REGION Network 34: TMP - ERROR - Protrusión
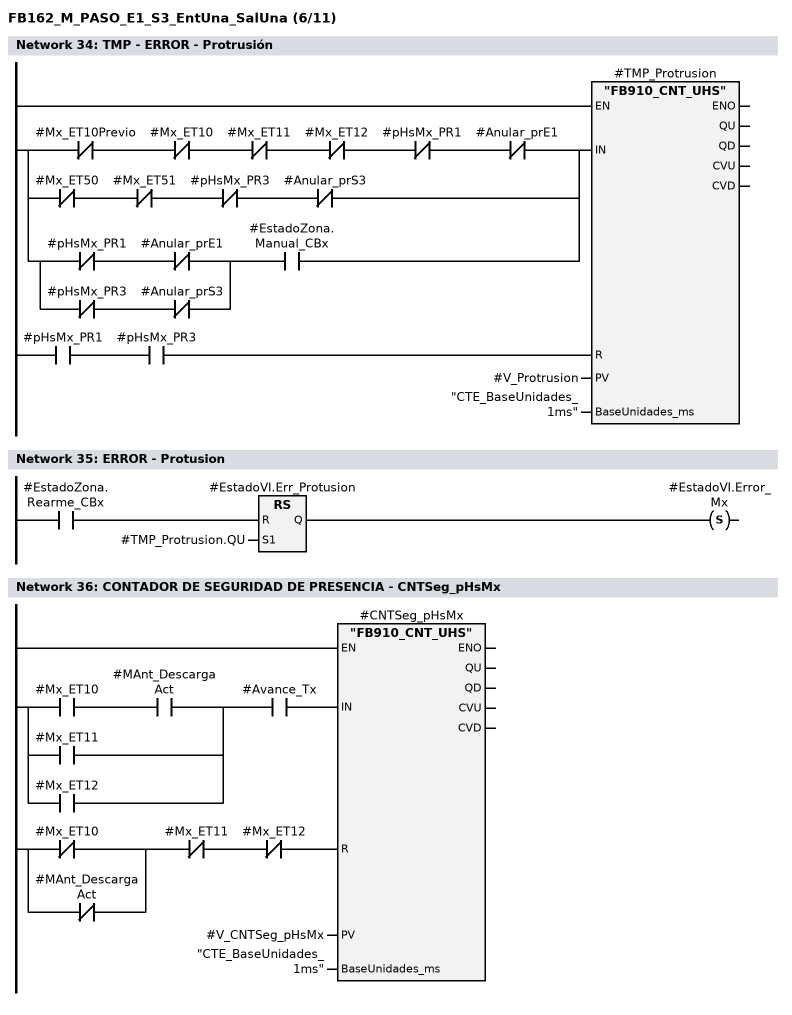
   RUNG wire#powerrail
      #TMP_Protrusion(IN := wire#w2, R := wire#w3, PV := #V_Protrusion, BaseUnidades_ms := "CTE_BaseUnidades_1ms", QU =>, QD =>, CVU =>, CVD =>)
   END_RUNG
   RUNG wire#powerrail
      I_Contact( #Mx_ET10Previo )
      I_Contact( #Mx_ET10 )
      I_Contact( #Mx_ET11 )
      I_Contact( #Mx_ET12 )
      I_Contact( #pHsMx_PR1 )
      I_Contact( #Anular_prE1 )
   END_RUNG wire#w2
   RUNG wire#powerrail
      I_Contact( #Mx_ET50 )
      I_Contact( #Mx_ET51 )
      I_Contact( #pHsMx_PR3 )
      I_Contact( #Anular_prS3 )
   END_RUNG wire#w2
   RUNG wire#powerrail
      I_Contact( #pHsMx_PR1 )
      I_Contact( #Anular_prE1 )
      wire#w1
      Contact( #EstadoZona.Manual_CBx )
   END_RUNG wire#w2
   RUNG wire#powerrail
      I_Contact( #pHsMx_PR3 )
      I_Contact( #Anular_prS3 )
   END_RUNG wire#w1
   RUNG wire#powerrail
      Contact( #pHsMx_PR1 )
      Contact( #pHsMx_PR3 )
   END_RUNG wire#w3
   // the same network as SCL:
   #TMP_Protrusion(IN := (NOT #Mx_ET10Previo AND NOT #Mx_ET10 AND NOT #Mx_ET11 AND NOT #Mx_ET12 AND NOT #pHsMx_PR1 AND NOT #Anular_prE1) OR (NOT #Mx_ET50 AND NOT #Mx_ET51 AND NOT #pHsMx_PR3 AND NOT #Anular_prS3) OR (((NOT #pHsMx_PR1 AND NOT #Anular_prE1) OR (NOT #pHsMx_PR3 AND NOT #Anular_prS3)) AND #EstadoZona.Manual_CBx),   // "FB910_CNT_UHS"
                   R := #pHsMx_PR1 AND #pHsMx_PR3,
                   PV := #V_Protrusion,
                   BaseUnidades_ms := "CTE_BaseUnidades_1ms");
END_REGION

REGION Network 35: ERROR - Protusion
   RUNG wire#powerrail
      Contact( #EstadoZona.Rearme_CBx )
      S_RS(operand := #EstadoVI.Err_Protusion, s1 := #TMP_Protrusion.QU)
      S_Coil( #EstadoVI.Error_Mx )
   END_RUNG
   // the same network as SCL:
   IF #EstadoZona.Rearme_CBx THEN
       #EstadoVI.Err_Protusion := FALSE;   // RS flip-flop
   END_IF;
   IF #TMP_Protrusion.QU THEN #EstadoVI.Err_Protusion := TRUE; END_IF;
   IF #EstadoVI.Err_Protusion THEN #EstadoVI.Error_Mx := TRUE; END_IF;
END_REGION

REGION Network 36: CONTADOR DE SEGURIDAD DE PRESENCIA - CNTSeg_pHsMx
   RUNG wire#powerrail
      #CNTSeg_pHsMx(IN := wire#w2, R := wire#w4, PV := #V_CNTSeg_pHsMx, BaseUnidades_ms := "CTE_BaseUnidades_1ms", QU =>, QD =>, CVU =>, CVD =>)
   END_RUNG
   RUNG wire#powerrail
      Contact( #Mx_ET10 )
      Contact( #MAnt_DescargaAct )
      wire#w1
      Contact( #Avance_Tx )
   END_RUNG wire#w2
   RUNG wire#powerrail
      Contact( #Mx_ET11 )
   END_RUNG wire#w1
   RUNG wire#powerrail
      Contact( #Mx_ET12 )
   END_RUNG wire#w1
   RUNG wire#powerrail
      I_Contact( #Mx_ET10 )
      wire#w3
      I_Contact( #Mx_ET11 )
      I_Contact( #Mx_ET12 )
   END_RUNG wire#w4
   RUNG wire#powerrail
      I_Contact( #MAnt_DescargaAct )
   END_RUNG wire#w3
   // the same network as SCL:
   #CNTSeg_pHsMx(IN := ((#Mx_ET10 AND #MAnt_DescargaAct) OR #Mx_ET11 OR #Mx_ET12) AND #Avance_Tx,   // "FB910_CNT_UHS"
                 R := (NOT #Mx_ET10 OR NOT #MAnt_DescargaAct) AND NOT #Mx_ET11 AND NOT #Mx_ET12,
                 PV := #V_CNTSeg_pHsMx,
                 BaseUnidades_ms := "CTE_BaseUnidades_1ms");
END_REGION

REGION Network 37: CONTADOR DE PRESENCIA - CNT_pHsMx
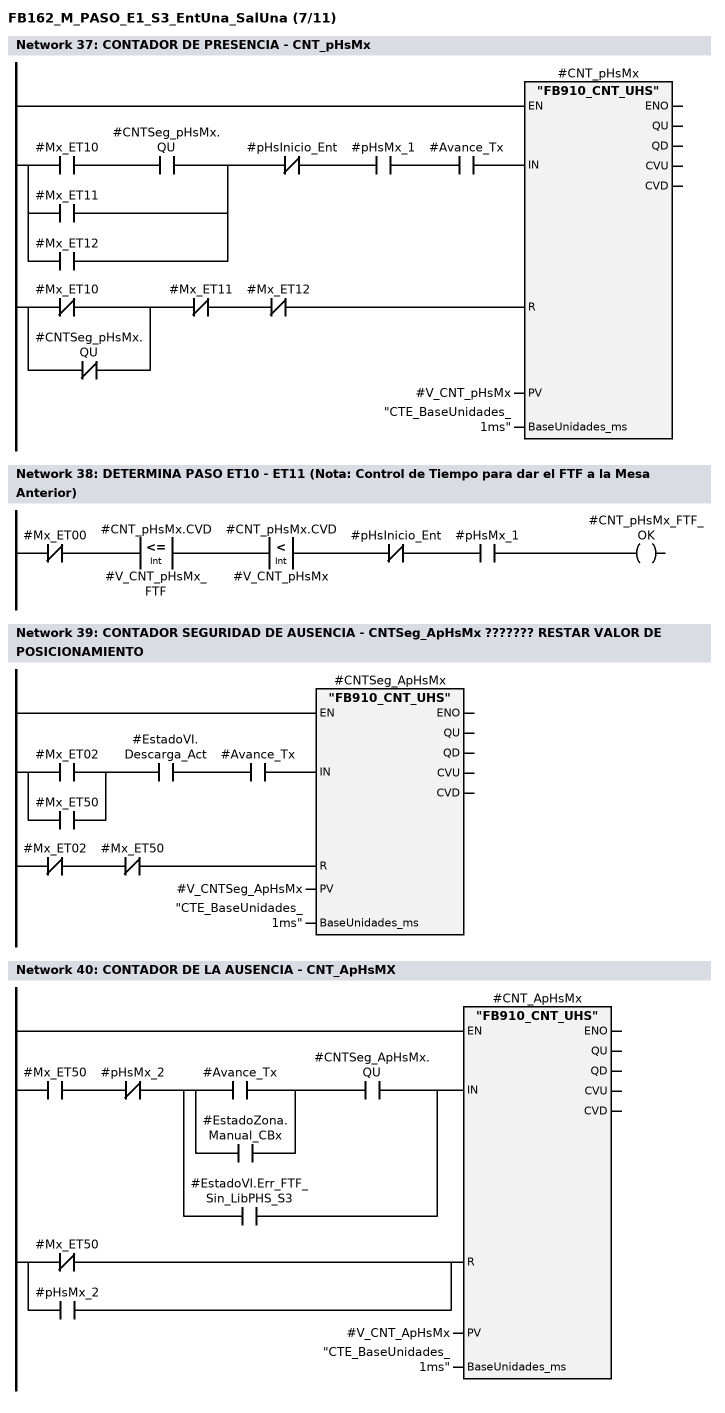
   RUNG wire#powerrail
      #CNT_pHsMx(IN := wire#w2, R := wire#w4, PV := #V_CNT_pHsMx, BaseUnidades_ms := "CTE_BaseUnidades_1ms", QU =>, QD =>, CVU =>, CVD =>)
   END_RUNG
   RUNG wire#powerrail
      Contact( #Mx_ET10 )
      Contact( #CNTSeg_pHsMx.QU )
      wire#w1
      I_Contact( #pHsInicio_Ent )
      Contact( #pHsMx_1 )
      Contact( #Avance_Tx )
   END_RUNG wire#w2
   RUNG wire#powerrail
      Contact( #Mx_ET11 )
   END_RUNG wire#w1
   RUNG wire#powerrail
      Contact( #Mx_ET12 )
   END_RUNG wire#w1
   RUNG wire#powerrail
      I_Contact( #Mx_ET10 )
      wire#w3
      I_Contact( #Mx_ET11 )
      I_Contact( #Mx_ET12 )
   END_RUNG wire#w4
   RUNG wire#powerrail
      I_Contact( #CNTSeg_pHsMx.QU )
   END_RUNG wire#w3
   // the same network as SCL:
   #CNT_pHsMx(IN := ((#Mx_ET10 AND #CNTSeg_pHsMx.QU) OR #Mx_ET11 OR #Mx_ET12) AND NOT #pHsInicio_Ent AND #pHsMx_1 AND #Avance_Tx,   // "FB910_CNT_UHS"
              R := (NOT #Mx_ET10 OR NOT #CNTSeg_pHsMx.QU) AND NOT #Mx_ET11 AND NOT #Mx_ET12,
              PV := #V_CNT_pHsMx,
              BaseUnidades_ms := "CTE_BaseUnidades_1ms");
END_REGION

REGION Network 38: DETERMINA PASO ET10 - ET11 (Nota: Control de Tiempo para dar el FTF a la Mesa Anterior)
   RUNG wire#powerrail
      I_Contact( #Mx_ET00 )
      { S7_Templates := "SrcType := Int" } LE_Contact(in1 := #CNT_pHsMx.CVD, in2 := #V_CNT_pHsMx_FTF)
      { S7_Templates := "SrcType := Int" } LT_Contact(in1 := #CNT_pHsMx.CVD, in2 := #V_CNT_pHsMx)
      I_Contact( #pHsInicio_Ent )
      Contact( #pHsMx_1 )
      Coil( #CNT_pHsMx_FTF_OK )
   END_RUNG
   // the same network as SCL:
   #CNT_pHsMx_FTF_OK := NOT #Mx_ET00 AND (#CNT_pHsMx.CVD <= #V_CNT_pHsMx_FTF) AND (#CNT_pHsMx.CVD < #V_CNT_pHsMx) AND NOT #pHsInicio_Ent AND #pHsMx_1;
END_REGION

REGION Network 39: CONTADOR SEGURIDAD DE AUSENCIA - CNTSeg_ApHsMx ??????? RESTAR VALOR DE POSICIONAMIENTO
   RUNG wire#powerrail
      #CNTSeg_ApHsMx(IN := wire#w2, R := wire#w3, PV := #V_CNTSeg_ApHsMx, BaseUnidades_ms := "CTE_BaseUnidades_1ms", QU =>, QD =>, CVU =>, CVD =>)
   END_RUNG
   RUNG wire#powerrail
      Contact( #Mx_ET02 )
      wire#w1
      Contact( #EstadoVI.Descarga_Act )
      Contact( #Avance_Tx )
   END_RUNG wire#w2
   RUNG wire#powerrail
      Contact( #Mx_ET50 )
   END_RUNG wire#w1
   RUNG wire#powerrail
      I_Contact( #Mx_ET02 )
      I_Contact( #Mx_ET50 )
   END_RUNG wire#w3
   // the same network as SCL:
   #CNTSeg_ApHsMx(IN := (#Mx_ET02 OR #Mx_ET50) AND #EstadoVI.Descarga_Act AND #Avance_Tx,   // "FB910_CNT_UHS"
                  R := NOT #Mx_ET02 AND NOT #Mx_ET50,
                  PV := #V_CNTSeg_ApHsMx,
                  BaseUnidades_ms := "CTE_BaseUnidades_1ms");
END_REGION

REGION Network 40: CONTADOR DE LA AUSENCIA - CNT_ApHsMX
   RUNG wire#powerrail
      #CNT_ApHsMx(IN := wire#w3, R := wire#w4, PV := #V_CNT_ApHsMx, BaseUnidades_ms := "CTE_BaseUnidades_1ms", QU =>, QD =>, CVU =>, CVD =>)
   END_RUNG
   RUNG wire#powerrail
      Contact( #Mx_ET50 )
      I_Contact( #pHsMx_2 )
      wire#w1
      Contact( #Avance_Tx )
      wire#w2
      Contact( #CNTSeg_ApHsMx.QU )
   END_RUNG wire#w3
   RUNG wire#w1
      Contact( #EstadoZona.Manual_CBx )
   END_RUNG wire#w2
   RUNG wire#w1
      Contact( #EstadoVI.Err_FTF_Sin_LibPHS_S3 )
   END_RUNG wire#w3
   RUNG wire#powerrail
      I_Contact( #Mx_ET50 )
   END_RUNG wire#w4
   RUNG wire#powerrail
      Contact( #pHsMx_2 )
   END_RUNG wire#w4
   // the same network as SCL:
   #CNT_ApHsMx(IN := #Mx_ET50 AND NOT #pHsMx_2 AND (((#Avance_Tx OR #EstadoZona.Manual_CBx) AND #CNTSeg_ApHsMx.QU) OR #EstadoVI.Err_FTF_Sin_LibPHS_S3),   // "FB910_CNT_UHS"
               R := NOT #Mx_ET50 OR #pHsMx_2,
               PV := #V_CNT_ApHsMx,
               BaseUnidades_ms := "CTE_BaseUnidades_1ms");
END_REGION

REGION Network 41: VARIABLES AUXILIARES - Fin de Reset
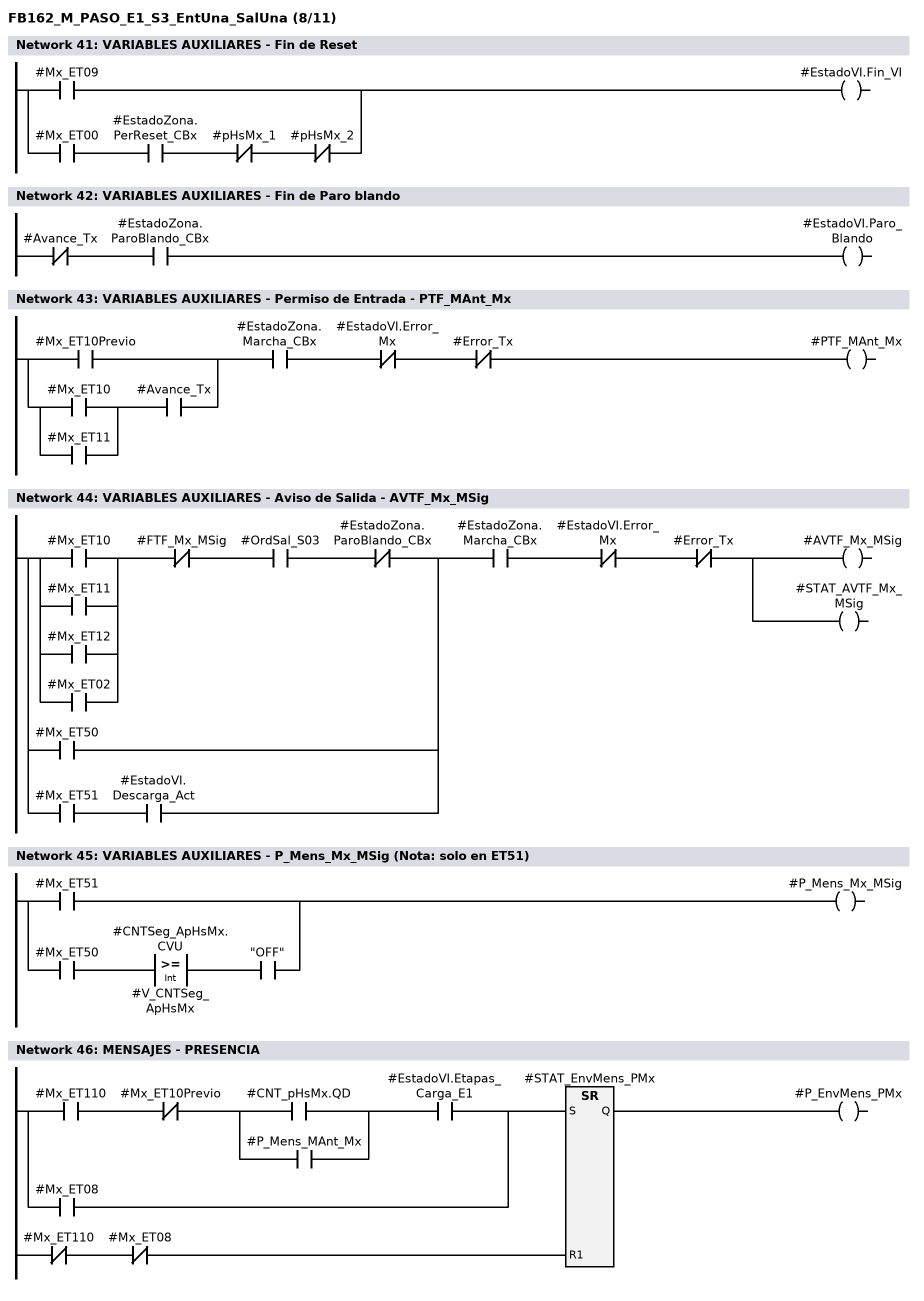
   RUNG wire#powerrail
      Contact( #Mx_ET09 )
      wire#w1
      Coil( #EstadoVI.Fin_VI )
   END_RUNG
   RUNG wire#powerrail
      Contact( #Mx_ET00 )
      Contact( #EstadoZona.PerReset_CBx )
      I_Contact( #pHsMx_1 )
      I_Contact( #pHsMx_2 )
   END_RUNG wire#w1
   // the same network as SCL:
   #EstadoVI.Fin_VI := #Mx_ET09 OR (#Mx_ET00 AND #EstadoZona.PerReset_CBx AND NOT #pHsMx_1 AND NOT #pHsMx_2);
END_REGION

REGION Network 42: VARIABLES AUXILIARES - Fin de Paro blando
   RUNG wire#powerrail
      I_Contact( #Avance_Tx )
      Contact( #EstadoZona.ParoBlando_CBx )
      Coil( #EstadoVI.Paro_Blando )
   END_RUNG
   // the same network as SCL:
   #EstadoVI.Paro_Blando := NOT #Avance_Tx AND #EstadoZona.ParoBlando_CBx;
END_REGION

REGION Network 43: VARIABLES AUXILIARES - Permiso de Entrada - PTF_MAnt_Mx
   RUNG wire#powerrail
      Contact( #Mx_ET10Previo )
      wire#w1
      Contact( #EstadoZona.Marcha_CBx )
      I_Contact( #EstadoVI.Error_Mx )
      I_Contact( #Error_Tx )
      Coil( #PTF_MAnt_Mx )
   END_RUNG
   RUNG wire#powerrail
      Contact( #Mx_ET10 )
      wire#w2
      Contact( #Avance_Tx )
   END_RUNG wire#w1
   RUNG wire#powerrail
      Contact( #Mx_ET11 )
   END_RUNG wire#w2
   // the same network as SCL:
   #PTF_MAnt_Mx := (#Mx_ET10Previo OR ((#Mx_ET10 OR #Mx_ET11) AND #Avance_Tx)) AND #EstadoZona.Marcha_CBx AND NOT #EstadoVI.Error_Mx AND NOT #Error_Tx;
END_REGION

REGION Network 44: VARIABLES AUXILIARES - Aviso de Salida - AVTF_Mx_MSig
   RUNG wire#powerrail
      Contact( #Mx_ET10 )
      wire#w1
      I_Contact( #FTF_Mx_MSig )
      Contact( #OrdSal_S03 )
      I_Contact( #EstadoZona.ParoBlando_CBx )
      wire#w2
      Contact( #EstadoZona.Marcha_CBx )
      I_Contact( #EstadoVI.Error_Mx )
      I_Contact( #Error_Tx )
      wire#w3
      Coil( #AVTF_Mx_MSig )
   END_RUNG
   RUNG wire#powerrail
      Contact( #Mx_ET11 )
   END_RUNG wire#w1
   RUNG wire#powerrail
      Contact( #Mx_ET12 )
   END_RUNG wire#w1
   RUNG wire#powerrail
      Contact( #Mx_ET02 )
   END_RUNG wire#w1
   RUNG wire#powerrail
      Contact( #Mx_ET50 )
   END_RUNG wire#w2
   RUNG wire#powerrail
      Contact( #Mx_ET51 )
      Contact( #EstadoVI.Descarga_Act )
   END_RUNG wire#w2
   RUNG wire#w3
      Coil( #STAT_AVTF_Mx_MSig )
   END_RUNG
   // the same network as SCL:
   #AVTF_Mx_MSig := (((#Mx_ET10 OR #Mx_ET11 OR #Mx_ET12 OR #Mx_ET02) AND NOT #FTF_Mx_MSig AND #OrdSal_S03 AND NOT #EstadoZona.ParoBlando_CBx) OR #Mx_ET50 OR (#Mx_ET51 AND #EstadoVI.Descarga_Act)) AND #EstadoZona.Marcha_CBx AND NOT #EstadoVI.Error_Mx AND NOT #Error_Tx;
   #STAT_AVTF_Mx_MSig := #AVTF_Mx_MSig;
END_REGION

REGION Network 45: VARIABLES AUXILIARES - P_Mens_Mx_MSig (Nota: solo en ET51)
   RUNG wire#powerrail
      Contact( #Mx_ET51 )
      wire#w1
      Coil( #P_Mens_Mx_MSig )
   END_RUNG
   RUNG wire#powerrail
      Contact( #Mx_ET50 )
      { S7_Templates := "SrcType := Int" } GE_Contact(in1 := #CNTSeg_ApHsMx.CVU, in2 := #V_CNTSeg_ApHsMx)
      Contact( "OFF" )
   END_RUNG wire#w1
   // the same network as SCL:
   #P_Mens_Mx_MSig := #Mx_ET51 OR (#Mx_ET50 AND (#CNTSeg_ApHsMx.CVU >= #V_CNTSeg_ApHsMx) AND "OFF");
END_REGION

REGION Network 46: MENSAJES - PRESENCIA
   RUNG wire#powerrail
      Contact( #Mx_ET110 )
      I_Contact( #Mx_ET10Previo )
      wire#w1
      Contact( #CNT_pHsMx.QD )
      wire#w2
      Contact( #EstadoVI.Etapas_Carga_E1 )
      wire#w3
      S_SR(operand := #STAT_EnvMens_PMx, r1 := wire#w4)
      Coil( #P_EnvMens_PMx )
   END_RUNG
   RUNG wire#w1
      Contact( #P_Mens_MAnt_Mx )
   END_RUNG wire#w2
   RUNG wire#powerrail
      Contact( #Mx_ET08 )
   END_RUNG wire#w3
   RUNG wire#powerrail
      I_Contact( #Mx_ET110 )
      I_Contact( #Mx_ET08 )
   END_RUNG wire#w4
   // the same network as SCL:
   IF (#Mx_ET110 AND NOT #Mx_ET10Previo AND (#CNT_pHsMx.QD OR #P_Mens_MAnt_Mx) AND #EstadoVI.Etapas_Carga_E1) OR #Mx_ET08 THEN
       #STAT_EnvMens_PMx := TRUE;   // SR flip-flop
   END_IF;
   IF NOT #Mx_ET110 AND NOT #Mx_ET08 THEN #STAT_EnvMens_PMx := FALSE; END_IF;
   #P_EnvMens_PMx := #STAT_EnvMens_PMx;
END_REGION

REGION Network 47: MENSAJES - PROTOCOLO INICIADO
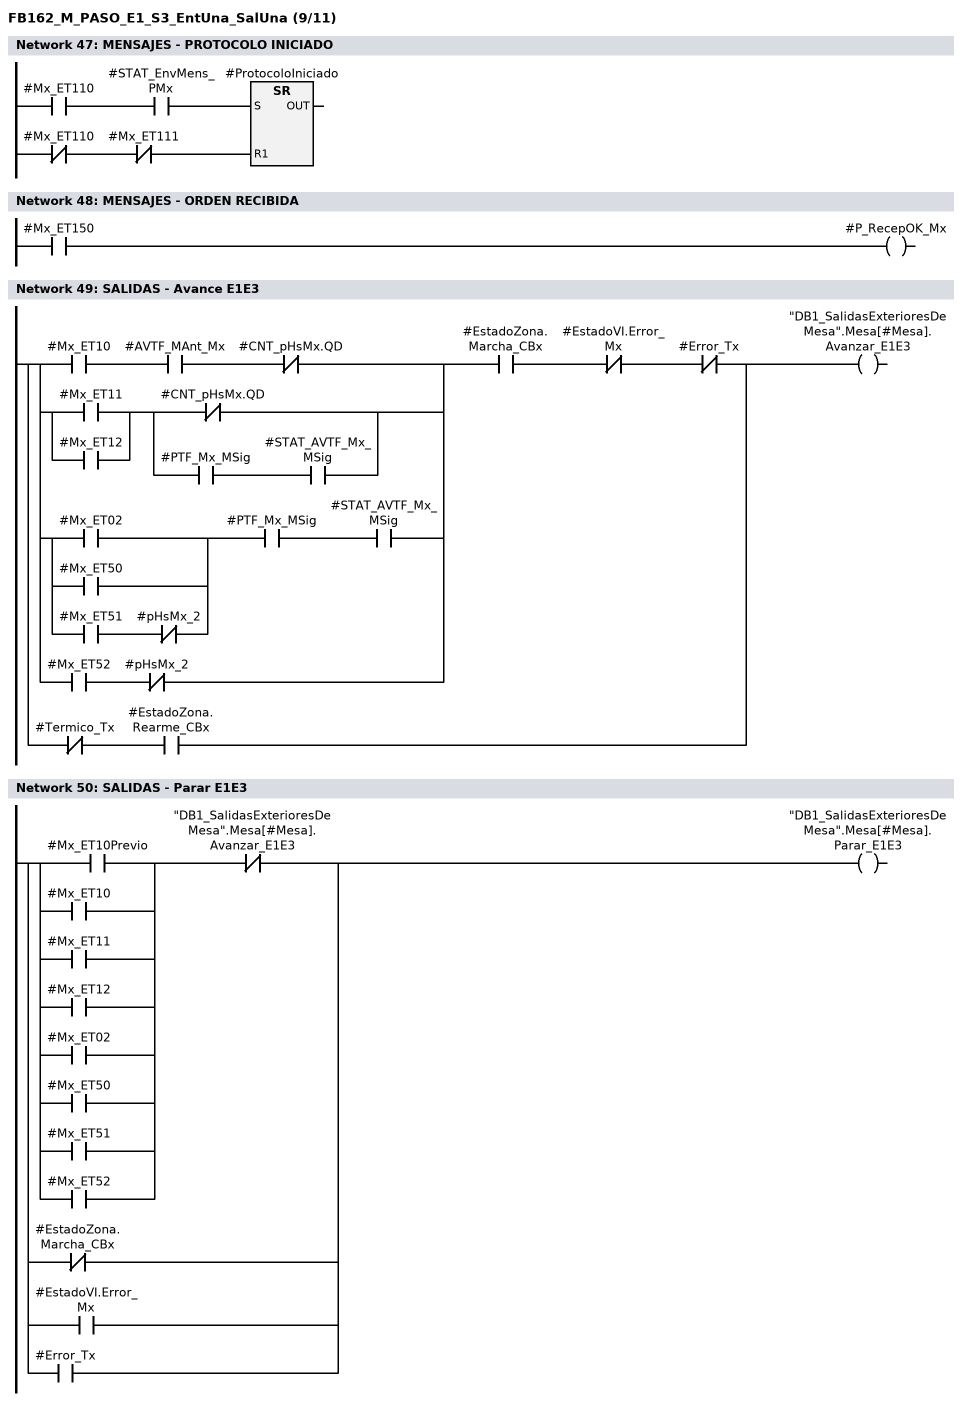
   RUNG wire#powerrail
      Contact( #Mx_ET110 )
      Contact( #STAT_EnvMens_PMx )
      S_SR(operand := #ProtocoloIniciado, r1 := wire#w1)
   END_RUNG
   RUNG wire#powerrail
      I_Contact( #Mx_ET110 )
      I_Contact( #Mx_ET111 )
   END_RUNG wire#w1
   // the same network as SCL:
   IF #Mx_ET110 AND #STAT_EnvMens_PMx THEN
       #ProtocoloIniciado := TRUE;   // SR flip-flop
   END_IF;
   IF NOT #Mx_ET110 AND NOT #Mx_ET111 THEN #ProtocoloIniciado := FALSE; END_IF;
END_REGION

REGION Network 48: MENSAJES - ORDEN RECIBIDA
   RUNG wire#powerrail
      Contact( #Mx_ET150 )
      Coil( #P_RecepOK_Mx )
   END_RUNG
   // the same network as SCL:
   #P_RecepOK_Mx := #Mx_ET150;
END_REGION

REGION Network 49: SALIDAS - Avance E1E3
   RUNG wire#powerrail
      Contact( #Mx_ET10 )
      Contact( #AVTF_MAnt_Mx )
      I_Contact( #CNT_pHsMx.QD )
      wire#w1
      Contact( #EstadoZona.Marcha_CBx )
      I_Contact( #EstadoVI.Error_Mx )
      I_Contact( #Error_Tx )
      wire#w4
      Coil( "DB1_SalidasExterioresDeMesa".Mesa[#Mesa].Avanzar_E1E3 )
   END_RUNG
   RUNG wire#powerrail
      Contact( #Mx_ET11 )
      wire#w2
      I_Contact( #CNT_pHsMx.QD )
   END_RUNG wire#w1
   RUNG wire#powerrail
      Contact( #Mx_ET12 )
   END_RUNG wire#w2
   RUNG wire#w2
      Contact( #PTF_Mx_MSig )
      Contact( #STAT_AVTF_Mx_MSig )
   END_RUNG wire#w1
   RUNG wire#powerrail
      Contact( #Mx_ET02 )
      wire#w3
      Contact( #PTF_Mx_MSig )
      Contact( #STAT_AVTF_Mx_MSig )
   END_RUNG wire#w1
   RUNG wire#powerrail
      Contact( #Mx_ET50 )
   END_RUNG wire#w3
   RUNG wire#powerrail
      Contact( #Mx_ET51 )
      I_Contact( #pHsMx_2 )
   END_RUNG wire#w3
   RUNG wire#powerrail
      Contact( #Mx_ET52 )
      I_Contact( #pHsMx_2 )
   END_RUNG wire#w1
   RUNG wire#powerrail
      I_Contact( #Termico_Tx )
      Contact( #EstadoZona.Rearme_CBx )
   END_RUNG wire#w4
   // the same network as SCL:
   "DB1_SalidasExterioresDeMesa".Mesa[#Mesa].Avanzar_E1E3 := (((#Mx_ET10 AND #AVTF_MAnt_Mx AND NOT #CNT_pHsMx.QD) OR ((#Mx_ET11 OR #Mx_ET12) AND (NOT #CNT_pHsMx.QD OR (#PTF_Mx_MSig AND #STAT_AVTF_Mx_MSig))) OR ((#Mx_ET02 OR #Mx_ET50 OR (#Mx_ET51 AND NOT #pHsMx_2)) AND #PTF_Mx_MSig AND #STAT_AVTF_Mx_MSig) OR (#Mx_ET52 AND NOT #pHsMx_2)) AND #EstadoZona.Marcha_CBx AND NOT #EstadoVI.Error_Mx AND NOT #Error_Tx) OR (NOT #Termico_Tx AND #EstadoZona.Rearme_CBx);
END_REGION

REGION Network 50: SALIDAS - Parar E1E3
   RUNG wire#powerrail
      Contact( #Mx_ET10Previo )
      wire#w1
      I_Contact( "DB1_SalidasExterioresDeMesa".Mesa[#Mesa].Avanzar_E1E3 )
      wire#w2
      Coil( "DB1_SalidasExterioresDeMesa".Mesa[#Mesa].Parar_E1E3 )
   END_RUNG
   RUNG wire#powerrail
      Contact( #Mx_ET10 )
   END_RUNG wire#w1
   RUNG wire#powerrail
      Contact( #Mx_ET11 )
   END_RUNG wire#w1
   RUNG wire#powerrail
      Contact( #Mx_ET12 )
   END_RUNG wire#w1
   RUNG wire#powerrail
      Contact( #Mx_ET02 )
   END_RUNG wire#w1
   RUNG wire#powerrail
      Contact( #Mx_ET50 )
   END_RUNG wire#w1
   RUNG wire#powerrail
      Contact( #Mx_ET51 )
   END_RUNG wire#w1
   RUNG wire#powerrail
      Contact( #Mx_ET52 )
   END_RUNG wire#w1
   RUNG wire#powerrail
      I_Contact( #EstadoZona.Marcha_CBx )
   END_RUNG wire#w2
   RUNG wire#powerrail
      Contact( #EstadoVI.Error_Mx )
   END_RUNG wire#w2
   RUNG wire#powerrail
      Contact( #Error_Tx )
   END_RUNG wire#w2
   // the same network as SCL:
   "DB1_SalidasExterioresDeMesa".Mesa[#Mesa].Parar_E1E3 := ((#Mx_ET10Previo OR #Mx_ET10 OR #Mx_ET11 OR #Mx_ET12 OR #Mx_ET02 OR #Mx_ET50 OR #Mx_ET51 OR #Mx_ET52) AND NOT "DB1_SalidasExterioresDeMesa".Mesa[#Mesa].Avanzar_E1E3) OR NOT #EstadoZona.Marcha_CBx OR #EstadoVI.Error_Mx OR #Error_Tx;
END_REGION

REGION Network 51: SALIDAS - Valor Frecuencia Lenta E1E3
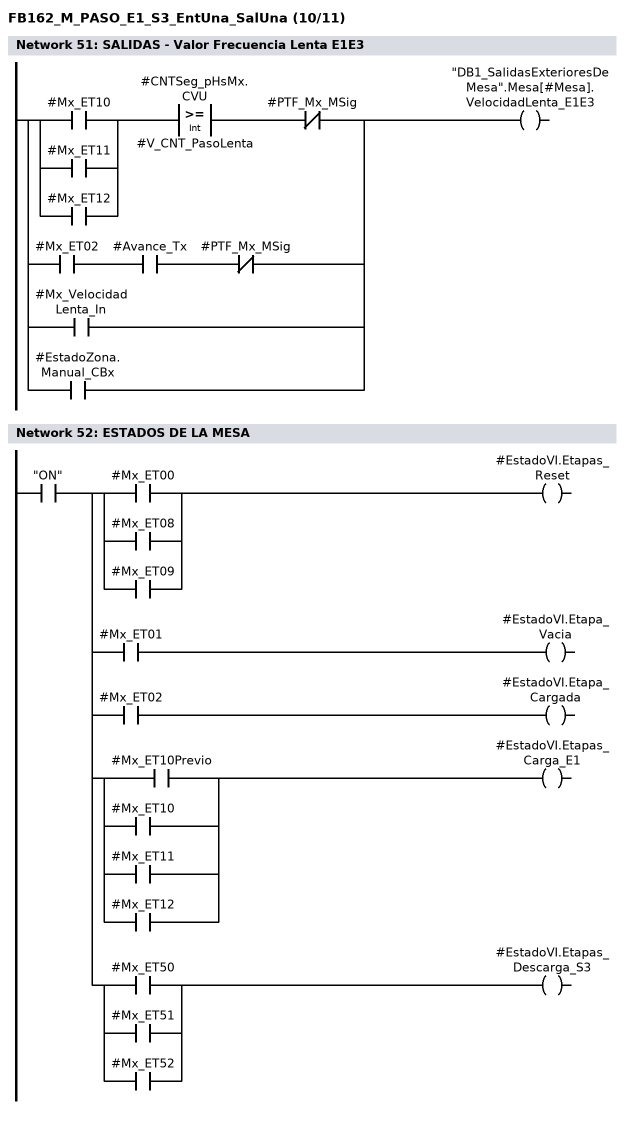
   RUNG wire#powerrail
      Contact( #Mx_ET10 )
      wire#w1
      { S7_Templates := "SrcType := Int" } GE_Contact(in1 := #CNTSeg_pHsMx.CVU, in2 := #V_CNT_PasoLenta)
      I_Contact( #PTF_Mx_MSig )
      wire#w2
      Coil( "DB1_SalidasExterioresDeMesa".Mesa[#Mesa].VelocidadLenta_E1E3 )
   END_RUNG
   RUNG wire#powerrail
      Contact( #Mx_ET11 )
   END_RUNG wire#w1
   RUNG wire#powerrail
      Contact( #Mx_ET12 )
   END_RUNG wire#w1
   RUNG wire#powerrail
      Contact( #Mx_ET02 )
      Contact( #Avance_Tx )
      I_Contact( #PTF_Mx_MSig )
   END_RUNG wire#w2
   RUNG wire#powerrail
      Contact( #Mx_VelocidadLenta_In )
   END_RUNG wire#w2
   RUNG wire#powerrail
      Contact( #EstadoZona.Manual_CBx )
   END_RUNG wire#w2
   // the same network as SCL:
   "DB1_SalidasExterioresDeMesa".Mesa[#Mesa].VelocidadLenta_E1E3 := ((#Mx_ET10 OR #Mx_ET11 OR #Mx_ET12) AND (#CNTSeg_pHsMx.CVU >= #V_CNT_PasoLenta) AND NOT #PTF_Mx_MSig) OR (#Mx_ET02 AND #Avance_Tx AND NOT #PTF_Mx_MSig) OR #Mx_VelocidadLenta_In OR #EstadoZona.Manual_CBx;
END_REGION

REGION Network 52: ESTADOS DE LA MESA
   RUNG wire#powerrail
      Contact( "ON" )
      wire#w1
      Contact( #Mx_ET00 )
      wire#w2
      Coil( #EstadoVI.Etapas_Reset )
   END_RUNG
   RUNG wire#w1
      Contact( #Mx_ET08 )
   END_RUNG wire#w2
   RUNG wire#w1
      Contact( #Mx_ET09 )
   END_RUNG wire#w2
   RUNG wire#w1
      Contact( #Mx_ET01 )
      Coil( #EstadoVI.Etapa_Vacia )
   END_RUNG
   RUNG wire#w1
      Contact( #Mx_ET02 )
      Coil( #EstadoVI.Etapa_Cargada )
   END_RUNG
   RUNG wire#w1
      Contact( #Mx_ET10Previo )
      wire#w3
      Coil( #EstadoVI.Etapas_Carga_E1 )
   END_RUNG
   RUNG wire#w1
      Contact( #Mx_ET10 )
   END_RUNG wire#w3
   RUNG wire#w1
      Contact( #Mx_ET11 )
   END_RUNG wire#w3
   RUNG wire#w1
      Contact( #Mx_ET12 )
   END_RUNG wire#w3
   RUNG wire#w1
      Contact( #Mx_ET50 )
      wire#w4
      Coil( #EstadoVI.Etapas_Descarga_S3 )
   END_RUNG
   RUNG wire#w1
      Contact( #Mx_ET51 )
   END_RUNG wire#w4
   RUNG wire#w1
      Contact( #Mx_ET52 )
   END_RUNG wire#w4
   // the same network as SCL:
   #EstadoVI.Etapas_Reset := "ON" AND (#Mx_ET00 OR #Mx_ET08 OR #Mx_ET09);
   #EstadoVI.Etapa_Vacia := "ON" AND #Mx_ET01;
   #EstadoVI.Etapa_Cargada := "ON" AND #Mx_ET02;
   #EstadoVI.Etapas_Carga_E1 := "ON" AND (#Mx_ET10Previo OR #Mx_ET10 OR #Mx_ET11 OR #Mx_ET12);
   #EstadoVI.Etapas_Descarga_S3 := "ON" AND (#Mx_ET50 OR #Mx_ET51 OR #Mx_ET52);
END_REGION

REGION Network 53: ENTRADAS DE LA MESA
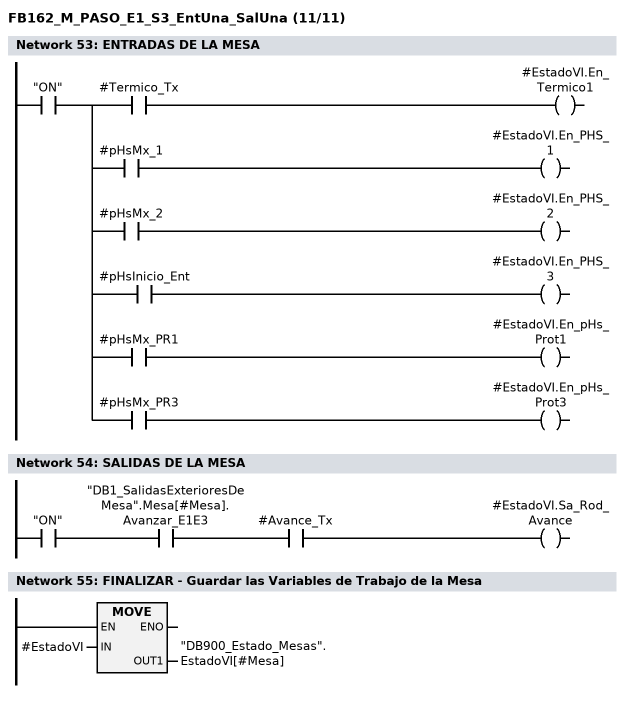
   RUNG wire#powerrail
      Contact( "ON" )
      wire#w1
      Contact( #Termico_Tx )
      Coil( #EstadoVI.En_Termico1 )
   END_RUNG
   RUNG wire#w1
      Contact( #pHsMx_1 )
      Coil( #EstadoVI.En_PHS_1 )
   END_RUNG
   RUNG wire#w1
      Contact( #pHsMx_2 )
      Coil( #EstadoVI.En_PHS_2 )
   END_RUNG
   RUNG wire#w1
      Contact( #pHsInicio_Ent )
      Coil( #EstadoVI.En_PHS_3 )
   END_RUNG
   RUNG wire#w1
      Contact( #pHsMx_PR1 )
      Coil( #EstadoVI.En_pHs_Prot1 )
   END_RUNG
   RUNG wire#w1
      Contact( #pHsMx_PR3 )
      Coil( #EstadoVI.En_pHs_Prot3 )
   END_RUNG
   // the same network as SCL:
   #EstadoVI.En_Termico1 := "ON" AND #Termico_Tx;
   #EstadoVI.En_PHS_1 := "ON" AND #pHsMx_1;
   #EstadoVI.En_PHS_2 := "ON" AND #pHsMx_2;
   #EstadoVI.En_PHS_3 := "ON" AND #pHsInicio_Ent;
   #EstadoVI.En_pHs_Prot1 := "ON" AND #pHsMx_PR1;
   #EstadoVI.En_pHs_Prot3 := "ON" AND #pHsMx_PR3;
END_REGION

REGION Network 54: SALIDAS DE LA MESA
   RUNG wire#powerrail
      Contact( "ON" )
      Contact( "DB1_SalidasExterioresDeMesa".Mesa[#Mesa].Avanzar_E1E3 )
      Contact( #Avance_Tx )
      Coil( #EstadoVI.Sa_Rod_Avance )
   END_RUNG
   // the same network as SCL:
   #EstadoVI.Sa_Rod_Avance := "ON" AND "DB1_SalidasExterioresDeMesa".Mesa[#Mesa].Avanzar_E1E3 AND #Avance_Tx;
END_REGION

REGION Network 55: FINALIZAR - Guardar las Variables de Trabajo de la Mesa
   RUNG wire#powerrail
      Move(in := #EstadoVI, out1 => "DB900_Estado_Mesas".EstadoVI[#Mesa])
   END_RUNG
   // the same network as SCL:
   "DB900_Estado_Mesas".EstadoVI[#Mesa] := #EstadoVI;
END_REGION
END_FUNCTION_BLOCK

FUNCTION_BLOCK "FB201_M_CS_Carga"   // FB201, LAD
TITLE = Control del Ramal de Salidas
{ S7_Optimized_Access := 'FALSE' }
AUTHOR : TE_CS
NAME : 20160509
VERSION : 3.4
// stored: AutoNumber false, SetENOAutomatically false
   VAR_INPUT
      Mesa : UInt;   // Mesa de la FB
      Error_Tx : Bool;   // Error en el Tx
      EnTension : Bool;   // Existe Tension en la Mesa
      Termico_Tx : Bool;   // Proteccion del Tx
      pHsMx : Bool;   // pHs de la Mesa
      pHsMx_PR1 : Bool;   // pHs de Protrusion de la Mesa. Nota: No existe >> ON
      pHsMx_PR3 : Bool;   // pHs de Protrusion de la Mesa. Nota: No existe >> ON
      Avance_Tx : Bool;   // Avance del Tx
      TP1_Up : Bool;   // TP1 Arriba. Nota Movimiento E1 >> S3
      TP1_Down : Bool;   // TP1 Abajo. Nota Movimiento E1 >> S3
      EnMovimiento_TP1 : Bool;   // En movimiento el TP1
      TE_MoveOK : Bool;   // Move OK del TE (Horquilla Centrada)
      TE_OFFLine : Bool;   // OFF Line del TE
      TE_PotenciaOK : Bool;   // Potencia OK del TE
      MAnt_DescargaAct : Bool;   // E1 >> Mesa Anterior DescargaAct
      AVTF_MAnt_Mx : Bool;   // E1 >> Mesa Anterior AVTF
      P_Mens_MAnt_Mx : Bool;   // E1 >> Mesa Anterior P_Mens
      PTF_Mx_MSig : Bool;   // S3 >> Mesa Siguiente PTF
      FTF_Mx_MSig : Bool;   // S3 >> Mesa Siguiente FTF
      Mx_VelocidadLenta_In : Bool;   // Forzar a Velociada Lenta
      F_EnvMens_Mx : Bool;   // Fin de Envio de Mensaje
      OrdSal_S03 : Bool;   // Orden de Salida por S03
      OrdSal_S00 : Bool;   // Orden de Salida por S00 (TE)
      V_CNT_pHsMx : Int := 1000;   // Valor de Presencia
      V_CNT_pHsMx_FTF : Int := 200;   // Valor para activar FTF. Nota: < = V_CNT_pHsMx.
      V_CNTSeg_pHsMx : Int := 2000;   // Valor de Seguriadad para Presencia
      V_Subir_TP_Min : Int := 2000;   // Valor Minimo para Subir Tope
      V_Bajar_TP_Max : Int := 4000;   // Valor Maximo para Bajar Tope
      V_CNT_PasoLenta : Int := 2000;   // Valor de Paso a Lenta
      V_CNT_ApHsMx : Int := 200;   // Valor de Ausencia
      V_CNTSeg_ApHsMx : Int := 2000;   // Valor de Seguriadad para Ausencia
      V_CNT_Simultaneo : Int := 2000;   // Valor de Simultaneo
      V_InicioSimultaneo : Int := 0;   // Inicio de Simultaneo. Nota: <= V_CNT_Simultaneo
      V_FinSimultaneo : Int := 0;   // Final de Simultaneo. Nota: <= V_InicioSimultaneo
      V_TOut_Tx_Mx : Int := 7000;   // TimeOut de Entrada por E1
      V_TOut_TP : Int := 5000;   // TimeOut de Tope
      V_TMP_Protrusion : Int := 200;   // TMP de Protrusion
      V_CNT_PerdidapHs : Int := 1000;   // CNT de Perdida de pHs
   END_VAR
   VAR_OUTPUT
      P_EnvMens_PMx : Bool;   // Permiso de Enviar Mensaje de Presencia
      P_EnvMens_AMx : Bool;   // Permiso de Enviar Mensaje de Ausencia
      P_RecepOK_Mx : Bool;   // Recepcion OK
      PTF_MAnt_Mx : Bool;   // E1 >> Mesa Anterior PTF
      FTF_MAnt_Mx : Bool;   // E1 >> Mesa Anterior FTF
      AVTF_Mx_MSig : Bool;   // S3 >> Mesa Siguiente AVTF
      P_Mens_Mx_MSig : Bool;   // S3 >> Mesa Siguiente P_Mens
   END_VAR
   VAR
      Anular_prE1 : Bool;   // ???
      Anular_prS3 : Bool;   // ???
      Mx_ET00 : Bool;
      Mx_ET01 : Bool;
      Mx_ET02 : Bool;
      Mx_ET08 : Bool;
      Mx_ET09 : Bool;
      Mx_ET10 : Bool;
      Mx_ET11 : Bool;
      Mx_ET12 : Bool;
      Mx_ET110 : Bool;
      Mx_ET111 : Bool;
      Mx_ET50 : Bool;
      Mx_ET51 : Bool;
      Mx_ET150 : Bool;
      Mx_ET151 : Bool;
      Mx_ET70 : Bool;
      Mx_ET71 : Bool;
      Mx_ET170 : Bool;
      Mx_ET171 : Bool;
      TE_OK : Bool;   // El TE esta Operativo
      ProtocoloIniciado : Bool;   // Iniciado el Envio del Mensaje de Presencia
      Simultaneo_Mx : Bool;   // Activo Simultaneo E1
      CNT_pHsMx_FTF_OK : Bool;   // Enviar ya FTF
      STAT_EnvMens_PMx : Bool;   // Interna >> Envio del Mensaje de Presencia
      STAT_EnvMens_AMx : Bool;   // Interna >> Envio de Mensaje de Ausencia
      STAT_FTF_MAnt_Mx : Bool;   // Interna >> FTF de MAnt >> Mx
      STAT_AVTF_Mx_MSig : Bool;   // Interna >> AVTF de Mx >> MSig
      CNT_pHsMx { S7_SetPoint := 'True'} : "FB910_CNT_UHS";   // CNT de la Presencia
      CNTSeg_pHsMx { S7_SetPoint := 'True'} : "FB910_CNT_UHS";   // CNT de Seguridad de la Presencia
      CNT_ApHsMx { S7_SetPoint := 'True'} : "FB910_CNT_UHS";   // CNT de la Ausencia
      CNTSeg_ApHsMx { S7_SetPoint := 'True'} : "FB910_CNT_UHS";   // CNT de Seguridad de la Ausencia
      CNT_Simultaneo { S7_SetPoint := 'True'} : "FB910_CNT_UHS";   // CNT de Simultaneo
      TMP_EnTension { S7_SetPoint := 'True'} : "FB910_CNT_UHS";
      TOut_Av_Mx { S7_SetPoint := 'True'} : "FB910_CNT_UHS";   // Time Out de Entrada de E1
      TOut_Subir_TP { S7_SetPoint := 'True'} : "FB910_CNT_UHS";   // Time Out de Subida del TP
      TOut_Bajar_TP { S7_SetPoint := 'True'} : "FB910_CNT_UHS";   // Time Out de Bajada del TP
      TMP_Protrusion { S7_SetPoint := 'True'} : "FB910_CNT_UHS";   // TMP de la Protrusion
      CNT_PerdidapHs { S7_SetPoint := 'True'} : "FB910_CNT_UHS";   // CNT de Perdida de pHs
      Interlock_manual : "UDT_Interlock_manual_TE_CS/FS";
   END_VAR
   VAR_TEMP
      EstadoZona : "EstadoZona";   // Estado de Zona de la Mesa
      EstadoVI : "EstadosMesa";   // Estado del Vehiculo Inteliguente de la Mesa
      ConfigFB : "UDT_ConfigFB";   // Configuracion de la FB de la Mesa
      Interlock : "UDT_Interlock_TE_CS/FS";
      V_Protrusion : Int;
      retval : Int;
      cero : USInt;
      Aux_ET00 : Bool;
   END_VAR
BEGIN

REGION Network 1
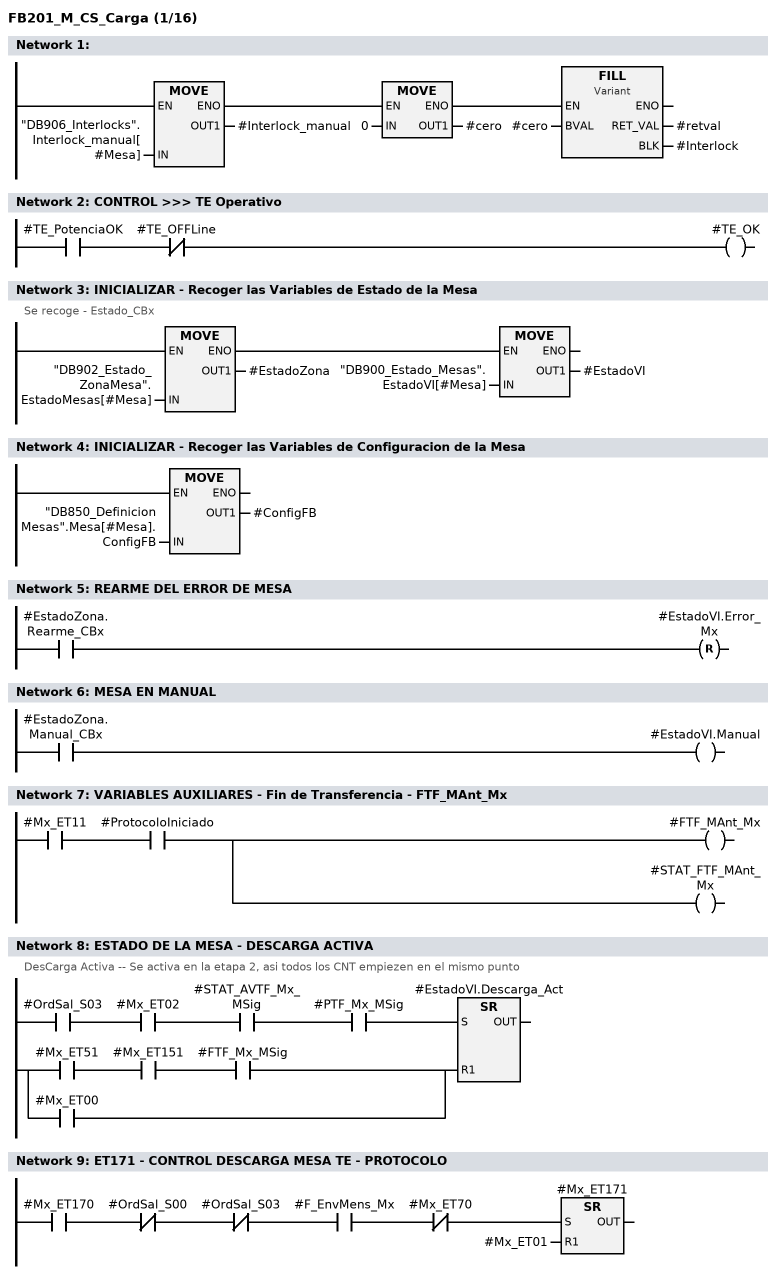
   RUNG wire#powerrail
      Move(in := "DB906_Interlocks".Interlock_manual[#Mesa], out1 => #Interlock_manual)
      Move(in := 0, out1 => #cero)
      { S7_Templates := "ptr_type := Variant" } FILL(BVAL := #cero, RET_VAL => #retval, BLK => #Interlock)
   END_RUNG
   // the same network as SCL:
   #Interlock_manual := "DB906_Interlocks".Interlock_manual[#Mesa];
   #cero := 0;
   #retval := FILL(BVAL := #cero, BLK => #Interlock);
END_REGION

REGION Network 2: CONTROL >>> TE Operativo
   RUNG wire#powerrail
      Contact( #TE_PotenciaOK )
      I_Contact( #TE_OFFLine )
      Coil( #TE_OK )
   END_RUNG
   // the same network as SCL:
   #TE_OK := #TE_PotenciaOK AND NOT #TE_OFFLine;
END_REGION

REGION Network 3: INICIALIZAR - Recoger las Variables de Estado de la Mesa
   // Se recoge - Estado_CBx
   RUNG wire#powerrail
      Move(in := "DB902_Estado_ZonaMesa".EstadoMesas[#Mesa], out1 => #EstadoZona)
      Move(in := "DB900_Estado_Mesas".EstadoVI[#Mesa], out1 => #EstadoVI)
   END_RUNG
   // the same network as SCL:
   #EstadoZona := "DB902_Estado_ZonaMesa".EstadoMesas[#Mesa];
   #EstadoVI := "DB900_Estado_Mesas".EstadoVI[#Mesa];
END_REGION

REGION Network 4: INICIALIZAR - Recoger las Variables de Configuracion de la Mesa
   RUNG wire#powerrail
      Move(in := "DB850_DefinicionMesas".Mesa[#Mesa].ConfigFB, out1 => #ConfigFB)
   END_RUNG
   // the same network as SCL:
   #ConfigFB := "DB850_DefinicionMesas".Mesa[#Mesa].ConfigFB;
END_REGION

REGION Network 5: REARME DEL ERROR DE MESA
   RUNG wire#powerrail
      Contact( #EstadoZona.Rearme_CBx )
      R_Coil( #EstadoVI.Error_Mx )
   END_RUNG
   // the same network as SCL:
   IF #EstadoZona.Rearme_CBx THEN #EstadoVI.Error_Mx := FALSE; END_IF;
END_REGION

REGION Network 6: MESA EN MANUAL
   RUNG wire#powerrail
      Contact( #EstadoZona.Manual_CBx )
      Coil( #EstadoVI.Manual )
   END_RUNG
   // the same network as SCL:
   #EstadoVI.Manual := #EstadoZona.Manual_CBx;
END_REGION

REGION Network 7: VARIABLES AUXILIARES - Fin de Transferencia - FTF_MAnt_Mx
   RUNG wire#powerrail
      Contact( #Mx_ET11 )
      Contact( #ProtocoloIniciado )
      wire#w1
      Coil( #FTF_MAnt_Mx )
   END_RUNG
   RUNG wire#w1
      Coil( #STAT_FTF_MAnt_Mx )
   END_RUNG
   // the same network as SCL:
   #FTF_MAnt_Mx := #Mx_ET11 AND #ProtocoloIniciado;
   #STAT_FTF_MAnt_Mx := #FTF_MAnt_Mx;
END_REGION

REGION Network 8: ESTADO DE LA MESA - DESCARGA ACTIVA
   // DesCarga Activa -- Se activa en la etapa 2, asi todos los CNT empiezen en el mismo punto
   RUNG wire#powerrail
      Contact( #OrdSal_S03 )
      Contact( #Mx_ET02 )
      Contact( #STAT_AVTF_Mx_MSig )
      Contact( #PTF_Mx_MSig )
      S_SR(operand := #EstadoVI.Descarga_Act, r1 := wire#w1)
   END_RUNG
   RUNG wire#powerrail
      Contact( #Mx_ET51 )
      Contact( #Mx_ET151 )
      Contact( #FTF_Mx_MSig )
   END_RUNG wire#w1
   RUNG wire#powerrail
      Contact( #Mx_ET00 )
   END_RUNG wire#w1
   // the same network as SCL:
   IF #OrdSal_S03 AND #Mx_ET02 AND #STAT_AVTF_Mx_MSig AND #PTF_Mx_MSig THEN
       #EstadoVI.Descarga_Act := TRUE;   // SR flip-flop
   END_IF;
   IF (#Mx_ET51 AND #Mx_ET151 AND #FTF_Mx_MSig) OR #Mx_ET00 THEN #EstadoVI.Descarga_Act := FALSE; END_IF;
END_REGION

REGION Network 9: ET171 - CONTROL DESCARGA MESA TE - PROTOCOLO
   RUNG wire#powerrail
      Contact( #Mx_ET170 )
      I_Contact( #OrdSal_S00 )
      I_Contact( #OrdSal_S03 )
      Contact( #F_EnvMens_Mx )
      I_Contact( #Mx_ET70 )
      S_SR(operand := #Mx_ET171, r1 := #Mx_ET01)
   END_RUNG
   // the same network as SCL:
   IF #Mx_ET170 AND NOT #OrdSal_S00 AND NOT #OrdSal_S03 AND #F_EnvMens_Mx AND NOT #Mx_ET70 THEN
       #Mx_ET171 := TRUE;   // SR flip-flop
   END_IF;
   IF #Mx_ET01 THEN #Mx_ET171 := FALSE; END_IF;
END_REGION

REGION Network 10: ET170
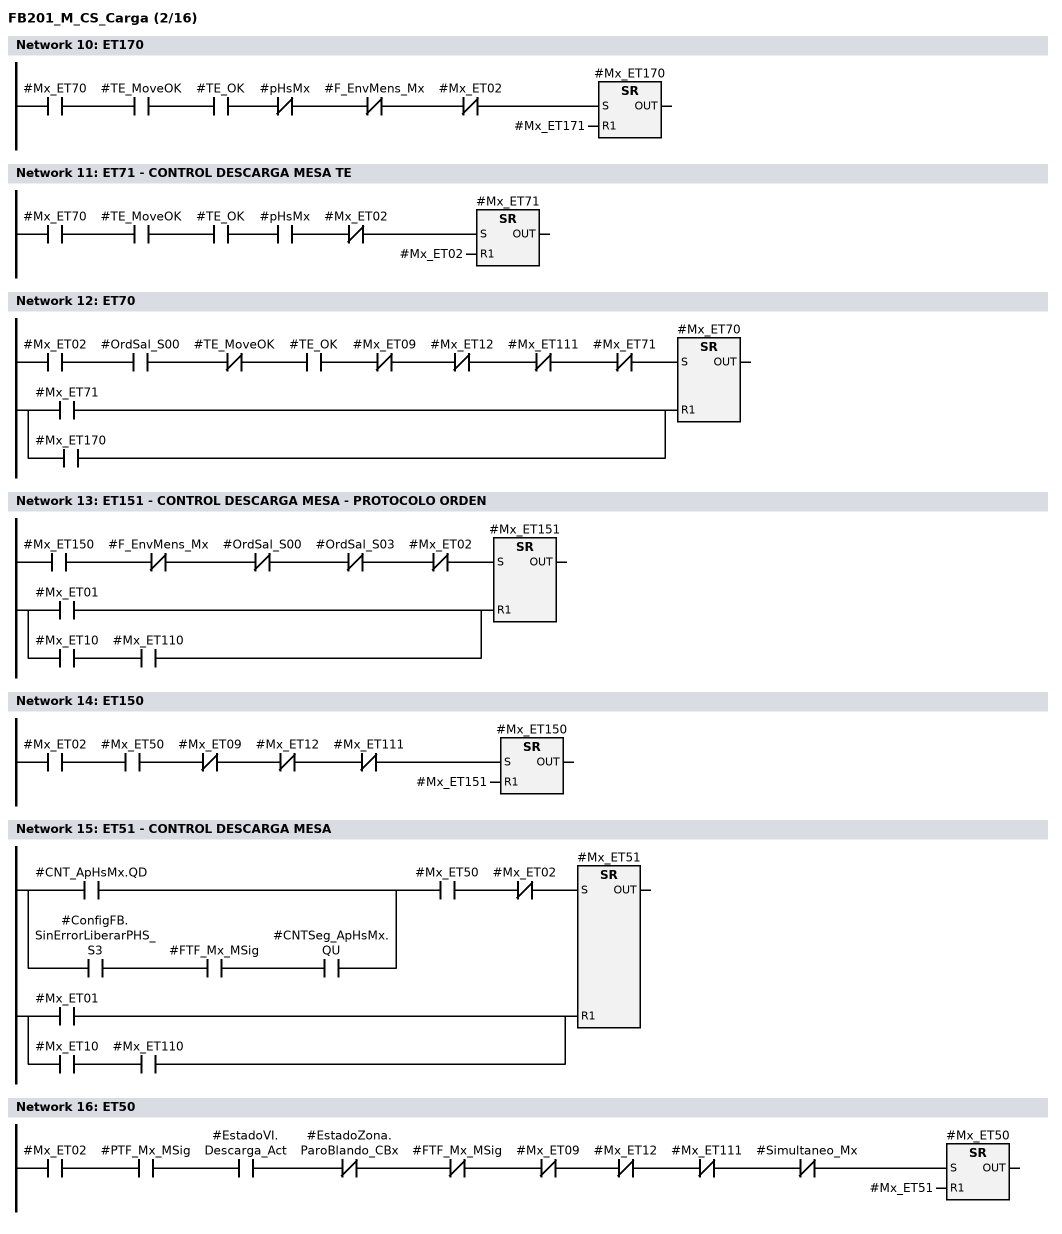
   RUNG wire#powerrail
      Contact( #Mx_ET70 )
      Contact( #TE_MoveOK )
      Contact( #TE_OK )
      I_Contact( #pHsMx )
      I_Contact( #F_EnvMens_Mx )
      I_Contact( #Mx_ET02 )
      S_SR(operand := #Mx_ET170, r1 := #Mx_ET171)
   END_RUNG
   // the same network as SCL:
   IF #Mx_ET70 AND #TE_MoveOK AND #TE_OK AND NOT #pHsMx AND NOT #F_EnvMens_Mx AND NOT #Mx_ET02 THEN
       #Mx_ET170 := TRUE;   // SR flip-flop
   END_IF;
   IF #Mx_ET171 THEN #Mx_ET170 := FALSE; END_IF;
END_REGION

REGION Network 11: ET71 - CONTROL DESCARGA MESA TE
   RUNG wire#powerrail
      Contact( #Mx_ET70 )
      Contact( #TE_MoveOK )
      Contact( #TE_OK )
      Contact( #pHsMx )
      I_Contact( #Mx_ET02 )
      S_SR(operand := #Mx_ET71, r1 := #Mx_ET02)
   END_RUNG
   // the same network as SCL:
   IF #Mx_ET70 AND #TE_MoveOK AND #TE_OK AND #pHsMx AND NOT #Mx_ET02 THEN
       #Mx_ET71 := TRUE;   // SR flip-flop
   END_IF;
   IF #Mx_ET02 THEN #Mx_ET71 := FALSE; END_IF;
END_REGION

REGION Network 12: ET70
   RUNG wire#powerrail
      Contact( #Mx_ET02 )
      Contact( #OrdSal_S00 )
      I_Contact( #TE_MoveOK )
      Contact( #TE_OK )
      I_Contact( #Mx_ET09 )
      I_Contact( #Mx_ET12 )
      I_Contact( #Mx_ET111 )
      I_Contact( #Mx_ET71 )
      S_SR(operand := #Mx_ET70, r1 := wire#w1)
   END_RUNG
   RUNG wire#powerrail
      Contact( #Mx_ET71 )
   END_RUNG wire#w1
   RUNG wire#powerrail
      Contact( #Mx_ET170 )
   END_RUNG wire#w1
   // the same network as SCL:
   IF #Mx_ET02 AND #OrdSal_S00 AND NOT #TE_MoveOK AND #TE_OK AND NOT #Mx_ET09 AND NOT #Mx_ET12 AND NOT #Mx_ET111 AND NOT #Mx_ET71 THEN
       #Mx_ET70 := TRUE;   // SR flip-flop
   END_IF;
   IF #Mx_ET71 OR #Mx_ET170 THEN #Mx_ET70 := FALSE; END_IF;
END_REGION

REGION Network 13: ET151 - CONTROL DESCARGA MESA - PROTOCOLO ORDEN
   RUNG wire#powerrail
      Contact( #Mx_ET150 )
      I_Contact( #F_EnvMens_Mx )
      I_Contact( #OrdSal_S00 )
      I_Contact( #OrdSal_S03 )
      I_Contact( #Mx_ET02 )
      S_SR(operand := #Mx_ET151, r1 := wire#w1)
   END_RUNG
   RUNG wire#powerrail
      Contact( #Mx_ET01 )
   END_RUNG wire#w1
   RUNG wire#powerrail
      Contact( #Mx_ET10 )
      Contact( #Mx_ET110 )
   END_RUNG wire#w1
   // the same network as SCL:
   IF #Mx_ET150 AND NOT #F_EnvMens_Mx AND NOT #OrdSal_S00 AND NOT #OrdSal_S03 AND NOT #Mx_ET02 THEN
       #Mx_ET151 := TRUE;   // SR flip-flop
   END_IF;
   IF #Mx_ET01 OR (#Mx_ET10 AND #Mx_ET110) THEN #Mx_ET151 := FALSE; END_IF;
END_REGION

REGION Network 14: ET150
   RUNG wire#powerrail
      Contact( #Mx_ET02 )
      Contact( #Mx_ET50 )
      I_Contact( #Mx_ET09 )
      I_Contact( #Mx_ET12 )
      I_Contact( #Mx_ET111 )
      S_SR(operand := #Mx_ET150, r1 := #Mx_ET151)
   END_RUNG
   // the same network as SCL:
   IF #Mx_ET02 AND #Mx_ET50 AND NOT #Mx_ET09 AND NOT #Mx_ET12 AND NOT #Mx_ET111 THEN
       #Mx_ET150 := TRUE;   // SR flip-flop
   END_IF;
   IF #Mx_ET151 THEN #Mx_ET150 := FALSE; END_IF;
END_REGION

REGION Network 15: ET51 - CONTROL DESCARGA MESA
   RUNG wire#powerrail
      Contact( #CNT_ApHsMx.QD )
      wire#w1
      Contact( #Mx_ET50 )
      I_Contact( #Mx_ET02 )
      S_SR(operand := #Mx_ET51, r1 := wire#w2)
   END_RUNG
   RUNG wire#powerrail
      Contact( #ConfigFB.SinErrorLiberarPHS_S3 )
      Contact( #FTF_Mx_MSig )
      Contact( #CNTSeg_ApHsMx.QU )
   END_RUNG wire#w1
   RUNG wire#powerrail
      Contact( #Mx_ET01 )
   END_RUNG wire#w2
   RUNG wire#powerrail
      Contact( #Mx_ET10 )
      Contact( #Mx_ET110 )
   END_RUNG wire#w2
   // the same network as SCL:
   IF (#CNT_ApHsMx.QD OR (#ConfigFB.SinErrorLiberarPHS_S3 AND #FTF_Mx_MSig AND #CNTSeg_ApHsMx.QU)) AND #Mx_ET50 AND NOT #Mx_ET02 THEN
       #Mx_ET51 := TRUE;   // SR flip-flop
   END_IF;
   IF #Mx_ET01 OR (#Mx_ET10 AND #Mx_ET110) THEN #Mx_ET51 := FALSE; END_IF;
END_REGION

REGION Network 16: ET50
   RUNG wire#powerrail
      Contact( #Mx_ET02 )
      Contact( #PTF_Mx_MSig )
      Contact( #EstadoVI.Descarga_Act )
      I_Contact( #EstadoZona.ParoBlando_CBx )
      I_Contact( #FTF_Mx_MSig )
      I_Contact( #Mx_ET09 )
      I_Contact( #Mx_ET12 )
      I_Contact( #Mx_ET111 )
      I_Contact( #Simultaneo_Mx )
      S_SR(operand := #Mx_ET50, r1 := #Mx_ET51)
   END_RUNG
   // the same network as SCL:
   IF #Mx_ET02 AND #PTF_Mx_MSig AND #EstadoVI.Descarga_Act AND NOT #EstadoZona.ParoBlando_CBx AND NOT #FTF_Mx_MSig AND NOT #Mx_ET09 AND NOT #Mx_ET12 AND NOT #Mx_ET111 AND NOT #Simultaneo_Mx THEN
       #Mx_ET50 := TRUE;   // SR flip-flop
   END_IF;
   IF #Mx_ET51 THEN #Mx_ET50 := FALSE; END_IF;
END_REGION

REGION Network 17: ET02 - ESTADO REPOSO CARGADA
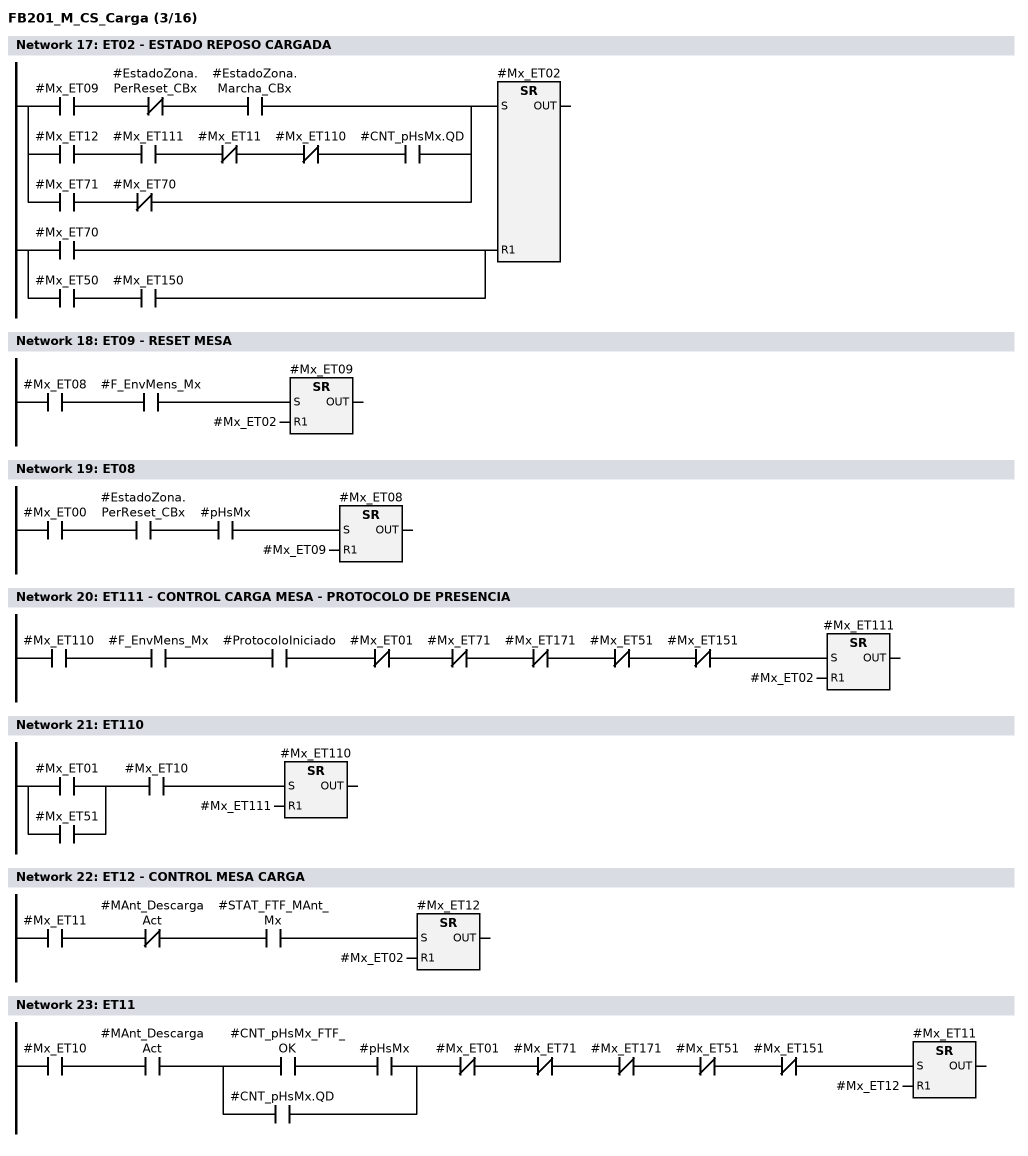
   RUNG wire#powerrail
      Contact( #Mx_ET09 )
      I_Contact( #EstadoZona.PerReset_CBx )
      Contact( #EstadoZona.Marcha_CBx )
      wire#w1
      S_SR(operand := #Mx_ET02, r1 := wire#w2)
   END_RUNG
   RUNG wire#powerrail
      Contact( #Mx_ET12 )
      Contact( #Mx_ET111 )
      I_Contact( #Mx_ET11 )
      I_Contact( #Mx_ET110 )
      Contact( #CNT_pHsMx.QD )
   END_RUNG wire#w1
   RUNG wire#powerrail
      Contact( #Mx_ET71 )
      I_Contact( #Mx_ET70 )
   END_RUNG wire#w1
   RUNG wire#powerrail
      Contact( #Mx_ET70 )
   END_RUNG wire#w2
   RUNG wire#powerrail
      Contact( #Mx_ET50 )
      Contact( #Mx_ET150 )
   END_RUNG wire#w2
   // the same network as SCL:
   IF (#Mx_ET09 AND NOT #EstadoZona.PerReset_CBx AND #EstadoZona.Marcha_CBx) OR (#Mx_ET12 AND #Mx_ET111 AND NOT #Mx_ET11 AND NOT #Mx_ET110 AND #CNT_pHsMx.QD) OR (#Mx_ET71 AND NOT #Mx_ET70) THEN
       #Mx_ET02 := TRUE;   // SR flip-flop
   END_IF;
   IF #Mx_ET70 OR (#Mx_ET50 AND #Mx_ET150) THEN #Mx_ET02 := FALSE; END_IF;
END_REGION

REGION Network 18: ET09 - RESET MESA
   RUNG wire#powerrail
      Contact( #Mx_ET08 )
      Contact( #F_EnvMens_Mx )
      S_SR(operand := #Mx_ET09, r1 := #Mx_ET02)
   END_RUNG
   // the same network as SCL:
   IF #Mx_ET08 AND #F_EnvMens_Mx THEN
       #Mx_ET09 := TRUE;   // SR flip-flop
   END_IF;
   IF #Mx_ET02 THEN #Mx_ET09 := FALSE; END_IF;
END_REGION

REGION Network 19: ET08
   RUNG wire#powerrail
      Contact( #Mx_ET00 )
      Contact( #EstadoZona.PerReset_CBx )
      Contact( #pHsMx )
      S_SR(operand := #Mx_ET08, r1 := #Mx_ET09)
   END_RUNG
   // the same network as SCL:
   IF #Mx_ET00 AND #EstadoZona.PerReset_CBx AND #pHsMx THEN
       #Mx_ET08 := TRUE;   // SR flip-flop
   END_IF;
   IF #Mx_ET09 THEN #Mx_ET08 := FALSE; END_IF;
END_REGION

REGION Network 20: ET111 - CONTROL CARGA MESA - PROTOCOLO DE PRESENCIA
   RUNG wire#powerrail
      Contact( #Mx_ET110 )
      Contact( #F_EnvMens_Mx )
      Contact( #ProtocoloIniciado )
      I_Contact( #Mx_ET01 )
      I_Contact( #Mx_ET71 )
      I_Contact( #Mx_ET171 )
      I_Contact( #Mx_ET51 )
      I_Contact( #Mx_ET151 )
      S_SR(operand := #Mx_ET111, r1 := #Mx_ET02)
   END_RUNG
   // the same network as SCL:
   IF #Mx_ET110 AND #F_EnvMens_Mx AND #ProtocoloIniciado AND NOT #Mx_ET01 AND NOT #Mx_ET71 AND NOT #Mx_ET171 AND NOT #Mx_ET51 AND NOT #Mx_ET151 THEN
       #Mx_ET111 := TRUE;   // SR flip-flop
   END_IF;
   IF #Mx_ET02 THEN #Mx_ET111 := FALSE; END_IF;
END_REGION

REGION Network 21: ET110
   RUNG wire#powerrail
      Contact( #Mx_ET01 )
      wire#w1
      Contact( #Mx_ET10 )
      S_SR(operand := #Mx_ET110, r1 := #Mx_ET111)
   END_RUNG
   RUNG wire#powerrail
      Contact( #Mx_ET51 )
   END_RUNG wire#w1
   // the same network as SCL:
   IF (#Mx_ET01 OR #Mx_ET51) AND #Mx_ET10 THEN
       #Mx_ET110 := TRUE;   // SR flip-flop
   END_IF;
   IF #Mx_ET111 THEN #Mx_ET110 := FALSE; END_IF;
END_REGION

REGION Network 22: ET12 - CONTROL MESA CARGA
   RUNG wire#powerrail
      Contact( #Mx_ET11 )
      I_Contact( #MAnt_DescargaAct )
      Contact( #STAT_FTF_MAnt_Mx )
      S_SR(operand := #Mx_ET12, r1 := #Mx_ET02)
   END_RUNG
   // the same network as SCL:
   IF #Mx_ET11 AND NOT #MAnt_DescargaAct AND #STAT_FTF_MAnt_Mx THEN
       #Mx_ET12 := TRUE;   // SR flip-flop
   END_IF;
   IF #Mx_ET02 THEN #Mx_ET12 := FALSE; END_IF;
END_REGION

REGION Network 23: ET11
   RUNG wire#powerrail
      Contact( #Mx_ET10 )
      Contact( #MAnt_DescargaAct )
      wire#w1
      Contact( #CNT_pHsMx_FTF_OK )
      Contact( #pHsMx )
      wire#w2
      I_Contact( #Mx_ET01 )
      I_Contact( #Mx_ET71 )
      I_Contact( #Mx_ET171 )
      I_Contact( #Mx_ET51 )
      I_Contact( #Mx_ET151 )
      S_SR(operand := #Mx_ET11, r1 := #Mx_ET12)
   END_RUNG
   RUNG wire#w1
      Contact( #CNT_pHsMx.QD )
   END_RUNG wire#w2
   // the same network as SCL:
   IF #Mx_ET10 AND #MAnt_DescargaAct AND ((#CNT_pHsMx_FTF_OK AND #pHsMx) OR #CNT_pHsMx.QD) AND NOT #Mx_ET01 AND NOT #Mx_ET71 AND NOT #Mx_ET171 AND NOT #Mx_ET51 AND NOT #Mx_ET151 THEN
       #Mx_ET11 := TRUE;   // SR flip-flop
   END_IF;
   IF #Mx_ET12 THEN #Mx_ET11 := FALSE; END_IF;
END_REGION

REGION Network 24: ET10
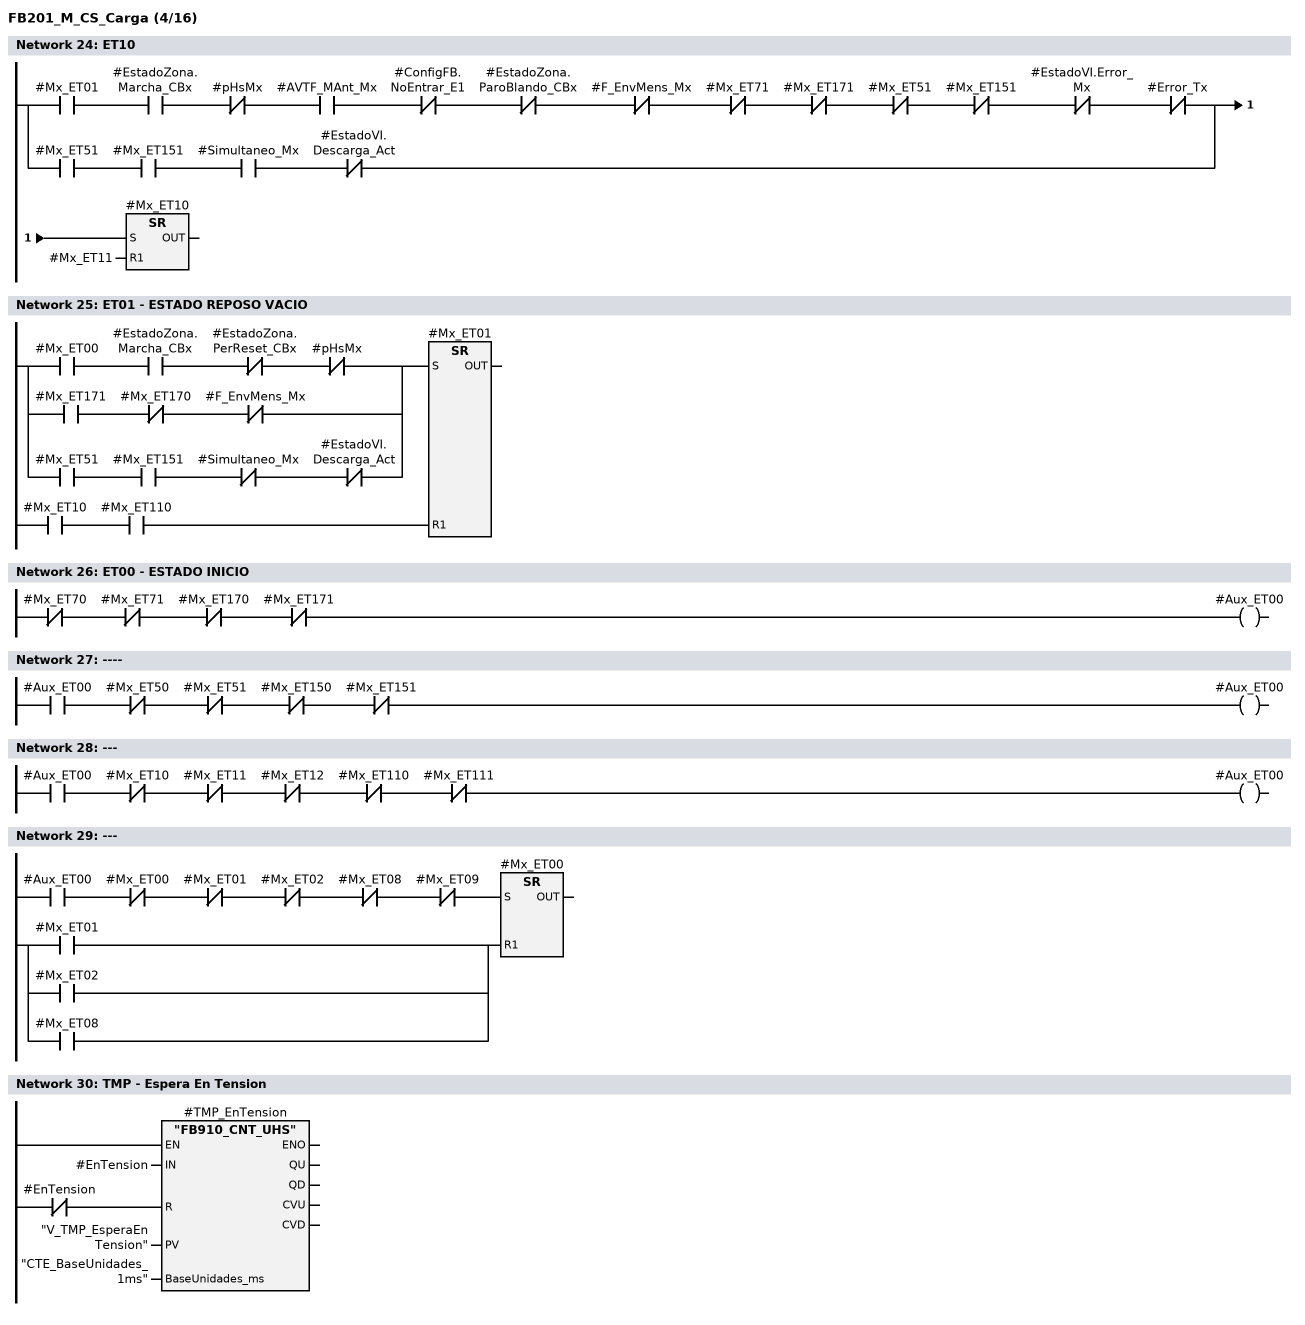
   RUNG wire#powerrail
      Contact( #Mx_ET01 )
      Contact( #EstadoZona.Marcha_CBx )
      I_Contact( #pHsMx )
      Contact( #AVTF_MAnt_Mx )
      I_Contact( #ConfigFB.NoEntrar_E1 )
      I_Contact( #EstadoZona.ParoBlando_CBx )
      I_Contact( #F_EnvMens_Mx )
      I_Contact( #Mx_ET71 )
      I_Contact( #Mx_ET171 )
      I_Contact( #Mx_ET51 )
      I_Contact( #Mx_ET151 )
      I_Contact( #EstadoVI.Error_Mx )
      I_Contact( #Error_Tx )
      wire#w1
      S_SR(operand := #Mx_ET10, r1 := #Mx_ET11)
   END_RUNG
   RUNG wire#powerrail
      Contact( #Mx_ET51 )
      Contact( #Mx_ET151 )
      Contact( #Simultaneo_Mx )
      I_Contact( #EstadoVI.Descarga_Act )
   END_RUNG wire#w1
   // the same network as SCL:
   IF (#Mx_ET01 AND #EstadoZona.Marcha_CBx AND NOT #pHsMx AND #AVTF_MAnt_Mx AND NOT #ConfigFB.NoEntrar_E1 AND NOT #EstadoZona.ParoBlando_CBx AND NOT #F_EnvMens_Mx AND NOT #Mx_ET71 AND NOT #Mx_ET171 AND NOT #Mx_ET51 AND NOT #Mx_ET151 AND NOT #EstadoVI.Error_Mx AND NOT #Error_Tx) OR (#Mx_ET51 AND #Mx_ET151 AND #Simultaneo_Mx AND NOT #EstadoVI.Descarga_Act) THEN
       #Mx_ET10 := TRUE;   // SR flip-flop
   END_IF;
   IF #Mx_ET11 THEN #Mx_ET10 := FALSE; END_IF;
END_REGION

REGION Network 25: ET01 - ESTADO REPOSO VACIO
   RUNG wire#powerrail
      Contact( #Mx_ET00 )
      Contact( #EstadoZona.Marcha_CBx )
      I_Contact( #EstadoZona.PerReset_CBx )
      I_Contact( #pHsMx )
      wire#w1
      S_SR(operand := #Mx_ET01, r1 := wire#w2)
   END_RUNG
   RUNG wire#powerrail
      Contact( #Mx_ET171 )
      I_Contact( #Mx_ET170 )
      I_Contact( #F_EnvMens_Mx )
   END_RUNG wire#w1
   RUNG wire#powerrail
      Contact( #Mx_ET51 )
      Contact( #Mx_ET151 )
      I_Contact( #Simultaneo_Mx )
      I_Contact( #EstadoVI.Descarga_Act )
   END_RUNG wire#w1
   RUNG wire#powerrail
      Contact( #Mx_ET10 )
      Contact( #Mx_ET110 )
   END_RUNG wire#w2
   // the same network as SCL:
   IF (#Mx_ET00 AND #EstadoZona.Marcha_CBx AND NOT #EstadoZona.PerReset_CBx AND NOT #pHsMx) OR (#Mx_ET171 AND NOT #Mx_ET170 AND NOT #F_EnvMens_Mx) OR (#Mx_ET51 AND #Mx_ET151 AND NOT #Simultaneo_Mx AND NOT #EstadoVI.Descarga_Act) THEN
       #Mx_ET01 := TRUE;   // SR flip-flop
   END_IF;
   IF #Mx_ET10 AND #Mx_ET110 THEN #Mx_ET01 := FALSE; END_IF;
END_REGION

REGION Network 26: ET00 - ESTADO INICIO
   RUNG wire#powerrail
      I_Contact( #Mx_ET70 )
      I_Contact( #Mx_ET71 )
      I_Contact( #Mx_ET170 )
      I_Contact( #Mx_ET171 )
      Coil( #Aux_ET00 )
   END_RUNG
   // the same network as SCL:
   #Aux_ET00 := NOT #Mx_ET70 AND NOT #Mx_ET71 AND NOT #Mx_ET170 AND NOT #Mx_ET171;
END_REGION

REGION Network 27: ----
   RUNG wire#powerrail
      Contact( #Aux_ET00 )
      I_Contact( #Mx_ET50 )
      I_Contact( #Mx_ET51 )
      I_Contact( #Mx_ET150 )
      I_Contact( #Mx_ET151 )
      Coil( #Aux_ET00 )
   END_RUNG
   // the same network as SCL:
   #Aux_ET00 := #Aux_ET00 AND NOT #Mx_ET50 AND NOT #Mx_ET51 AND NOT #Mx_ET150 AND NOT #Mx_ET151;
END_REGION

REGION Network 28: ---
   RUNG wire#powerrail
      Contact( #Aux_ET00 )
      I_Contact( #Mx_ET10 )
      I_Contact( #Mx_ET11 )
      I_Contact( #Mx_ET12 )
      I_Contact( #Mx_ET110 )
      I_Contact( #Mx_ET111 )
      Coil( #Aux_ET00 )
   END_RUNG
   // the same network as SCL:
   #Aux_ET00 := #Aux_ET00 AND NOT #Mx_ET10 AND NOT #Mx_ET11 AND NOT #Mx_ET12 AND NOT #Mx_ET110 AND NOT #Mx_ET111;
END_REGION

REGION Network 29: ---
   RUNG wire#powerrail
      Contact( #Aux_ET00 )
      I_Contact( #Mx_ET00 )
      I_Contact( #Mx_ET01 )
      I_Contact( #Mx_ET02 )
      I_Contact( #Mx_ET08 )
      I_Contact( #Mx_ET09 )
      S_SR(operand := #Mx_ET00, r1 := wire#w1)
   END_RUNG
   RUNG wire#powerrail
      Contact( #Mx_ET01 )
   END_RUNG wire#w1
   RUNG wire#powerrail
      Contact( #Mx_ET02 )
   END_RUNG wire#w1
   RUNG wire#powerrail
      Contact( #Mx_ET08 )
   END_RUNG wire#w1
   // the same network as SCL:
   IF #Aux_ET00 AND NOT #Mx_ET00 AND NOT #Mx_ET01 AND NOT #Mx_ET02 AND NOT #Mx_ET08 AND NOT #Mx_ET09 THEN
       #Mx_ET00 := TRUE;   // SR flip-flop
   END_IF;
   IF #Mx_ET01 OR #Mx_ET02 OR #Mx_ET08 THEN #Mx_ET00 := FALSE; END_IF;
END_REGION

REGION Network 30: TMP - Espera En Tension
   RUNG wire#powerrail
      #TMP_EnTension(R := wire#w1, IN := #EnTension, PV := "V_TMP_EsperaEnTension", BaseUnidades_ms := "CTE_BaseUnidades_1ms", QU =>, QD =>, CVU =>, CVD =>)
   END_RUNG
   RUNG wire#powerrail
      I_Contact( #EnTension )
   END_RUNG wire#w1
   // the same network as SCL:
   #TMP_EnTension(IN := #EnTension,   // "FB910_CNT_UHS"
                  R := NOT #EnTension,
                  PV := "V_TMP_EsperaEnTension",
                  BaseUnidades_ms := "CTE_BaseUnidades_1ms");
END_REGION

REGION Network 31: ERROR - Termico
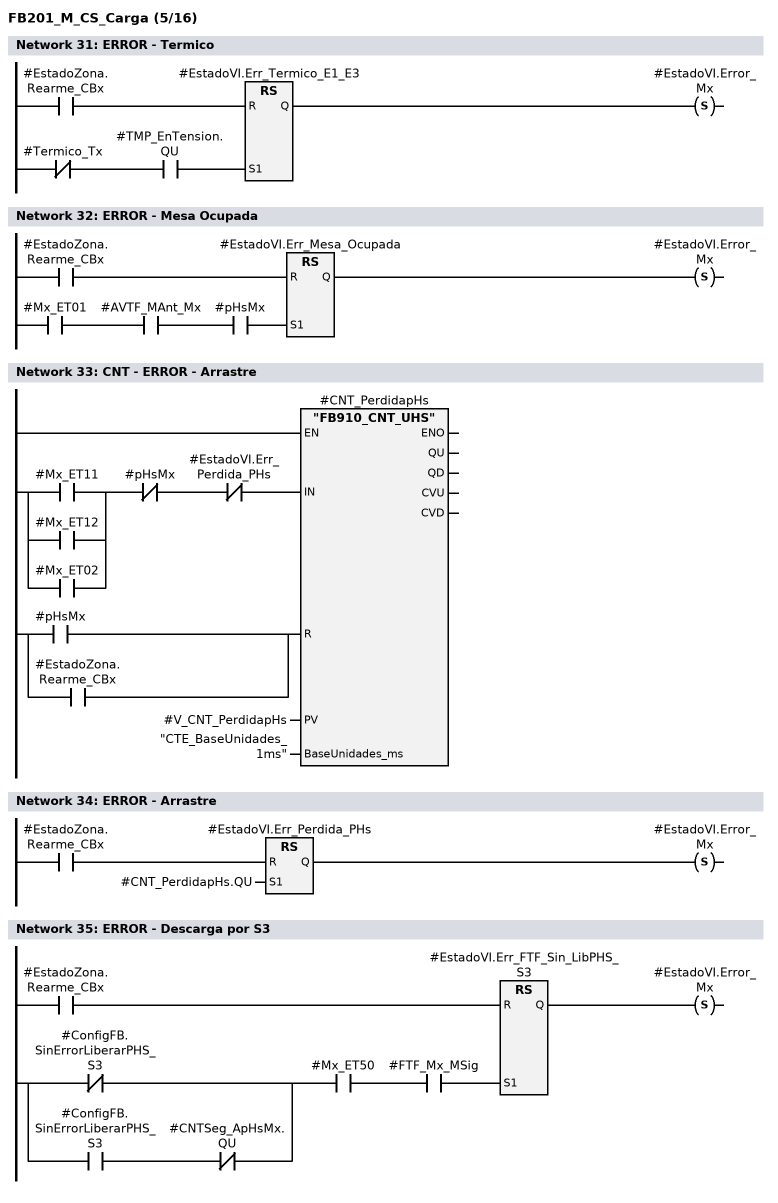
   RUNG wire#powerrail
      Contact( #EstadoZona.Rearme_CBx )
      S_RS(operand := #EstadoVI.Err_Termico_E1_E3, s1 := wire#w1)
      S_Coil( #EstadoVI.Error_Mx )
   END_RUNG
   RUNG wire#powerrail
      I_Contact( #Termico_Tx )
      Contact( #TMP_EnTension.QU )
   END_RUNG wire#w1
   // the same network as SCL:
   IF #EstadoZona.Rearme_CBx THEN
       #EstadoVI.Err_Termico_E1_E3 := FALSE;   // RS flip-flop
   END_IF;
   IF NOT #Termico_Tx AND #TMP_EnTension.QU THEN #EstadoVI.Err_Termico_E1_E3 := TRUE; END_IF;
   IF #EstadoVI.Err_Termico_E1_E3 THEN #EstadoVI.Error_Mx := TRUE; END_IF;
END_REGION

REGION Network 32: ERROR - Mesa Ocupada
   RUNG wire#powerrail
      Contact( #EstadoZona.Rearme_CBx )
      S_RS(operand := #EstadoVI.Err_Mesa_Ocupada, s1 := wire#w1)
      S_Coil( #EstadoVI.Error_Mx )
   END_RUNG
   RUNG wire#powerrail
      Contact( #Mx_ET01 )
      Contact( #AVTF_MAnt_Mx )
      Contact( #pHsMx )
   END_RUNG wire#w1
   // the same network as SCL:
   IF #EstadoZona.Rearme_CBx THEN
       #EstadoVI.Err_Mesa_Ocupada := FALSE;   // RS flip-flop
   END_IF;
   IF #Mx_ET01 AND #AVTF_MAnt_Mx AND #pHsMx THEN #EstadoVI.Err_Mesa_Ocupada := TRUE; END_IF;
   IF #EstadoVI.Err_Mesa_Ocupada THEN #EstadoVI.Error_Mx := TRUE; END_IF;
END_REGION

REGION Network 33: CNT - ERROR - Arrastre
   RUNG wire#powerrail
      #CNT_PerdidapHs(IN := wire#w2, R := wire#w3, PV := #V_CNT_PerdidapHs, BaseUnidades_ms := "CTE_BaseUnidades_1ms", QU =>, QD =>, CVU =>, CVD =>)
   END_RUNG
   RUNG wire#powerrail
      Contact( #Mx_ET11 )
      wire#w1
      I_Contact( #pHsMx )
      I_Contact( #EstadoVI.Err_Perdida_PHs )
   END_RUNG wire#w2
   RUNG wire#powerrail
      Contact( #Mx_ET12 )
   END_RUNG wire#w1
   RUNG wire#powerrail
      Contact( #Mx_ET02 )
   END_RUNG wire#w1
   RUNG wire#powerrail
      Contact( #pHsMx )
   END_RUNG wire#w3
   RUNG wire#powerrail
      Contact( #EstadoZona.Rearme_CBx )
   END_RUNG wire#w3
   // the same network as SCL:
   #CNT_PerdidapHs(IN := (#Mx_ET11 OR #Mx_ET12 OR #Mx_ET02) AND NOT #pHsMx AND NOT #EstadoVI.Err_Perdida_PHs,   // "FB910_CNT_UHS"
                   R := #pHsMx OR #EstadoZona.Rearme_CBx,
                   PV := #V_CNT_PerdidapHs,
                   BaseUnidades_ms := "CTE_BaseUnidades_1ms");
END_REGION

REGION Network 34: ERROR - Arrastre
   RUNG wire#powerrail
      Contact( #EstadoZona.Rearme_CBx )
      S_RS(operand := #EstadoVI.Err_Perdida_PHs, s1 := #CNT_PerdidapHs.QU)
      S_Coil( #EstadoVI.Error_Mx )
   END_RUNG
   // the same network as SCL:
   IF #EstadoZona.Rearme_CBx THEN
       #EstadoVI.Err_Perdida_PHs := FALSE;   // RS flip-flop
   END_IF;
   IF #CNT_PerdidapHs.QU THEN #EstadoVI.Err_Perdida_PHs := TRUE; END_IF;
   IF #EstadoVI.Err_Perdida_PHs THEN #EstadoVI.Error_Mx := TRUE; END_IF;
END_REGION

REGION Network 35: ERROR - Descarga por S3
   RUNG wire#powerrail
      Contact( #EstadoZona.Rearme_CBx )
      S_RS(operand := #EstadoVI.Err_FTF_Sin_LibPHS_S3, s1 := wire#w2)
      S_Coil( #EstadoVI.Error_Mx )
   END_RUNG
   RUNG wire#powerrail
      I_Contact( #ConfigFB.SinErrorLiberarPHS_S3 )
      wire#w1
      Contact( #Mx_ET50 )
      Contact( #FTF_Mx_MSig )
   END_RUNG wire#w2
   RUNG wire#powerrail
      Contact( #ConfigFB.SinErrorLiberarPHS_S3 )
      I_Contact( #CNTSeg_ApHsMx.QU )
   END_RUNG wire#w1
   // the same network as SCL:
   IF #EstadoZona.Rearme_CBx THEN
       #EstadoVI.Err_FTF_Sin_LibPHS_S3 := FALSE;   // RS flip-flop
   END_IF;
   IF (NOT #ConfigFB.SinErrorLiberarPHS_S3 OR (#ConfigFB.SinErrorLiberarPHS_S3 AND NOT #CNTSeg_ApHsMx.QU)) AND #Mx_ET50 AND #FTF_Mx_MSig THEN
       #EstadoVI.Err_FTF_Sin_LibPHS_S3 := TRUE;
   END_IF;
   IF #EstadoVI.Err_FTF_Sin_LibPHS_S3 THEN #EstadoVI.Error_Mx := TRUE; END_IF;
END_REGION

REGION Network 36: TMP - ERROR - TimeOut Avance
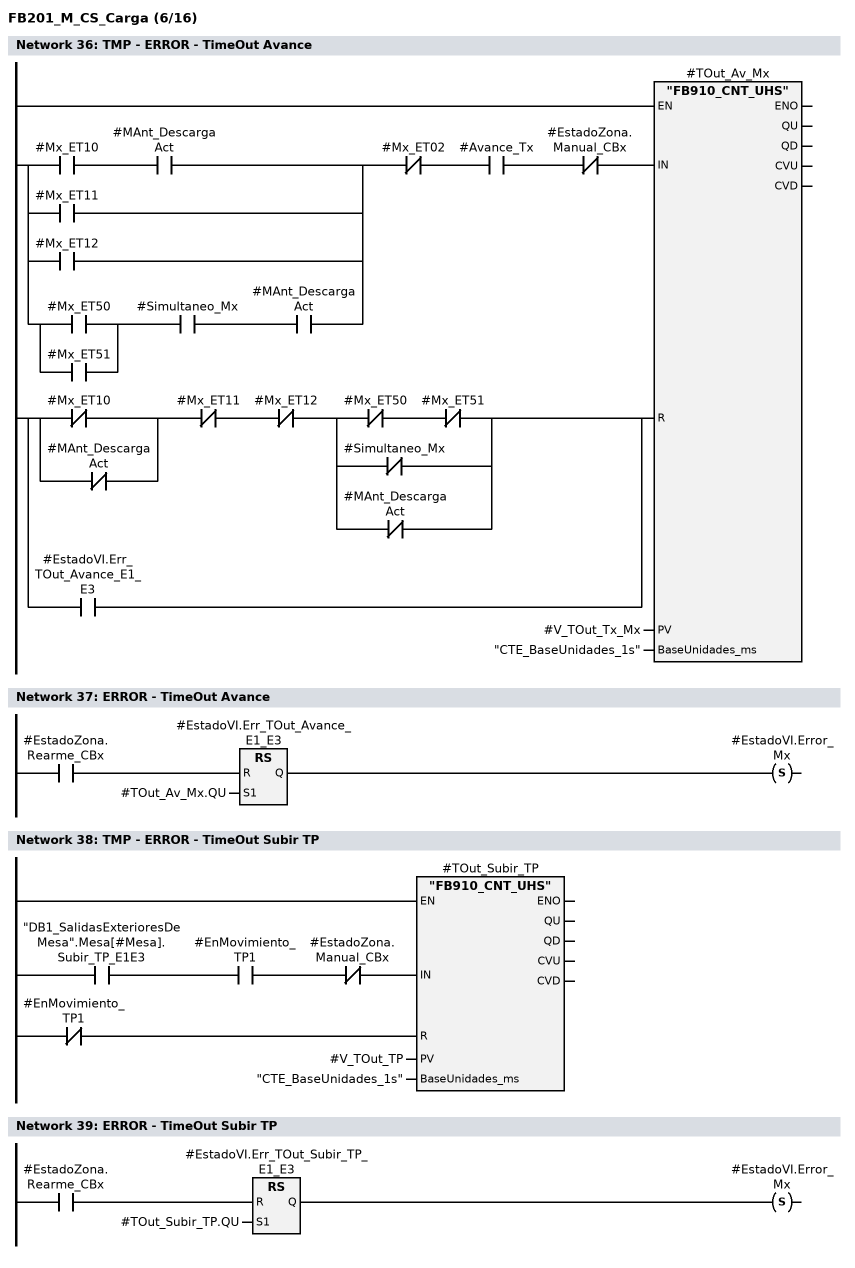
   RUNG wire#powerrail
      #TOut_Av_Mx(IN := wire#w3, R := wire#w6, PV := #V_TOut_Tx_Mx, BaseUnidades_ms := "CTE_BaseUnidades_1s", QU =>, QD =>, CVU =>, CVD =>)
   END_RUNG
   RUNG wire#powerrail
      Contact( #Mx_ET10 )
      Contact( #MAnt_DescargaAct )
      wire#w1
      I_Contact( #Mx_ET02 )
      Contact( #Avance_Tx )
      I_Contact( #EstadoZona.Manual_CBx )
   END_RUNG wire#w3
   RUNG wire#powerrail
      Contact( #Mx_ET11 )
   END_RUNG wire#w1
   RUNG wire#powerrail
      Contact( #Mx_ET12 )
   END_RUNG wire#w1
   RUNG wire#powerrail
      Contact( #Mx_ET50 )
      wire#w2
      Contact( #Simultaneo_Mx )
      Contact( #MAnt_DescargaAct )
   END_RUNG wire#w1
   RUNG wire#powerrail
      Contact( #Mx_ET51 )
   END_RUNG wire#w2
   RUNG wire#powerrail
      I_Contact( #Mx_ET10 )
      wire#w4
      I_Contact( #Mx_ET11 )
      I_Contact( #Mx_ET12 )
      wire#w5
      I_Contact( #Mx_ET50 )
      I_Contact( #Mx_ET51 )
   END_RUNG wire#w6
   RUNG wire#powerrail
      I_Contact( #MAnt_DescargaAct )
   END_RUNG wire#w4
   RUNG wire#w5
      I_Contact( #Simultaneo_Mx )
   END_RUNG wire#w6
   RUNG wire#w5
      I_Contact( #MAnt_DescargaAct )
   END_RUNG wire#w6
   RUNG wire#powerrail
      Contact( #EstadoVI.Err_TOut_Avance_E1_E3 )
   END_RUNG wire#w6
   // the same network as SCL:
   #TOut_Av_Mx(IN := ((#Mx_ET10 AND #MAnt_DescargaAct) OR #Mx_ET11 OR #Mx_ET12 OR ((#Mx_ET50 OR #Mx_ET51) AND #Simultaneo_Mx AND #MAnt_DescargaAct)) AND NOT #Mx_ET02 AND #Avance_Tx AND NOT #EstadoZona.Manual_CBx,   // "FB910_CNT_UHS"
               R := ((NOT #Mx_ET10 OR NOT #MAnt_DescargaAct) AND NOT #Mx_ET11 AND NOT #Mx_ET12 AND ((NOT #Mx_ET50 AND NOT #Mx_ET51) OR NOT #Simultaneo_Mx OR NOT #MAnt_DescargaAct)) OR #EstadoVI.Err_TOut_Avance_E1_E3,
               PV := #V_TOut_Tx_Mx,
               BaseUnidades_ms := "CTE_BaseUnidades_1s");
END_REGION

REGION Network 37: ERROR - TimeOut Avance
   RUNG wire#powerrail
      Contact( #EstadoZona.Rearme_CBx )
      S_RS(operand := #EstadoVI.Err_TOut_Avance_E1_E3, s1 := #TOut_Av_Mx.QU)
      S_Coil( #EstadoVI.Error_Mx )
   END_RUNG
   // the same network as SCL:
   IF #EstadoZona.Rearme_CBx THEN
       #EstadoVI.Err_TOut_Avance_E1_E3 := FALSE;   // RS flip-flop
   END_IF;
   IF #TOut_Av_Mx.QU THEN #EstadoVI.Err_TOut_Avance_E1_E3 := TRUE; END_IF;
   IF #EstadoVI.Err_TOut_Avance_E1_E3 THEN #EstadoVI.Error_Mx := TRUE; END_IF;
END_REGION

REGION Network 38: TMP - ERROR - TimeOut Subir TP
   RUNG wire#powerrail
      #TOut_Subir_TP(IN := wire#w1, R := wire#w2, PV := #V_TOut_TP, BaseUnidades_ms := "CTE_BaseUnidades_1s", QU =>, QD =>, CVU =>, CVD =>)
   END_RUNG
   RUNG wire#powerrail
      Contact( "DB1_SalidasExterioresDeMesa".Mesa[#Mesa].Subir_TP_E1E3 )
      Contact( #EnMovimiento_TP1 )
      I_Contact( #EstadoZona.Manual_CBx )
   END_RUNG wire#w1
   RUNG wire#powerrail
      I_Contact( #EnMovimiento_TP1 )
   END_RUNG wire#w2
   // the same network as SCL:
   #TOut_Subir_TP(IN := "DB1_SalidasExterioresDeMesa".Mesa[#Mesa].Subir_TP_E1E3 AND #EnMovimiento_TP1 AND NOT #EstadoZona.Manual_CBx,   // "FB910_CNT_UHS"
                  R := NOT #EnMovimiento_TP1,
                  PV := #V_TOut_TP,
                  BaseUnidades_ms := "CTE_BaseUnidades_1s");
END_REGION

REGION Network 39: ERROR - TimeOut Subir TP
   RUNG wire#powerrail
      Contact( #EstadoZona.Rearme_CBx )
      S_RS(operand := #EstadoVI.Err_TOut_Subir_TP_E1_E3, s1 := #TOut_Subir_TP.QU)
      S_Coil( #EstadoVI.Error_Mx )
   END_RUNG
   // the same network as SCL:
   IF #EstadoZona.Rearme_CBx THEN
       #EstadoVI.Err_TOut_Subir_TP_E1_E3 := FALSE;   // RS flip-flop
   END_IF;
   IF #TOut_Subir_TP.QU THEN #EstadoVI.Err_TOut_Subir_TP_E1_E3 := TRUE; END_IF;
   IF #EstadoVI.Err_TOut_Subir_TP_E1_E3 THEN #EstadoVI.Error_Mx := TRUE; END_IF;
END_REGION

REGION Network 40: TMP - ERROR - TimeOut Bajar TP
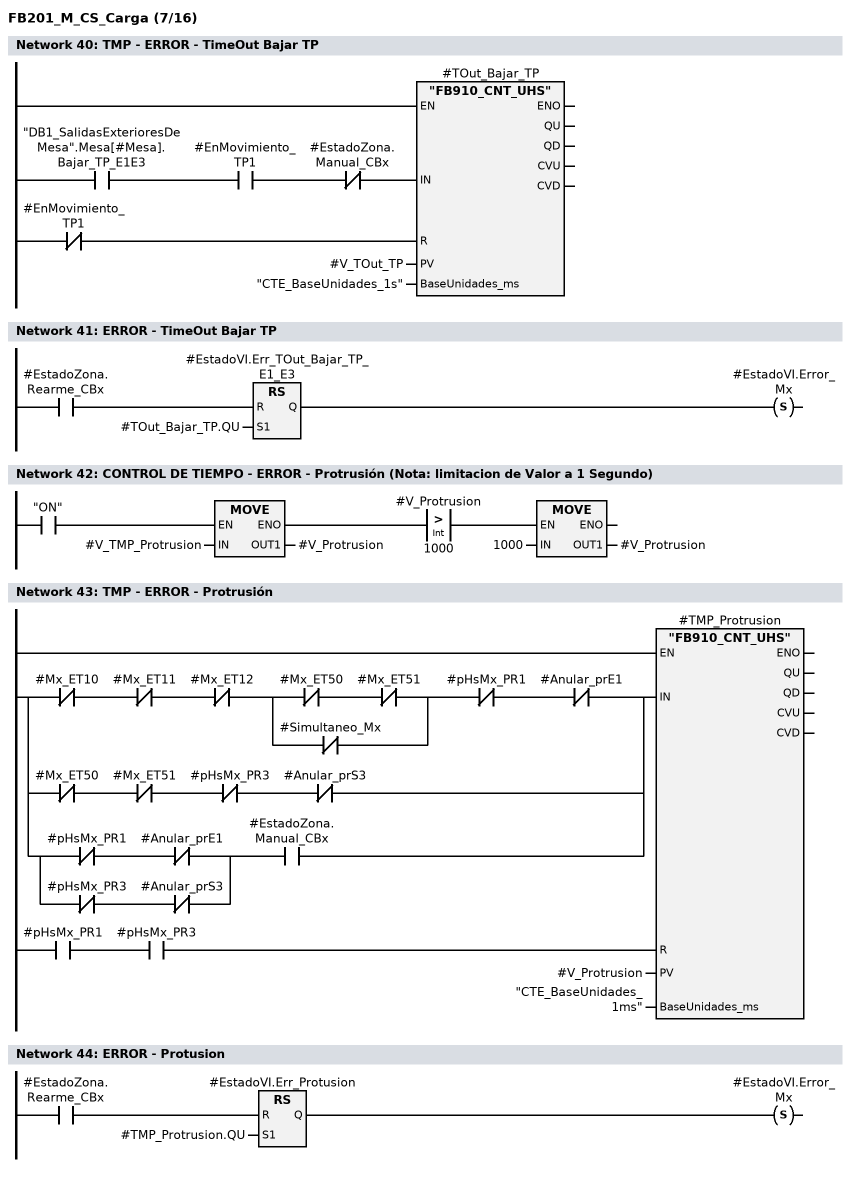
   RUNG wire#powerrail
      #TOut_Bajar_TP(IN := wire#w1, R := wire#w2, PV := #V_TOut_TP, BaseUnidades_ms := "CTE_BaseUnidades_1s", QU =>, QD =>, CVU =>, CVD =>)
   END_RUNG
   RUNG wire#powerrail
      Contact( "DB1_SalidasExterioresDeMesa".Mesa[#Mesa].Bajar_TP_E1E3 )
      Contact( #EnMovimiento_TP1 )
      I_Contact( #EstadoZona.Manual_CBx )
   END_RUNG wire#w1
   RUNG wire#powerrail
      I_Contact( #EnMovimiento_TP1 )
   END_RUNG wire#w2
   // the same network as SCL:
   #TOut_Bajar_TP(IN := "DB1_SalidasExterioresDeMesa".Mesa[#Mesa].Bajar_TP_E1E3 AND #EnMovimiento_TP1 AND NOT #EstadoZona.Manual_CBx,   // "FB910_CNT_UHS"
                  R := NOT #EnMovimiento_TP1,
                  PV := #V_TOut_TP,
                  BaseUnidades_ms := "CTE_BaseUnidades_1s");
END_REGION

REGION Network 41: ERROR - TimeOut Bajar TP
   RUNG wire#powerrail
      Contact( #EstadoZona.Rearme_CBx )
      S_RS(operand := #EstadoVI.Err_TOut_Bajar_TP_E1_E3, s1 := #TOut_Bajar_TP.QU)
      S_Coil( #EstadoVI.Error_Mx )
   END_RUNG
   // the same network as SCL:
   IF #EstadoZona.Rearme_CBx THEN
       #EstadoVI.Err_TOut_Bajar_TP_E1_E3 := FALSE;   // RS flip-flop
   END_IF;
   IF #TOut_Bajar_TP.QU THEN #EstadoVI.Err_TOut_Bajar_TP_E1_E3 := TRUE; END_IF;
   IF #EstadoVI.Err_TOut_Bajar_TP_E1_E3 THEN #EstadoVI.Error_Mx := TRUE; END_IF;
END_REGION

REGION Network 42: CONTROL DE TIEMPO - ERROR - Protrusión (Nota: limitacion de Valor a 1 Segundo)
   RUNG wire#powerrail
      Contact( "ON" )
      Move(in := #V_TMP_Protrusion, out1 => #V_Protrusion)
      { S7_Templates := "SrcType := Int" } GT_Contact(in1 := #V_Protrusion, in2 := 1000)
      Move(in := 1000, out1 => #V_Protrusion)
   END_RUNG
   // the same network as SCL:
   IF "ON" THEN #V_Protrusion := #V_TMP_Protrusion; END_IF;
   IF "ON" AND (#V_Protrusion > 1000) THEN #V_Protrusion := 1000; END_IF;
END_REGION

REGION Network 43: TMP - ERROR - Protrusión
   RUNG wire#powerrail
      #TMP_Protrusion(IN := wire#w4, R := wire#w5, PV := #V_Protrusion, BaseUnidades_ms := "CTE_BaseUnidades_1ms", QU =>, QD =>, CVU =>, CVD =>)
   END_RUNG
   RUNG wire#powerrail
      I_Contact( #Mx_ET10 )
      I_Contact( #Mx_ET11 )
      I_Contact( #Mx_ET12 )
      wire#w1
      I_Contact( #Mx_ET50 )
      I_Contact( #Mx_ET51 )
      wire#w2
      I_Contact( #pHsMx_PR1 )
      I_Contact( #Anular_prE1 )
   END_RUNG wire#w4
   RUNG wire#w1
      I_Contact( #Simultaneo_Mx )
   END_RUNG wire#w2
   RUNG wire#powerrail
      I_Contact( #Mx_ET50 )
      I_Contact( #Mx_ET51 )
      I_Contact( #pHsMx_PR3 )
      I_Contact( #Anular_prS3 )
   END_RUNG wire#w4
   RUNG wire#powerrail
      I_Contact( #pHsMx_PR1 )
      I_Contact( #Anular_prE1 )
      wire#w3
      Contact( #EstadoZona.Manual_CBx )
   END_RUNG wire#w4
   RUNG wire#powerrail
      I_Contact( #pHsMx_PR3 )
      I_Contact( #Anular_prS3 )
   END_RUNG wire#w3
   RUNG wire#powerrail
      Contact( #pHsMx_PR1 )
      Contact( #pHsMx_PR3 )
   END_RUNG wire#w5
   // the same network as SCL:
   #TMP_Protrusion(IN := (NOT #Mx_ET10 AND NOT #Mx_ET11 AND NOT #Mx_ET12 AND ((NOT #Mx_ET50 AND NOT #Mx_ET51) OR NOT #Simultaneo_Mx) AND NOT #pHsMx_PR1 AND NOT #Anular_prE1) OR (NOT #Mx_ET50 AND NOT #Mx_ET51 AND NOT #pHsMx_PR3 AND NOT #Anular_prS3) OR (((NOT #pHsMx_PR1 AND NOT #Anular_prE1) OR (NOT #pHsMx_PR3 AND NOT #Anular_prS3)) AND #EstadoZona.Manual_CBx),   // "FB910_CNT_UHS"
                   R := #pHsMx_PR1 AND #pHsMx_PR3,
                   PV := #V_Protrusion,
                   BaseUnidades_ms := "CTE_BaseUnidades_1ms");
END_REGION

REGION Network 44: ERROR - Protusion
   RUNG wire#powerrail
      Contact( #EstadoZona.Rearme_CBx )
      S_RS(operand := #EstadoVI.Err_Protusion, s1 := #TMP_Protrusion.QU)
      S_Coil( #EstadoVI.Error_Mx )
   END_RUNG
   // the same network as SCL:
   IF #EstadoZona.Rearme_CBx THEN
       #EstadoVI.Err_Protusion := FALSE;   // RS flip-flop
   END_IF;
   IF #TMP_Protrusion.QU THEN #EstadoVI.Err_Protusion := TRUE; END_IF;
   IF #EstadoVI.Err_Protusion THEN #EstadoVI.Error_Mx := TRUE; END_IF;
END_REGION

REGION Network 45: CONTADOR DE SEGURIDAD DE PRESENCIA - CNTSeg_pHsMx
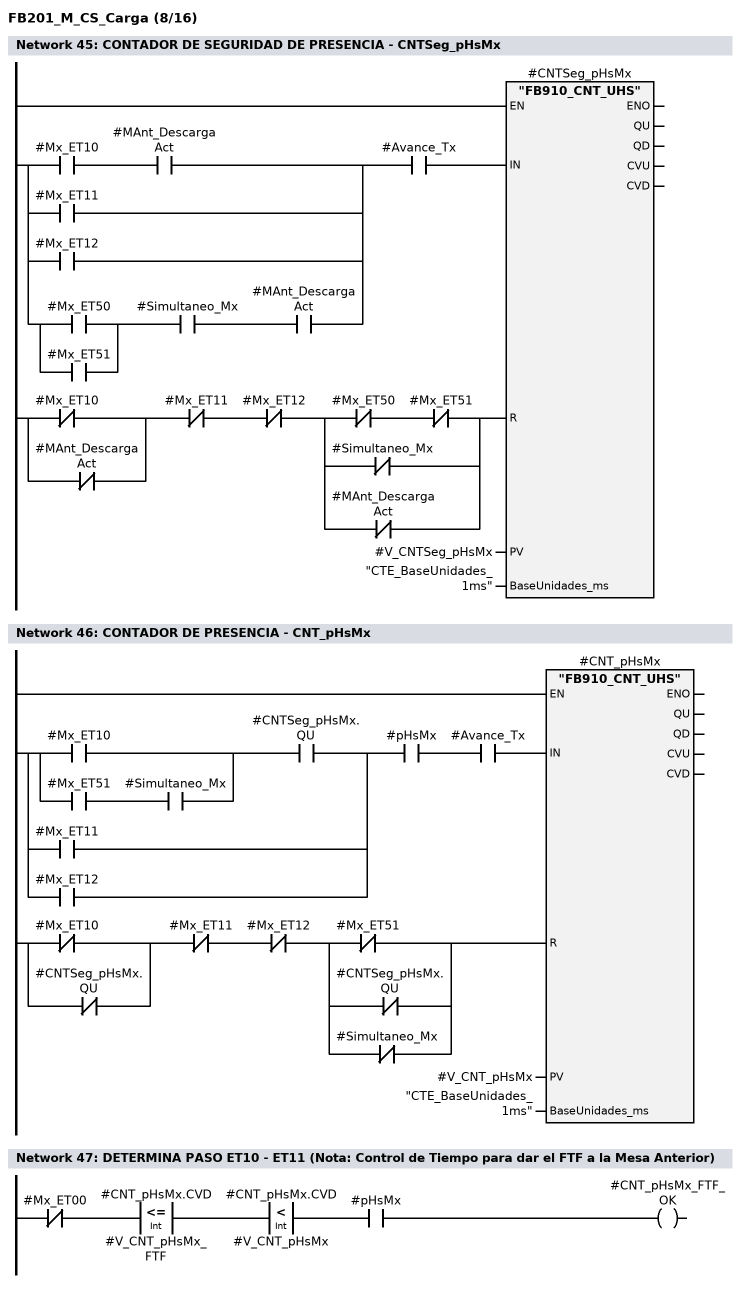
   RUNG wire#powerrail
      #CNTSeg_pHsMx(IN := wire#w3, R := wire#w6, PV := #V_CNTSeg_pHsMx, BaseUnidades_ms := "CTE_BaseUnidades_1ms", QU =>, QD =>, CVU =>, CVD =>)
   END_RUNG
   RUNG wire#powerrail
      Contact( #Mx_ET10 )
      Contact( #MAnt_DescargaAct )
      wire#w1
      Contact( #Avance_Tx )
   END_RUNG wire#w3
   RUNG wire#powerrail
      Contact( #Mx_ET11 )
   END_RUNG wire#w1
   RUNG wire#powerrail
      Contact( #Mx_ET12 )
   END_RUNG wire#w1
   RUNG wire#powerrail
      Contact( #Mx_ET50 )
      wire#w2
      Contact( #Simultaneo_Mx )
      Contact( #MAnt_DescargaAct )
   END_RUNG wire#w1
   RUNG wire#powerrail
      Contact( #Mx_ET51 )
   END_RUNG wire#w2
   RUNG wire#powerrail
      I_Contact( #Mx_ET10 )
      wire#w4
      I_Contact( #Mx_ET11 )
      I_Contact( #Mx_ET12 )
      wire#w5
      I_Contact( #Mx_ET50 )
      I_Contact( #Mx_ET51 )
   END_RUNG wire#w6
   RUNG wire#powerrail
      I_Contact( #MAnt_DescargaAct )
   END_RUNG wire#w4
   RUNG wire#w5
      I_Contact( #Simultaneo_Mx )
   END_RUNG wire#w6
   RUNG wire#w5
      I_Contact( #MAnt_DescargaAct )
   END_RUNG wire#w6
   // the same network as SCL:
   #CNTSeg_pHsMx(IN := ((#Mx_ET10 AND #MAnt_DescargaAct) OR #Mx_ET11 OR #Mx_ET12 OR ((#Mx_ET50 OR #Mx_ET51) AND #Simultaneo_Mx AND #MAnt_DescargaAct)) AND #Avance_Tx,   // "FB910_CNT_UHS"
                 R := (NOT #Mx_ET10 OR NOT #MAnt_DescargaAct) AND NOT #Mx_ET11 AND NOT #Mx_ET12 AND ((NOT #Mx_ET50 AND NOT #Mx_ET51) OR NOT #Simultaneo_Mx OR NOT #MAnt_DescargaAct),
                 PV := #V_CNTSeg_pHsMx,
                 BaseUnidades_ms := "CTE_BaseUnidades_1ms");
END_REGION

REGION Network 46: CONTADOR DE PRESENCIA - CNT_pHsMx
   RUNG wire#powerrail
      #CNT_pHsMx(IN := wire#w3, R := wire#w6, PV := #V_CNT_pHsMx, BaseUnidades_ms := "CTE_BaseUnidades_1ms", QU =>, QD =>, CVU =>, CVD =>)
   END_RUNG
   RUNG wire#powerrail
      Contact( #Mx_ET10 )
      wire#w1
      Contact( #CNTSeg_pHsMx.QU )
      wire#w2
      Contact( #pHsMx )
      Contact( #Avance_Tx )
   END_RUNG wire#w3
   RUNG wire#powerrail
      Contact( #Mx_ET51 )
      Contact( #Simultaneo_Mx )
   END_RUNG wire#w1
   RUNG wire#powerrail
      Contact( #Mx_ET11 )
   END_RUNG wire#w2
   RUNG wire#powerrail
      Contact( #Mx_ET12 )
   END_RUNG wire#w2
   RUNG wire#powerrail
      I_Contact( #Mx_ET10 )
      wire#w4
      I_Contact( #Mx_ET11 )
      I_Contact( #Mx_ET12 )
      wire#w5
      I_Contact( #Mx_ET51 )
   END_RUNG wire#w6
   RUNG wire#powerrail
      I_Contact( #CNTSeg_pHsMx.QU )
   END_RUNG wire#w4
   RUNG wire#w5
      I_Contact( #CNTSeg_pHsMx.QU )
   END_RUNG wire#w6
   RUNG wire#w5
      I_Contact( #Simultaneo_Mx )
   END_RUNG wire#w6
   // the same network as SCL:
   #CNT_pHsMx(IN := (((#Mx_ET10 OR (#Mx_ET51 AND #Simultaneo_Mx)) AND #CNTSeg_pHsMx.QU) OR #Mx_ET11 OR #Mx_ET12) AND #pHsMx AND #Avance_Tx,   // "FB910_CNT_UHS"
              R := (NOT #Mx_ET10 OR NOT #CNTSeg_pHsMx.QU) AND NOT #Mx_ET11 AND NOT #Mx_ET12 AND (NOT #Mx_ET51 OR NOT #CNTSeg_pHsMx.QU OR NOT #Simultaneo_Mx),
              PV := #V_CNT_pHsMx,
              BaseUnidades_ms := "CTE_BaseUnidades_1ms");
END_REGION

REGION Network 47: DETERMINA PASO ET10 - ET11 (Nota: Control de Tiempo para dar el FTF a la Mesa Anterior)
   RUNG wire#powerrail
      I_Contact( #Mx_ET00 )
      { S7_Templates := "SrcType := Int" } LE_Contact(in1 := #CNT_pHsMx.CVD, in2 := #V_CNT_pHsMx_FTF)
      { S7_Templates := "SrcType := Int" } LT_Contact(in1 := #CNT_pHsMx.CVD, in2 := #V_CNT_pHsMx)
      Contact( #pHsMx )
      Coil( #CNT_pHsMx_FTF_OK )
   END_RUNG
   // the same network as SCL:
   #CNT_pHsMx_FTF_OK := NOT #Mx_ET00 AND (#CNT_pHsMx.CVD <= #V_CNT_pHsMx_FTF) AND (#CNT_pHsMx.CVD < #V_CNT_pHsMx) AND #pHsMx;
END_REGION

REGION Network 48: CONTADOR SEGURIDAD DE AUSENCIA - CNTSeg_ApHsMx ??????? RESTAR VALOR DE POSICIONAMIENTO
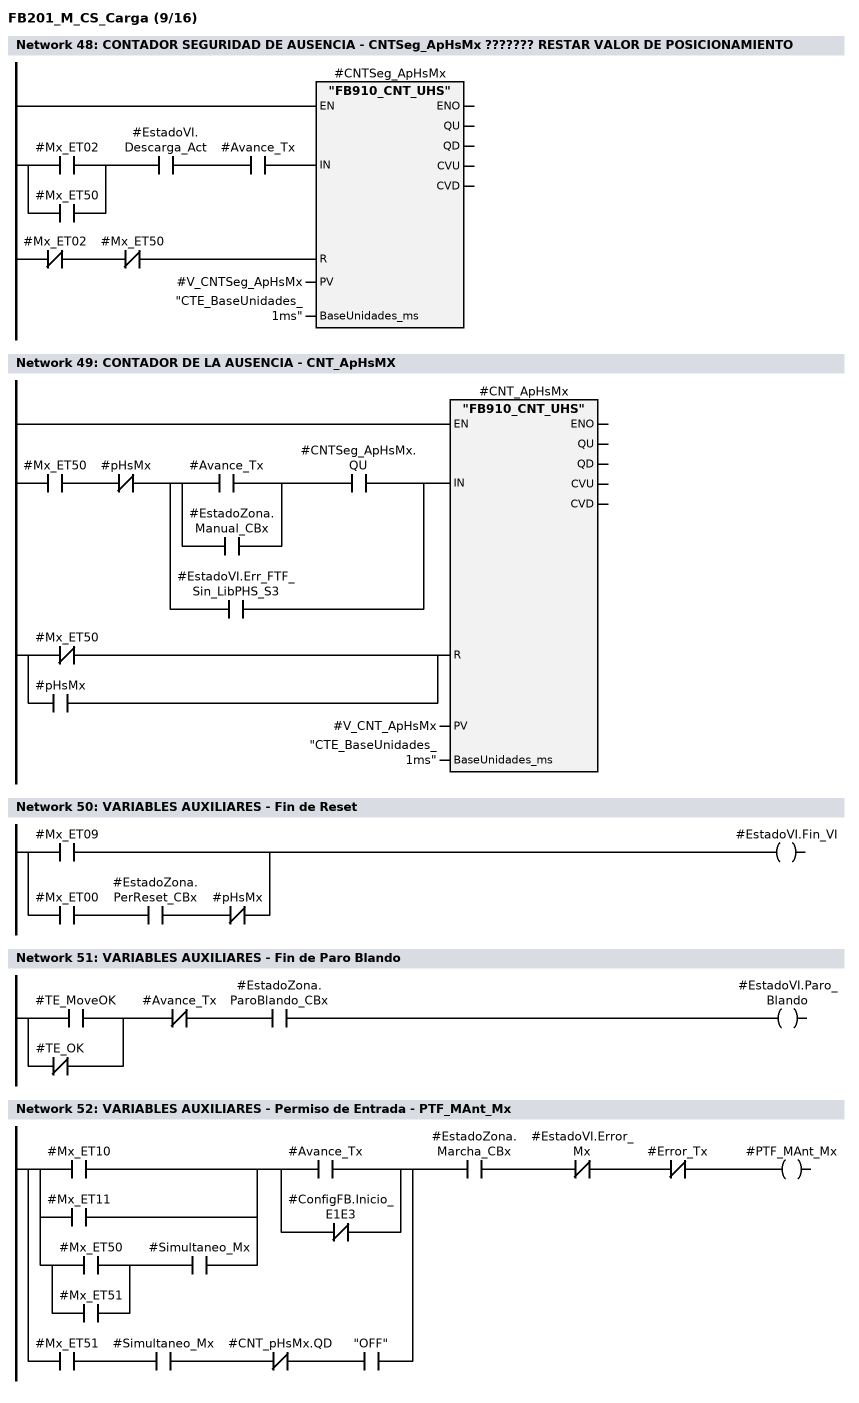
   RUNG wire#powerrail
      #CNTSeg_ApHsMx(IN := wire#w2, R := wire#w3, PV := #V_CNTSeg_ApHsMx, BaseUnidades_ms := "CTE_BaseUnidades_1ms", QU =>, QD =>, CVU =>, CVD =>)
   END_RUNG
   RUNG wire#powerrail
      Contact( #Mx_ET02 )
      wire#w1
      Contact( #EstadoVI.Descarga_Act )
      Contact( #Avance_Tx )
   END_RUNG wire#w2
   RUNG wire#powerrail
      Contact( #Mx_ET50 )
   END_RUNG wire#w1
   RUNG wire#powerrail
      I_Contact( #Mx_ET02 )
      I_Contact( #Mx_ET50 )
   END_RUNG wire#w3
   // the same network as SCL:
   #CNTSeg_ApHsMx(IN := (#Mx_ET02 OR #Mx_ET50) AND #EstadoVI.Descarga_Act AND #Avance_Tx,   // "FB910_CNT_UHS"
                  R := NOT #Mx_ET02 AND NOT #Mx_ET50,
                  PV := #V_CNTSeg_ApHsMx,
                  BaseUnidades_ms := "CTE_BaseUnidades_1ms");
END_REGION

REGION Network 49: CONTADOR DE LA AUSENCIA - CNT_ApHsMX
   RUNG wire#powerrail
      #CNT_ApHsMx(IN := wire#w3, R := wire#w4, PV := #V_CNT_ApHsMx, BaseUnidades_ms := "CTE_BaseUnidades_1ms", QU =>, QD =>, CVU =>, CVD =>)
   END_RUNG
   RUNG wire#powerrail
      Contact( #Mx_ET50 )
      I_Contact( #pHsMx )
      wire#w1
      Contact( #Avance_Tx )
      wire#w2
      Contact( #CNTSeg_ApHsMx.QU )
   END_RUNG wire#w3
   RUNG wire#w1
      Contact( #EstadoZona.Manual_CBx )
   END_RUNG wire#w2
   RUNG wire#w1
      Contact( #EstadoVI.Err_FTF_Sin_LibPHS_S3 )
   END_RUNG wire#w3
   RUNG wire#powerrail
      I_Contact( #Mx_ET50 )
   END_RUNG wire#w4
   RUNG wire#powerrail
      Contact( #pHsMx )
   END_RUNG wire#w4
   // the same network as SCL:
   #CNT_ApHsMx(IN := #Mx_ET50 AND NOT #pHsMx AND (((#Avance_Tx OR #EstadoZona.Manual_CBx) AND #CNTSeg_ApHsMx.QU) OR #EstadoVI.Err_FTF_Sin_LibPHS_S3),   // "FB910_CNT_UHS"
               R := NOT #Mx_ET50 OR #pHsMx,
               PV := #V_CNT_ApHsMx,
               BaseUnidades_ms := "CTE_BaseUnidades_1ms");
END_REGION

REGION Network 50: VARIABLES AUXILIARES - Fin de Reset
   RUNG wire#powerrail
      Contact( #Mx_ET09 )
      wire#w1
      Coil( #EstadoVI.Fin_VI )
   END_RUNG
   RUNG wire#powerrail
      Contact( #Mx_ET00 )
      Contact( #EstadoZona.PerReset_CBx )
      I_Contact( #pHsMx )
   END_RUNG wire#w1
   // the same network as SCL:
   #EstadoVI.Fin_VI := #Mx_ET09 OR (#Mx_ET00 AND #EstadoZona.PerReset_CBx AND NOT #pHsMx);
END_REGION

REGION Network 51: VARIABLES AUXILIARES - Fin de Paro Blando
   RUNG wire#powerrail
      Contact( #TE_MoveOK )
      wire#w1
      I_Contact( #Avance_Tx )
      Contact( #EstadoZona.ParoBlando_CBx )
      Coil( #EstadoVI.Paro_Blando )
   END_RUNG
   RUNG wire#powerrail
      I_Contact( #TE_OK )
   END_RUNG wire#w1
   // the same network as SCL:
   #EstadoVI.Paro_Blando := (#TE_MoveOK OR NOT #TE_OK) AND NOT #Avance_Tx AND #EstadoZona.ParoBlando_CBx;
END_REGION

REGION Network 52: VARIABLES AUXILIARES - Permiso de Entrada - PTF_MAnt_Mx
   RUNG wire#powerrail
      Contact( #Mx_ET10 )
      wire#w1
      Contact( #Avance_Tx )
      wire#w3
      Contact( #EstadoZona.Marcha_CBx )
      I_Contact( #EstadoVI.Error_Mx )
      I_Contact( #Error_Tx )
      Coil( #PTF_MAnt_Mx )
   END_RUNG
   RUNG wire#powerrail
      Contact( #Mx_ET11 )
   END_RUNG wire#w1
   RUNG wire#powerrail
      Contact( #Mx_ET50 )
      wire#w2
      Contact( #Simultaneo_Mx )
   END_RUNG wire#w1
   RUNG wire#powerrail
      Contact( #Mx_ET51 )
   END_RUNG wire#w2
   RUNG wire#w1
      I_Contact( #ConfigFB.Inicio_E1E3 )
   END_RUNG wire#w3
   RUNG wire#powerrail
      Contact( #Mx_ET51 )
      Contact( #Simultaneo_Mx )
      I_Contact( #CNT_pHsMx.QD )
      Contact( "OFF" )
   END_RUNG wire#w3
   // the same network as SCL:
   #PTF_MAnt_Mx := (((#Mx_ET10 OR #Mx_ET11 OR ((#Mx_ET50 OR #Mx_ET51) AND #Simultaneo_Mx)) AND (#Avance_Tx OR NOT #ConfigFB.Inicio_E1E3)) OR (#Mx_ET51 AND #Simultaneo_Mx AND NOT #CNT_pHsMx.QD AND "OFF")) AND #EstadoZona.Marcha_CBx AND NOT #EstadoVI.Error_Mx AND NOT #Error_Tx;
END_REGION

REGION Network 53: VARIABLES AUXILIARES - Aviso de Salida - AVTF_Mx_MSig
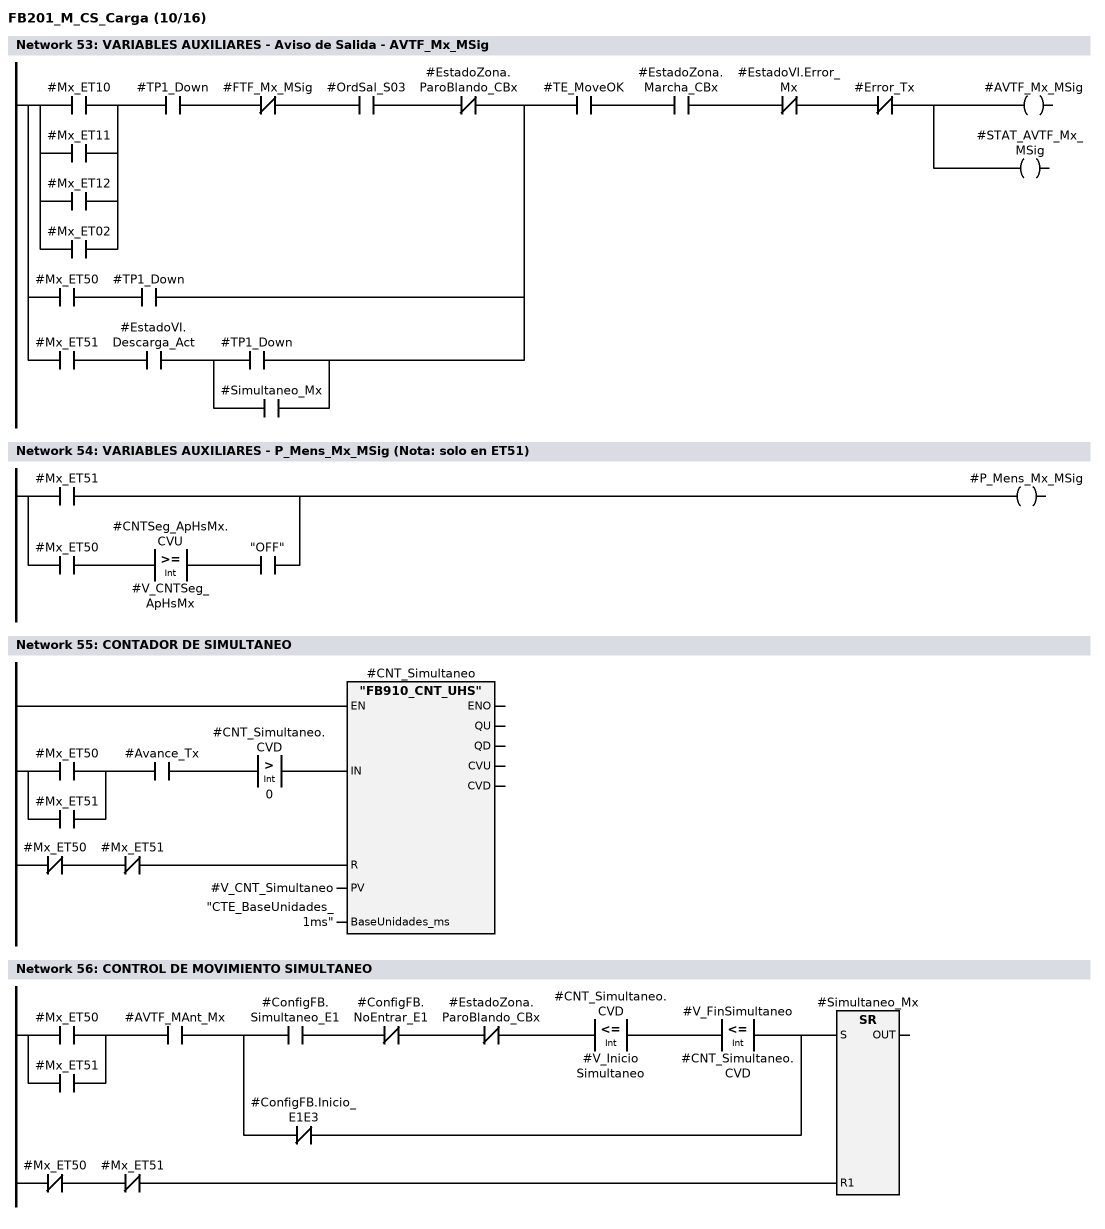
   RUNG wire#powerrail
      Contact( #Mx_ET10 )
      wire#w1
      Contact( #TP1_Down )
      I_Contact( #FTF_Mx_MSig )
      Contact( #OrdSal_S03 )
      I_Contact( #EstadoZona.ParoBlando_CBx )
      wire#w2
      Contact( #TE_MoveOK )
      Contact( #EstadoZona.Marcha_CBx )
      I_Contact( #EstadoVI.Error_Mx )
      I_Contact( #Error_Tx )
      wire#w4
      Coil( #AVTF_Mx_MSig )
   END_RUNG
   RUNG wire#powerrail
      Contact( #Mx_ET11 )
   END_RUNG wire#w1
   RUNG wire#powerrail
      Contact( #Mx_ET12 )
   END_RUNG wire#w1
   RUNG wire#powerrail
      Contact( #Mx_ET02 )
   END_RUNG wire#w1
   RUNG wire#powerrail
      Contact( #Mx_ET50 )
      Contact( #TP1_Down )
   END_RUNG wire#w2
   RUNG wire#powerrail
      Contact( #Mx_ET51 )
      Contact( #EstadoVI.Descarga_Act )
      wire#w3
      Contact( #TP1_Down )
   END_RUNG wire#w2
   RUNG wire#w3
      Contact( #Simultaneo_Mx )
   END_RUNG wire#w2
   RUNG wire#w4
      Coil( #STAT_AVTF_Mx_MSig )
   END_RUNG
   // the same network as SCL:
   #AVTF_Mx_MSig := (((#Mx_ET10 OR #Mx_ET11 OR #Mx_ET12 OR #Mx_ET02) AND #TP1_Down AND NOT #FTF_Mx_MSig AND #OrdSal_S03 AND NOT #EstadoZona.ParoBlando_CBx) OR (#Mx_ET50 AND #TP1_Down) OR (#Mx_ET51 AND #EstadoVI.Descarga_Act AND (#TP1_Down OR #Simultaneo_Mx))) AND #TE_MoveOK AND #EstadoZona.Marcha_CBx AND NOT #EstadoVI.Error_Mx AND NOT #Error_Tx;
   #STAT_AVTF_Mx_MSig := #AVTF_Mx_MSig;
END_REGION

REGION Network 54: VARIABLES AUXILIARES - P_Mens_Mx_MSig (Nota: solo en ET51)
   RUNG wire#powerrail
      Contact( #Mx_ET51 )
      wire#w1
      Coil( #P_Mens_Mx_MSig )
   END_RUNG
   RUNG wire#powerrail
      Contact( #Mx_ET50 )
      { S7_Templates := "SrcType := Int" } GE_Contact(in1 := #CNTSeg_ApHsMx.CVU, in2 := #V_CNTSeg_ApHsMx)
      Contact( "OFF" )
   END_RUNG wire#w1
   // the same network as SCL:
   #P_Mens_Mx_MSig := #Mx_ET51 OR (#Mx_ET50 AND (#CNTSeg_ApHsMx.CVU >= #V_CNTSeg_ApHsMx) AND "OFF");
END_REGION

REGION Network 55: CONTADOR DE SIMULTANEO
   RUNG wire#powerrail
      #CNT_Simultaneo(IN := wire#w2, R := wire#w3, PV := #V_CNT_Simultaneo, BaseUnidades_ms := "CTE_BaseUnidades_1ms", QU =>, QD =>, CVU =>, CVD =>)
   END_RUNG
   RUNG wire#powerrail
      Contact( #Mx_ET50 )
      wire#w1
      Contact( #Avance_Tx )
      { S7_Templates := "SrcType := Int" } GT_Contact(in1 := #CNT_Simultaneo.CVD, in2 := 0)
   END_RUNG wire#w2
   RUNG wire#powerrail
      Contact( #Mx_ET51 )
   END_RUNG wire#w1
   RUNG wire#powerrail
      I_Contact( #Mx_ET50 )
      I_Contact( #Mx_ET51 )
   END_RUNG wire#w3
   // the same network as SCL:
   #CNT_Simultaneo(IN := (#Mx_ET50 OR #Mx_ET51) AND #Avance_Tx AND (#CNT_Simultaneo.CVD > 0),   // "FB910_CNT_UHS"
                   R := NOT #Mx_ET50 AND NOT #Mx_ET51,
                   PV := #V_CNT_Simultaneo,
                   BaseUnidades_ms := "CTE_BaseUnidades_1ms");
END_REGION

REGION Network 56: CONTROL DE MOVIMIENTO SIMULTANEO
   RUNG wire#powerrail
      Contact( #Mx_ET50 )
      wire#w1
      Contact( #AVTF_MAnt_Mx )
      wire#w2
      Contact( #ConfigFB.Simultaneo_E1 )
      I_Contact( #ConfigFB.NoEntrar_E1 )
      I_Contact( #EstadoZona.ParoBlando_CBx )
      { S7_Templates := "SrcType := Int" } LE_Contact(in1 := #CNT_Simultaneo.CVD, in2 := #V_InicioSimultaneo)
      { S7_Templates := "SrcType := Int" } LE_Contact(in1 := #V_FinSimultaneo, in2 := #CNT_Simultaneo.CVD)
      wire#w3
      S_SR(operand := #Simultaneo_Mx, r1 := wire#w4)
   END_RUNG
   RUNG wire#powerrail
      Contact( #Mx_ET51 )
   END_RUNG wire#w1
   RUNG wire#w2
      I_Contact( #ConfigFB.Inicio_E1E3 )
   END_RUNG wire#w3
   RUNG wire#powerrail
      I_Contact( #Mx_ET50 )
      I_Contact( #Mx_ET51 )
   END_RUNG wire#w4
   // the same network as SCL:
   IF (#Mx_ET50 OR #Mx_ET51) AND #AVTF_MAnt_Mx AND ((#ConfigFB.Simultaneo_E1 AND NOT #ConfigFB.NoEntrar_E1 AND NOT #EstadoZona.ParoBlando_CBx AND (#CNT_Simultaneo.CVD <= #V_InicioSimultaneo) AND (#V_FinSimultaneo <= #CNT_Simultaneo.CVD)) OR NOT #ConfigFB.Inicio_E1E3) THEN
       #Simultaneo_Mx := TRUE;   // SR flip-flop
   END_IF;
   IF NOT #Mx_ET50 AND NOT #Mx_ET51 THEN #Simultaneo_Mx := FALSE; END_IF;
END_REGION

REGION Network 57: MENSAJES - PRESENCIA
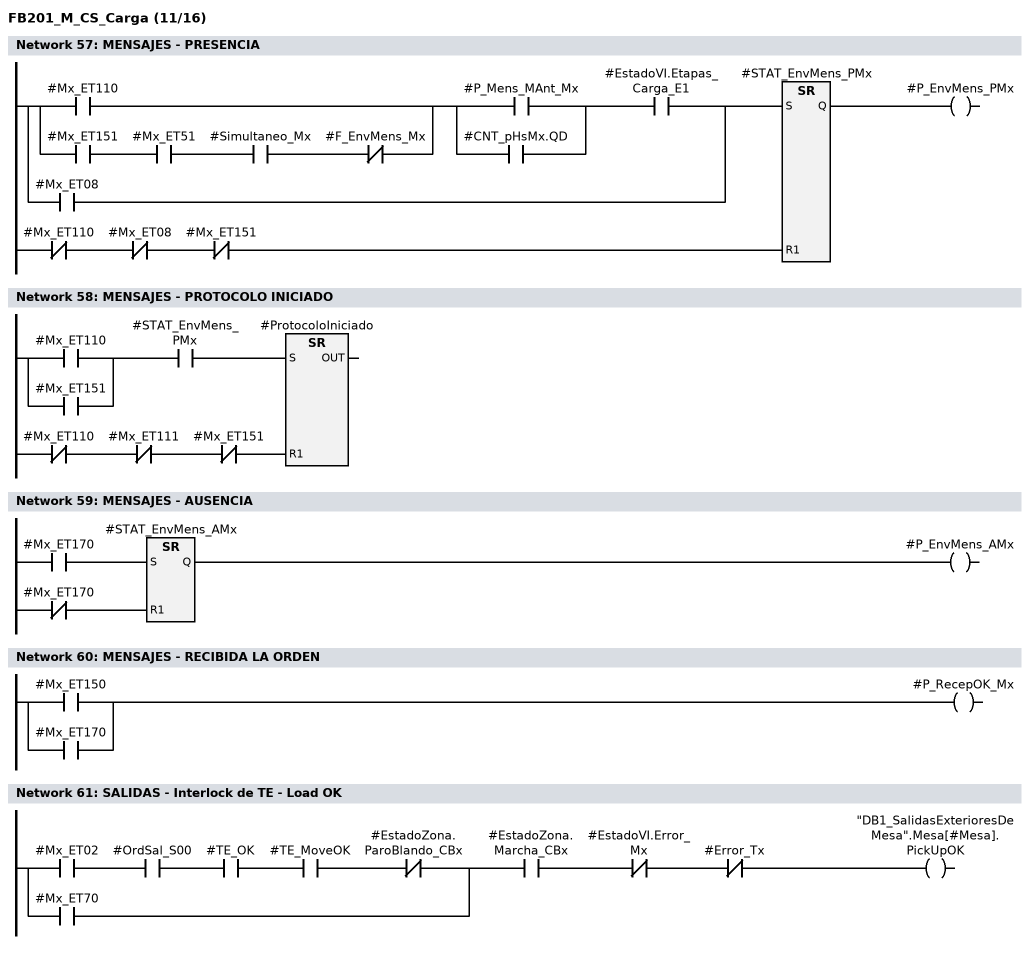
   RUNG wire#powerrail
      Contact( #Mx_ET110 )
      wire#w1
      Contact( #P_Mens_MAnt_Mx )
      wire#w2
      Contact( #EstadoVI.Etapas_Carga_E1 )
      wire#w3
      S_SR(operand := #STAT_EnvMens_PMx, r1 := wire#w4)
      Coil( #P_EnvMens_PMx )
   END_RUNG
   RUNG wire#powerrail
      Contact( #Mx_ET151 )
      Contact( #Mx_ET51 )
      Contact( #Simultaneo_Mx )
      I_Contact( #F_EnvMens_Mx )
   END_RUNG wire#w1
   RUNG wire#w1
      Contact( #CNT_pHsMx.QD )
   END_RUNG wire#w2
   RUNG wire#powerrail
      Contact( #Mx_ET08 )
   END_RUNG wire#w3
   RUNG wire#powerrail
      I_Contact( #Mx_ET110 )
      I_Contact( #Mx_ET08 )
      I_Contact( #Mx_ET151 )
   END_RUNG wire#w4
   // the same network as SCL:
   IF ((#Mx_ET110 OR (#Mx_ET151 AND #Mx_ET51 AND #Simultaneo_Mx AND NOT #F_EnvMens_Mx)) AND (#P_Mens_MAnt_Mx OR #CNT_pHsMx.QD) AND #EstadoVI.Etapas_Carga_E1) OR #Mx_ET08 THEN
       #STAT_EnvMens_PMx := TRUE;   // SR flip-flop
   END_IF;
   IF NOT #Mx_ET110 AND NOT #Mx_ET08 AND NOT #Mx_ET151 THEN #STAT_EnvMens_PMx := FALSE; END_IF;
   #P_EnvMens_PMx := #STAT_EnvMens_PMx;
END_REGION

REGION Network 58: MENSAJES - PROTOCOLO INICIADO
   RUNG wire#powerrail
      Contact( #Mx_ET110 )
      wire#w1
      Contact( #STAT_EnvMens_PMx )
      S_SR(operand := #ProtocoloIniciado, r1 := wire#w2)
   END_RUNG
   RUNG wire#powerrail
      Contact( #Mx_ET151 )
   END_RUNG wire#w1
   RUNG wire#powerrail
      I_Contact( #Mx_ET110 )
      I_Contact( #Mx_ET111 )
      I_Contact( #Mx_ET151 )
   END_RUNG wire#w2
   // the same network as SCL:
   IF (#Mx_ET110 OR #Mx_ET151) AND #STAT_EnvMens_PMx THEN
       #ProtocoloIniciado := TRUE;   // SR flip-flop
   END_IF;
   IF NOT #Mx_ET110 AND NOT #Mx_ET111 AND NOT #Mx_ET151 THEN #ProtocoloIniciado := FALSE; END_IF;
END_REGION

REGION Network 59: MENSAJES - AUSENCIA
   RUNG wire#powerrail
      Contact( #Mx_ET170 )
      S_SR(operand := #STAT_EnvMens_AMx, r1 := wire#w1)
      Coil( #P_EnvMens_AMx )
   END_RUNG
   RUNG wire#powerrail
      I_Contact( #Mx_ET170 )
   END_RUNG wire#w1
   // the same network as SCL:
   IF #Mx_ET170 THEN
       #STAT_EnvMens_AMx := TRUE;   // SR flip-flop
   END_IF;
   IF NOT #Mx_ET170 THEN #STAT_EnvMens_AMx := FALSE; END_IF;
   #P_EnvMens_AMx := #STAT_EnvMens_AMx;
END_REGION

REGION Network 60: MENSAJES - RECIBIDA LA ORDEN
   RUNG wire#powerrail
      Contact( #Mx_ET150 )
      wire#w1
      Coil( #P_RecepOK_Mx )
   END_RUNG
   RUNG wire#powerrail
      Contact( #Mx_ET170 )
   END_RUNG wire#w1
   // the same network as SCL:
   #P_RecepOK_Mx := #Mx_ET150 OR #Mx_ET170;
END_REGION

REGION Network 61: SALIDAS - Interlock de TE - Load OK
   RUNG wire#powerrail
      Contact( #Mx_ET02 )
      Contact( #OrdSal_S00 )
      Contact( #TE_OK )
      Contact( #TE_MoveOK )
      I_Contact( #EstadoZona.ParoBlando_CBx )
      wire#w1
      Contact( #EstadoZona.Marcha_CBx )
      I_Contact( #EstadoVI.Error_Mx )
      I_Contact( #Error_Tx )
      Coil( "DB1_SalidasExterioresDeMesa".Mesa[#Mesa].PickUpOK )
   END_RUNG
   RUNG wire#powerrail
      Contact( #Mx_ET70 )
   END_RUNG wire#w1
   // the same network as SCL:
   "DB1_SalidasExterioresDeMesa".Mesa[#Mesa].PickUpOK := ((#Mx_ET02 AND #OrdSal_S00 AND #TE_OK AND #TE_MoveOK AND NOT #EstadoZona.ParoBlando_CBx) OR #Mx_ET70) AND #EstadoZona.Marcha_CBx AND NOT #EstadoVI.Error_Mx AND NOT #Error_Tx;
END_REGION

REGION Network 62: SALIDAS - Avance E1E3
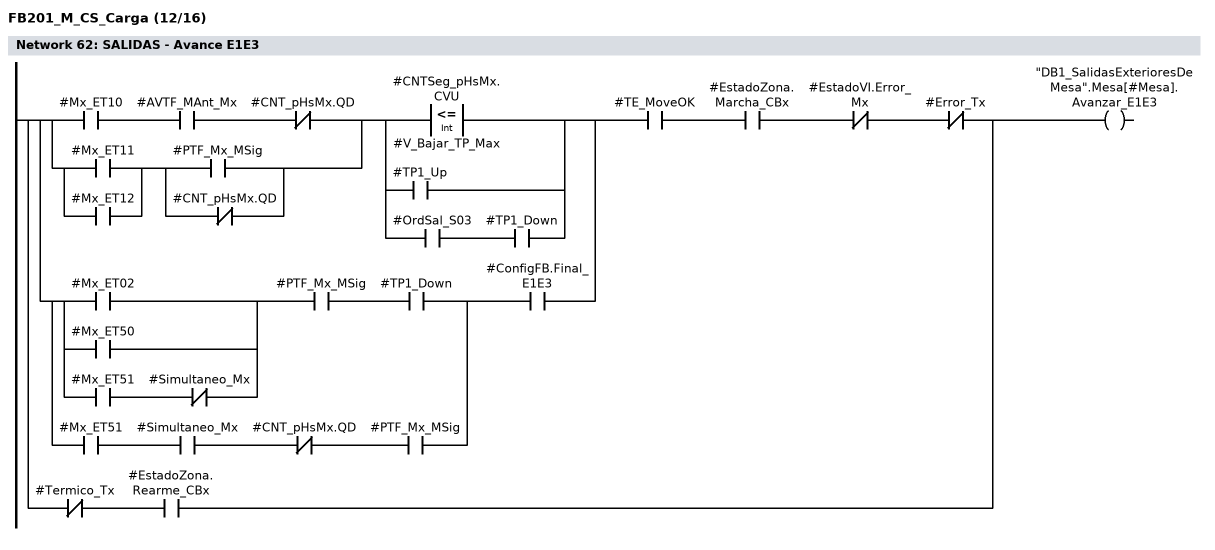
   RUNG wire#powerrail
      Contact( #Mx_ET10 )
      Contact( #AVTF_MAnt_Mx )
      I_Contact( #CNT_pHsMx.QD )
      wire#w1
      { S7_Templates := "SrcType := Int" } LE_Contact(in1 := #CNTSeg_pHsMx.CVU, in2 := #V_Bajar_TP_Max)
      wire#w3
      Contact( #TE_MoveOK )
      Contact( #EstadoZona.Marcha_CBx )
      I_Contact( #EstadoVI.Error_Mx )
      I_Contact( #Error_Tx )
      wire#w6
      Coil( "DB1_SalidasExterioresDeMesa".Mesa[#Mesa].Avanzar_E1E3 )
   END_RUNG
   RUNG wire#powerrail
      Contact( #Mx_ET11 )
      wire#w2
      Contact( #PTF_Mx_MSig )
   END_RUNG wire#w1
   RUNG wire#powerrail
      Contact( #Mx_ET12 )
   END_RUNG wire#w2
   RUNG wire#w2
      I_Contact( #CNT_pHsMx.QD )
   END_RUNG wire#w1
   RUNG wire#w1
      Contact( #TP1_Up )
   END_RUNG wire#w3
   RUNG wire#w1
      Contact( #OrdSal_S03 )
      Contact( #TP1_Down )
   END_RUNG wire#w3
   RUNG wire#powerrail
      Contact( #Mx_ET02 )
      wire#w4
      Contact( #PTF_Mx_MSig )
      Contact( #TP1_Down )
      wire#w5
      Contact( #ConfigFB.Final_E1E3 )
   END_RUNG wire#w3
   RUNG wire#powerrail
      Contact( #Mx_ET50 )
   END_RUNG wire#w4
   RUNG wire#powerrail
      Contact( #Mx_ET51 )
      I_Contact( #Simultaneo_Mx )
   END_RUNG wire#w4
   RUNG wire#powerrail
      Contact( #Mx_ET51 )
      Contact( #Simultaneo_Mx )
      I_Contact( #CNT_pHsMx.QD )
      Contact( #PTF_Mx_MSig )
   END_RUNG wire#w5
   RUNG wire#powerrail
      I_Contact( #Termico_Tx )
      Contact( #EstadoZona.Rearme_CBx )
   END_RUNG wire#w6
   // the same network as SCL:
   "DB1_SalidasExterioresDeMesa".Mesa[#Mesa].Avanzar_E1E3 := (((((#Mx_ET10 AND #AVTF_MAnt_Mx AND NOT #CNT_pHsMx.QD) OR ((#Mx_ET11 OR #Mx_ET12) AND (#PTF_Mx_MSig OR NOT #CNT_pHsMx.QD))) AND ((#CNTSeg_pHsMx.CVU <= #V_Bajar_TP_Max) OR #TP1_Up OR (#OrdSal_S03 AND #TP1_Down))) OR ((((#Mx_ET02 OR #Mx_ET50 OR (#Mx_ET51 AND NOT #Simultaneo_Mx)) AND #PTF_Mx_MSig AND #TP1_Down) OR (#Mx_ET51 AND #Simultaneo_Mx AND NOT #CNT_pHsMx.QD AND #PTF_Mx_MSig)) AND #ConfigFB.Final_E1E3)) AND #TE_MoveOK AND #EstadoZona.Marcha_CBx AND NOT #EstadoVI.Error_Mx AND NOT #Error_Tx) OR (NOT #Termico_Tx AND #EstadoZona.Rearme_CBx);
END_REGION

REGION Network 63: SALIDAS - Parar E1E3
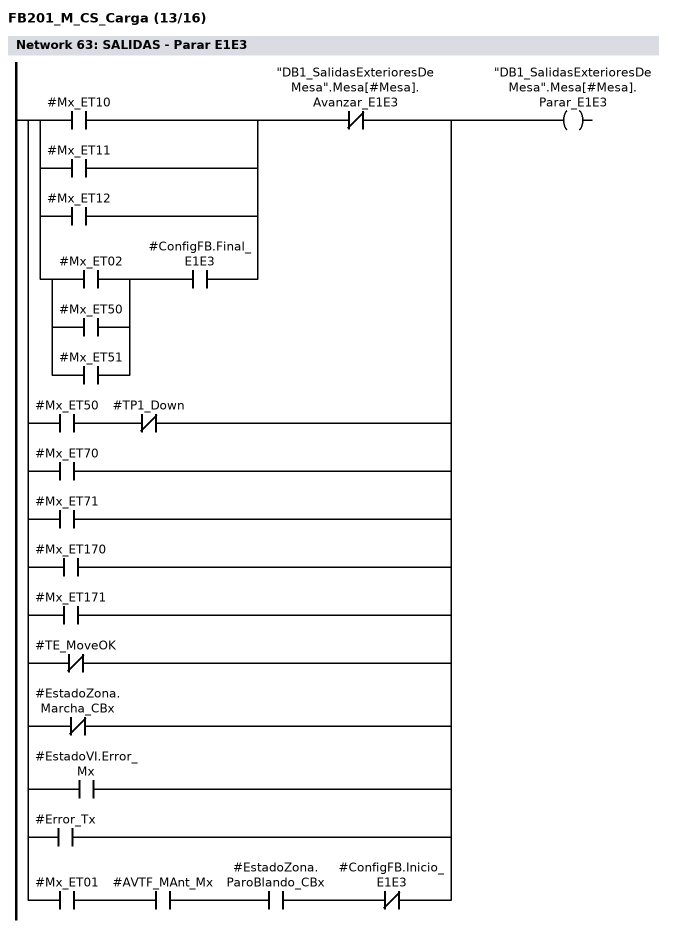
   RUNG wire#powerrail
      Contact( #Mx_ET10 )
      wire#w1
      I_Contact( "DB1_SalidasExterioresDeMesa".Mesa[#Mesa].Avanzar_E1E3 )
      wire#w3
      Coil( "DB1_SalidasExterioresDeMesa".Mesa[#Mesa].Parar_E1E3 )
   END_RUNG
   RUNG wire#powerrail
      Contact( #Mx_ET11 )
   END_RUNG wire#w1
   RUNG wire#powerrail
      Contact( #Mx_ET12 )
   END_RUNG wire#w1
   RUNG wire#powerrail
      Contact( #Mx_ET02 )
      wire#w2
      Contact( #ConfigFB.Final_E1E3 )
   END_RUNG wire#w1
   RUNG wire#powerrail
      Contact( #Mx_ET50 )
   END_RUNG wire#w2
   RUNG wire#powerrail
      Contact( #Mx_ET51 )
   END_RUNG wire#w2
   RUNG wire#powerrail
      Contact( #Mx_ET50 )
      I_Contact( #TP1_Down )
   END_RUNG wire#w3
   RUNG wire#powerrail
      Contact( #Mx_ET70 )
   END_RUNG wire#w3
   RUNG wire#powerrail
      Contact( #Mx_ET71 )
   END_RUNG wire#w3
   RUNG wire#powerrail
      Contact( #Mx_ET170 )
   END_RUNG wire#w3
   RUNG wire#powerrail
      Contact( #Mx_ET171 )
   END_RUNG wire#w3
   RUNG wire#powerrail
      I_Contact( #TE_MoveOK )
   END_RUNG wire#w3
   RUNG wire#powerrail
      I_Contact( #EstadoZona.Marcha_CBx )
   END_RUNG wire#w3
   RUNG wire#powerrail
      Contact( #EstadoVI.Error_Mx )
   END_RUNG wire#w3
   RUNG wire#powerrail
      Contact( #Error_Tx )
   END_RUNG wire#w3
   RUNG wire#powerrail
      Contact( #Mx_ET01 )
      Contact( #AVTF_MAnt_Mx )
      Contact( #EstadoZona.ParoBlando_CBx )
      I_Contact( #ConfigFB.Inicio_E1E3 )
   END_RUNG wire#w3
   // the same network as SCL:
   "DB1_SalidasExterioresDeMesa".Mesa[#Mesa].Parar_E1E3 := ((#Mx_ET10 OR #Mx_ET11 OR #Mx_ET12 OR ((#Mx_ET02 OR #Mx_ET50 OR #Mx_ET51) AND #ConfigFB.Final_E1E3)) AND NOT "DB1_SalidasExterioresDeMesa".Mesa[#Mesa].Avanzar_E1E3) OR (#Mx_ET50 AND NOT #TP1_Down) OR #Mx_ET70 OR #Mx_ET71 OR #Mx_ET170 OR #Mx_ET171 OR NOT #TE_MoveOK OR NOT #EstadoZona.Marcha_CBx OR #EstadoVI.Error_Mx OR #Error_Tx OR (#Mx_ET01 AND #AVTF_MAnt_Mx AND #EstadoZona.ParoBlando_CBx AND NOT #ConfigFB.Inicio_E1E3);
END_REGION

REGION Network 64: SALIDAS - Valor Frecuencia Lenta E1E3
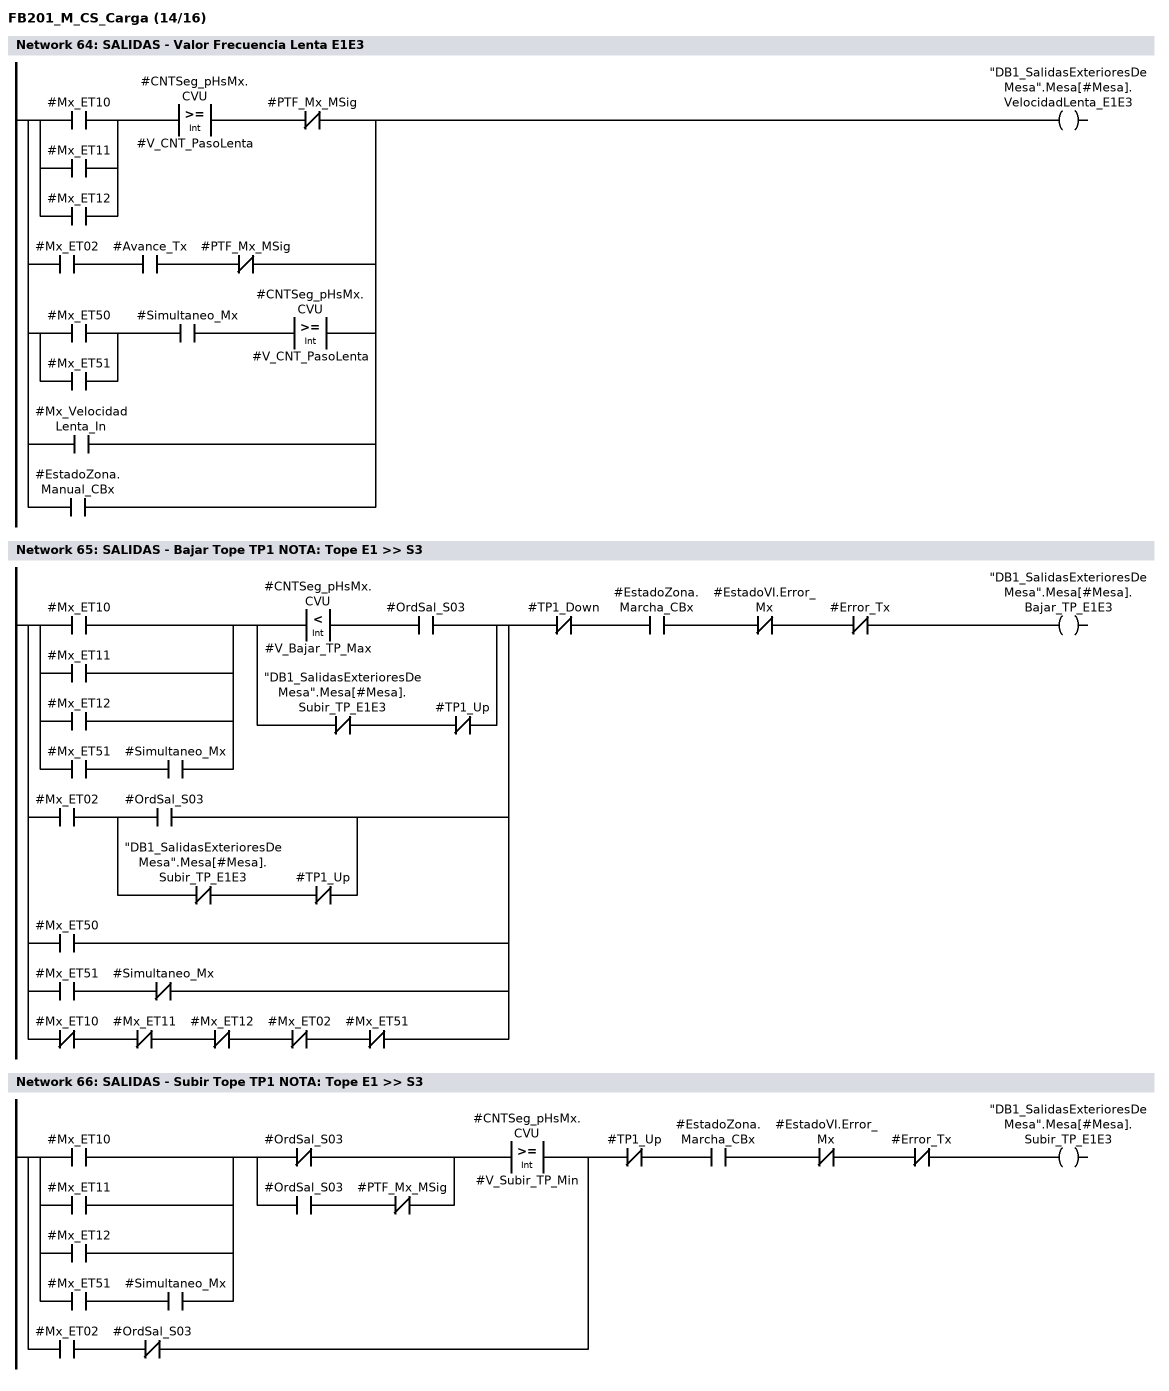
   RUNG wire#powerrail
      Contact( #Mx_ET10 )
      wire#w1
      { S7_Templates := "SrcType := Int" } GE_Contact(in1 := #CNTSeg_pHsMx.CVU, in2 := #V_CNT_PasoLenta)
      I_Contact( #PTF_Mx_MSig )
      wire#w2
      Coil( "DB1_SalidasExterioresDeMesa".Mesa[#Mesa].VelocidadLenta_E1E3 )
   END_RUNG
   RUNG wire#powerrail
      Contact( #Mx_ET11 )
   END_RUNG wire#w1
   RUNG wire#powerrail
      Contact( #Mx_ET12 )
   END_RUNG wire#w1
   RUNG wire#powerrail
      Contact( #Mx_ET02 )
      Contact( #Avance_Tx )
      I_Contact( #PTF_Mx_MSig )
   END_RUNG wire#w2
   RUNG wire#powerrail
      Contact( #Mx_ET50 )
      wire#w3
      Contact( #Simultaneo_Mx )
      { S7_Templates := "SrcType := Int" } GE_Contact(in1 := #CNTSeg_pHsMx.CVU, in2 := #V_CNT_PasoLenta)
   END_RUNG wire#w2
   RUNG wire#powerrail
      Contact( #Mx_ET51 )
   END_RUNG wire#w3
   RUNG wire#powerrail
      Contact( #Mx_VelocidadLenta_In )
   END_RUNG wire#w2
   RUNG wire#powerrail
      Contact( #EstadoZona.Manual_CBx )
   END_RUNG wire#w2
   // the same network as SCL:
   "DB1_SalidasExterioresDeMesa".Mesa[#Mesa].VelocidadLenta_E1E3 := ((#Mx_ET10 OR #Mx_ET11 OR #Mx_ET12) AND (#CNTSeg_pHsMx.CVU >= #V_CNT_PasoLenta) AND NOT #PTF_Mx_MSig) OR (#Mx_ET02 AND #Avance_Tx AND NOT #PTF_Mx_MSig) OR ((#Mx_ET50 OR #Mx_ET51) AND #Simultaneo_Mx AND (#CNTSeg_pHsMx.CVU >= #V_CNT_PasoLenta)) OR #Mx_VelocidadLenta_In OR #EstadoZona.Manual_CBx;
END_REGION

REGION Network 65: SALIDAS - Bajar Tope TP1 NOTA: Tope E1 >> S3
   RUNG wire#powerrail
      Contact( #Mx_ET10 )
      wire#w1
      { S7_Templates := "SrcType := Int" } LT_Contact(in1 := #CNTSeg_pHsMx.CVU, in2 := #V_Bajar_TP_Max)
      Contact( #OrdSal_S03 )
      wire#w2
      I_Contact( #TP1_Down )
      Contact( #EstadoZona.Marcha_CBx )
      I_Contact( #EstadoVI.Error_Mx )
      I_Contact( #Error_Tx )
      Coil( "DB1_SalidasExterioresDeMesa".Mesa[#Mesa].Bajar_TP_E1E3 )
   END_RUNG
   RUNG wire#powerrail
      Contact( #Mx_ET11 )
   END_RUNG wire#w1
   RUNG wire#powerrail
      Contact( #Mx_ET12 )
   END_RUNG wire#w1
   RUNG wire#powerrail
      Contact( #Mx_ET51 )
      Contact( #Simultaneo_Mx )
   END_RUNG wire#w1
   RUNG wire#w1
      I_Contact( "DB1_SalidasExterioresDeMesa".Mesa[#Mesa].Subir_TP_E1E3 )
      I_Contact( #TP1_Up )
   END_RUNG wire#w2
   RUNG wire#powerrail
      Contact( #Mx_ET02 )
      wire#w3
      Contact( #OrdSal_S03 )
   END_RUNG wire#w2
   RUNG wire#w3
      I_Contact( "DB1_SalidasExterioresDeMesa".Mesa[#Mesa].Subir_TP_E1E3 )
      I_Contact( #TP1_Up )
   END_RUNG wire#w2
   RUNG wire#powerrail
      Contact( #Mx_ET50 )
   END_RUNG wire#w2
   RUNG wire#powerrail
      Contact( #Mx_ET51 )
      I_Contact( #Simultaneo_Mx )
   END_RUNG wire#w2
   RUNG wire#powerrail
      I_Contact( #Mx_ET10 )
      I_Contact( #Mx_ET11 )
      I_Contact( #Mx_ET12 )
      I_Contact( #Mx_ET02 )
      I_Contact( #Mx_ET51 )
   END_RUNG wire#w2
   // the same network as SCL:
   "DB1_SalidasExterioresDeMesa".Mesa[#Mesa].Bajar_TP_E1E3 := (((#Mx_ET10 OR #Mx_ET11 OR #Mx_ET12 OR (#Mx_ET51 AND #Simultaneo_Mx)) AND (((#CNTSeg_pHsMx.CVU < #V_Bajar_TP_Max) AND #OrdSal_S03) OR (NOT "DB1_SalidasExterioresDeMesa".Mesa[#Mesa].Subir_TP_E1E3 AND NOT #TP1_Up))) OR (#Mx_ET02 AND (#OrdSal_S03 OR (NOT "DB1_SalidasExterioresDeMesa".Mesa[#Mesa].Subir_TP_E1E3 AND NOT #TP1_Up))) OR #Mx_ET50 OR (#Mx_ET51 AND NOT #Simultaneo_Mx) OR (NOT #Mx_ET10 AND NOT #Mx_ET11 AND NOT #Mx_ET12 AND NOT #Mx_ET02 AND NOT #Mx_ET51)) AND NOT #TP1_Down AND #EstadoZona.Marcha_CBx AND NOT #EstadoVI.Error_Mx AND NOT #Error_Tx;
END_REGION

REGION Network 66: SALIDAS - Subir Tope TP1 NOTA: Tope E1 >> S3
   RUNG wire#powerrail
      Contact( #Mx_ET10 )
      wire#w1
      I_Contact( #OrdSal_S03 )
      wire#w2
      { S7_Templates := "SrcType := Int" } GE_Contact(in1 := #CNTSeg_pHsMx.CVU, in2 := #V_Subir_TP_Min)
      wire#w3
      I_Contact( #TP1_Up )
      Contact( #EstadoZona.Marcha_CBx )
      I_Contact( #EstadoVI.Error_Mx )
      I_Contact( #Error_Tx )
      Coil( "DB1_SalidasExterioresDeMesa".Mesa[#Mesa].Subir_TP_E1E3 )
   END_RUNG
   RUNG wire#powerrail
      Contact( #Mx_ET11 )
   END_RUNG wire#w1
   RUNG wire#powerrail
      Contact( #Mx_ET12 )
   END_RUNG wire#w1
   RUNG wire#powerrail
      Contact( #Mx_ET51 )
      Contact( #Simultaneo_Mx )
   END_RUNG wire#w1
   RUNG wire#w1
      Contact( #OrdSal_S03 )
      I_Contact( #PTF_Mx_MSig )
   END_RUNG wire#w2
   RUNG wire#powerrail
      Contact( #Mx_ET02 )
      I_Contact( #OrdSal_S03 )
   END_RUNG wire#w3
   // the same network as SCL:
   "DB1_SalidasExterioresDeMesa".Mesa[#Mesa].Subir_TP_E1E3 := (((#Mx_ET10 OR #Mx_ET11 OR #Mx_ET12 OR (#Mx_ET51 AND #Simultaneo_Mx)) AND (NOT #OrdSal_S03 OR (#OrdSal_S03 AND NOT #PTF_Mx_MSig)) AND (#CNTSeg_pHsMx.CVU >= #V_Subir_TP_Min)) OR (#Mx_ET02 AND NOT #OrdSal_S03)) AND NOT #TP1_Up AND #EstadoZona.Marcha_CBx AND NOT #EstadoVI.Error_Mx AND NOT #Error_Tx;
END_REGION

REGION Network 67: ESTADOS DE LA MESA
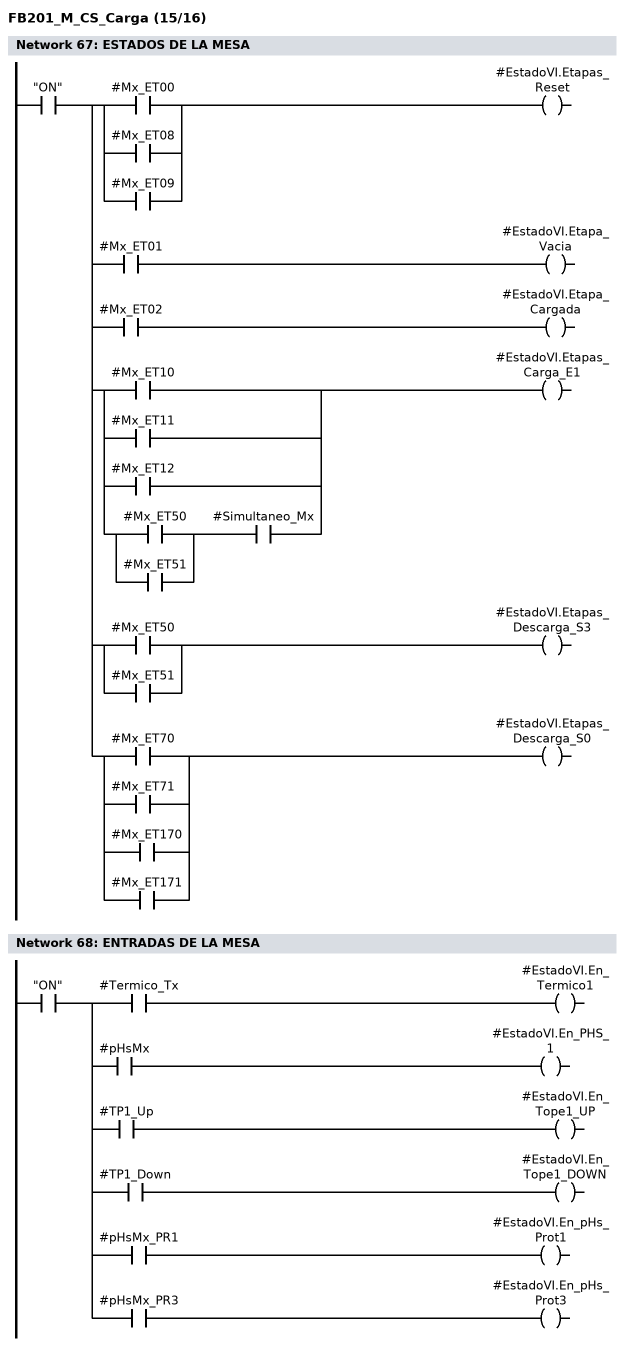
   RUNG wire#powerrail
      Contact( "ON" )
      wire#w1
      Contact( #Mx_ET00 )
      wire#w2
      Coil( #EstadoVI.Etapas_Reset )
   END_RUNG
   RUNG wire#w1
      Contact( #Mx_ET08 )
   END_RUNG wire#w2
   RUNG wire#w1
      Contact( #Mx_ET09 )
   END_RUNG wire#w2
   RUNG wire#w1
      Contact( #Mx_ET01 )
      Coil( #EstadoVI.Etapa_Vacia )
   END_RUNG
   RUNG wire#w1
      Contact( #Mx_ET02 )
      Coil( #EstadoVI.Etapa_Cargada )
   END_RUNG
   RUNG wire#w1
      Contact( #Mx_ET10 )
      wire#w3
      Coil( #EstadoVI.Etapas_Carga_E1 )
   END_RUNG
   RUNG wire#w1
      Contact( #Mx_ET11 )
   END_RUNG wire#w3
   RUNG wire#w1
      Contact( #Mx_ET12 )
   END_RUNG wire#w3
   RUNG wire#w1
      Contact( #Mx_ET50 )
      wire#w4
      Contact( #Simultaneo_Mx )
   END_RUNG wire#w3
   RUNG wire#w1
      Contact( #Mx_ET51 )
   END_RUNG wire#w4
   RUNG wire#w1
      Contact( #Mx_ET50 )
      wire#w5
      Coil( #EstadoVI.Etapas_Descarga_S3 )
   END_RUNG
   RUNG wire#w1
      Contact( #Mx_ET51 )
   END_RUNG wire#w5
   RUNG wire#w1
      Contact( #Mx_ET70 )
      wire#w6
      Coil( #EstadoVI.Etapas_Descarga_S0 )
   END_RUNG
   RUNG wire#w1
      Contact( #Mx_ET71 )
   END_RUNG wire#w6
   RUNG wire#w1
      Contact( #Mx_ET170 )
   END_RUNG wire#w6
   RUNG wire#w1
      Contact( #Mx_ET171 )
   END_RUNG wire#w6
   // the same network as SCL:
   #EstadoVI.Etapas_Reset := "ON" AND (#Mx_ET00 OR #Mx_ET08 OR #Mx_ET09);
   #EstadoVI.Etapa_Vacia := "ON" AND #Mx_ET01;
   #EstadoVI.Etapa_Cargada := "ON" AND #Mx_ET02;
   #EstadoVI.Etapas_Carga_E1 := "ON" AND (#Mx_ET10 OR #Mx_ET11 OR #Mx_ET12 OR ((#Mx_ET50 OR #Mx_ET51) AND #Simultaneo_Mx));
   #EstadoVI.Etapas_Descarga_S3 := "ON" AND (#Mx_ET50 OR #Mx_ET51);
   #EstadoVI.Etapas_Descarga_S0 := "ON" AND (#Mx_ET70 OR #Mx_ET71 OR #Mx_ET170 OR #Mx_ET171);
END_REGION

REGION Network 68: ENTRADAS DE LA MESA
   RUNG wire#powerrail
      Contact( "ON" )
      wire#w1
      Contact( #Termico_Tx )
      Coil( #EstadoVI.En_Termico1 )
   END_RUNG
   RUNG wire#w1
      Contact( #pHsMx )
      Coil( #EstadoVI.En_PHS_1 )
   END_RUNG
   RUNG wire#w1
      Contact( #TP1_Up )
      Coil( #EstadoVI.En_Tope1_UP )
   END_RUNG
   RUNG wire#w1
      Contact( #TP1_Down )
      Coil( #EstadoVI.En_Tope1_DOWN )
   END_RUNG
   RUNG wire#w1
      Contact( #pHsMx_PR1 )
      Coil( #EstadoVI.En_pHs_Prot1 )
   END_RUNG
   RUNG wire#w1
      Contact( #pHsMx_PR3 )
      Coil( #EstadoVI.En_pHs_Prot3 )
   END_RUNG
   // the same network as SCL:
   #EstadoVI.En_Termico1 := "ON" AND #Termico_Tx;
   #EstadoVI.En_PHS_1 := "ON" AND #pHsMx;
   #EstadoVI.En_Tope1_UP := "ON" AND #TP1_Up;
   #EstadoVI.En_Tope1_DOWN := "ON" AND #TP1_Down;
   #EstadoVI.En_pHs_Prot1 := "ON" AND #pHsMx_PR1;
   #EstadoVI.En_pHs_Prot3 := "ON" AND #pHsMx_PR3;
END_REGION

REGION Network 69: SALIDAS DE LA MESA
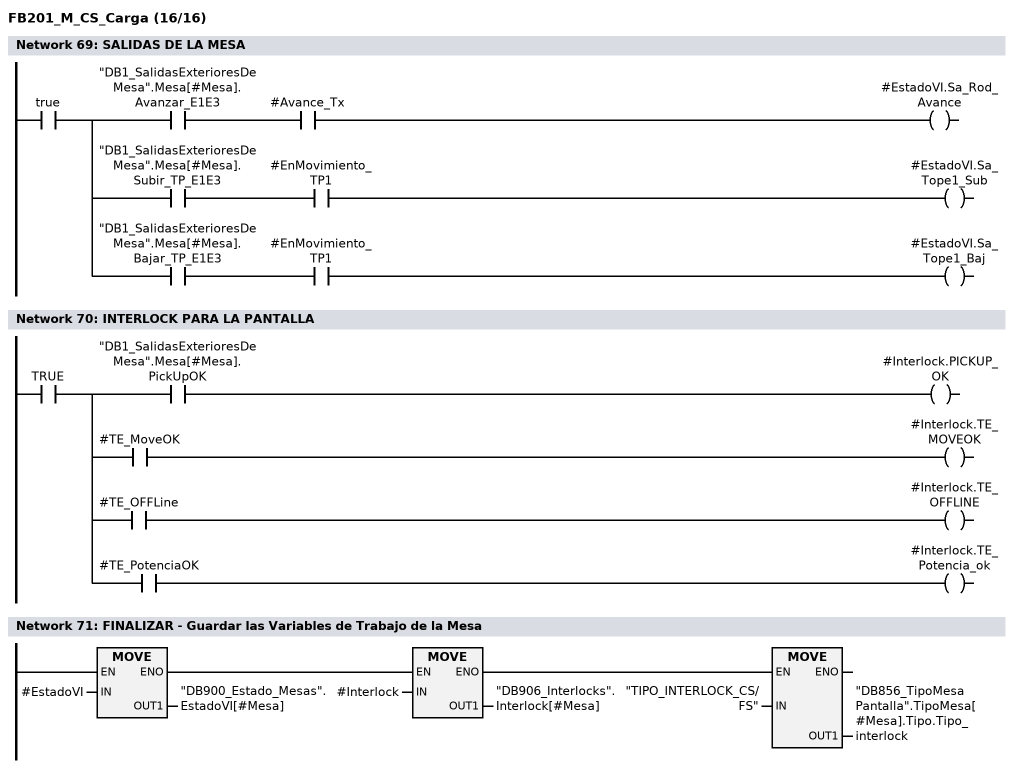
   RUNG wire#powerrail
      Contact( true )
      wire#w1
      Contact( "DB1_SalidasExterioresDeMesa".Mesa[#Mesa].Avanzar_E1E3 )
      Contact( #Avance_Tx )
      Coil( #EstadoVI.Sa_Rod_Avance )
   END_RUNG
   RUNG wire#w1
      Contact( "DB1_SalidasExterioresDeMesa".Mesa[#Mesa].Subir_TP_E1E3 )
      Contact( #EnMovimiento_TP1 )
      Coil( #EstadoVI.Sa_Tope1_Sub )
   END_RUNG
   RUNG wire#w1
      Contact( "DB1_SalidasExterioresDeMesa".Mesa[#Mesa].Bajar_TP_E1E3 )
      Contact( #EnMovimiento_TP1 )
      Coil( #EstadoVI.Sa_Tope1_Baj )
   END_RUNG
   // the same network as SCL:
   #EstadoVI.Sa_Rod_Avance := true AND "DB1_SalidasExterioresDeMesa".Mesa[#Mesa].Avanzar_E1E3 AND #Avance_Tx;
   #EstadoVI.Sa_Tope1_Sub := true AND "DB1_SalidasExterioresDeMesa".Mesa[#Mesa].Subir_TP_E1E3 AND #EnMovimiento_TP1;
   #EstadoVI.Sa_Tope1_Baj := true AND "DB1_SalidasExterioresDeMesa".Mesa[#Mesa].Bajar_TP_E1E3 AND #EnMovimiento_TP1;
END_REGION

REGION Network 70: INTERLOCK PARA LA PANTALLA
   RUNG wire#powerrail
      Contact( TRUE )
      wire#w1
      Contact( "DB1_SalidasExterioresDeMesa".Mesa[#Mesa].PickUpOK )
      Coil( #Interlock.PICKUP_OK )
   END_RUNG
   RUNG wire#w1
      Contact( #TE_MoveOK )
      Coil( #Interlock.TE_MOVEOK )
   END_RUNG
   RUNG wire#w1
      Contact( #TE_OFFLine )
      Coil( #Interlock.TE_OFFLINE )
   END_RUNG
   RUNG wire#w1
      Contact( #TE_PotenciaOK )
      Coil( #Interlock.TE_Potencia_ok )
   END_RUNG
   // the same network as SCL:
   #Interlock.PICKUP_OK := TRUE AND "DB1_SalidasExterioresDeMesa".Mesa[#Mesa].PickUpOK;
   #Interlock.TE_MOVEOK := TRUE AND #TE_MoveOK;
   #Interlock.TE_OFFLINE := TRUE AND #TE_OFFLine;
   #Interlock.TE_Potencia_ok := TRUE AND #TE_PotenciaOK;
END_REGION

REGION Network 71: FINALIZAR - Guardar las Variables de Trabajo de la Mesa
   RUNG wire#powerrail
      Move(in := #EstadoVI, out1 => "DB900_Estado_Mesas".EstadoVI[#Mesa])
      Move(in := #Interlock, out1 => "DB906_Interlocks".Interlock[#Mesa])
      Move(in := "TIPO_INTERLOCK_CS/FS", out1 => "DB856_TipoMesaPantalla".TipoMesa[#Mesa].Tipo.Tipo_interlock)
   END_RUNG
   // the same network as SCL:
   "DB900_Estado_Mesas".EstadoVI[#Mesa] := #EstadoVI;
   "DB906_Interlocks".Interlock[#Mesa] := #Interlock;
   "DB856_TipoMesaPantalla".TipoMesa[#Mesa].Tipo.Tipo_interlock := "TIPO_INTERLOCK_CS/FS";
END_REGION
END_FUNCTION_BLOCK

FUNCTION_BLOCK "FB204_M_CS_Carga_TPCentral"   // FB204, LAD
TITLE = Control del Ramal de Salidas
{ S7_Optimized_Access := 'FALSE' }
AUTHOR : TE_CS
NAME : 20160509
VERSION : 3.4
// stored: AutoNumber false, SetENOAutomatically false
   VAR_INPUT
      Mesa : UInt;   // Mesa de la FB
      Error_Tx : Bool;   // Error en el Tx
      EnTension : Bool;   // Existe Tension en la Mesa
      Termico_Tx : Bool;   // Proteccion del Tx
      pHsMx : Bool;   // pHs de la Mesa
      Avance_Tx : Bool;   // Avance del Tx
      TCentral_Up : Bool;   // TP Central Arriba. Nota Movimiento E1 >> S3
      TPCentral_DW : Bool;   // TP Central Abajo. Nota Movimiento E1 >> S3
      EnMovimiento_TPCentral : Bool;   // En movimiento el TP Central
      TE_MoveOK : Bool;   // Move OK del TE (Horquilla Centrada)
      TE_OFFLine : Bool;   // OFF Line del TE
      TE_PotenciaOK : Bool;   // Potencia OK del TE
      MAnt_DescargaAct : Bool;   // E1 >> Mesa Anterior DescargaAct
      AVTF_MAnt_Mx : Bool;   // E1 >> Mesa Anterior AVTF
      P_Mens_MAnt_Mx : Bool;   // E1 >> Mesa Anterior P_Mens
      PTF_Mx_MSig : Bool;   // S3 >> Mesa Siguiente PTF
      FTF_Mx_MSig : Bool;   // S3 >> Mesa Siguiente FTF
      MSig_CargaAct : Bool;
      Mx_VelocidadLenta_In : Bool;   // Forzar a Velociada Lenta
      F_EnvMens_Mx : Bool;   // Fin de Envio de Mensaje
      OrdSal_S03 : Bool;   // Orden de Salida por S03
      OrdSal_S00 : Bool;   // Orden de Salida por S00 (TE)
      V_CNT_pHsMx : Int := 1000;   // Valor de Presencia
      V_CNT_pHsMx_FTF : Int := 200;   // Valor para activar FTF. Nota: < = V_CNT_pHsMx.
      V_CNTSeg_pHsMx : Int := 2000;   // Valor de Seguriadad para Presencia
      V_CNT_PasoLenta : Int := 2000;   // Valor de Paso a Lenta
      V_CNT_SubirTPCentral : Int := 2000;   // Valor para Subir TP Central
      V_CNT_ApHsMx : Int := 200;   // Valor de Ausencia
      V_CNTSeg_ApHsMx : Int := 2000;   // Valor de Seguriadad para Ausencia
      V_TOut_Tx_Mx : Int := 15000;   // TimeOut de Entrada por E1
      V_TOut_TPCentral : Int := 5000;   // TimeOut de Tope Central
      V_CNT_PerdidapHs : Int := 1000;   // CNT de Perdida de pHs
   END_VAR
   VAR_OUTPUT
      P_EnvMens_PMx : Bool;   // Permiso de Enviar Mensaje de Presencia
      P_EnvMens_AMx : Bool;   // Permiso de Enviar Mensaje de Ausencia
      P_RecepOK_Mx : Bool;   // Recepcion OK
      PTF_MAnt_Mx : Bool;   // E1 >> Mesa Anterior PTF
      FTF_MAnt_Mx : Bool;   // E1 >> Mesa Anterior FTF
      AVTF_Mx_MSig : Bool;   // S3 >> Mesa Siguiente AVTF
      P_Mens_Mx_MSig : Bool;   // S3 >> Mesa Siguiente P_Mens
   END_VAR
   VAR
      Anular_prE1 : Bool;   // ???
      Anular_prS3 : Bool;   // ???
      Mx_ET00 : Bool;
      Mx_ET01 : Bool;
      Mx_ET02 : Bool;
      Mx_ET08 : Bool;
      Mx_ET09 : Bool;
      Mx_ET10 : Bool;
      Mx_ET10TP : Bool;
      Mx_ET11 : Bool;
      Mx_ET12 : Bool;
      Mx_ET110 : Bool;
      Mx_ET111 : Bool;
      Mx_ET50 : Bool;
      Mx_ET51 : Bool;
      Mx_ET150 : Bool;
      Mx_ET151 : Bool;
      Mx_ET70 : Bool;
      Mx_ET71 : Bool;
      Mx_ET170 : Bool;
      Mx_ET171 : Bool;
      TE_OK : Bool;   // El TE esta Operativo
      ProtocoloIniciado : Bool;   // Iniciado el Envio del Mensaje de Presencia
      CNT_pHsMx_FTF_OK : Bool;   // Enviar ya FTF
      STAT_EnvMens_PMx : Bool;   // Interna >> Envio del Mensaje de Presencia
      STAT_EnvMens_AMx : Bool;   // Interna >> Envio de Mensaje de Ausencia
      STAT_FTF_MAnt_Mx : Bool;   // Interna >> FTF de MAnt >> Mx
      STAT_AVTF_Mx_MSig : Bool;   // Interna >> AVTF de Mx >> MSig
      CNT_pHsMx { S7_SetPoint := 'True'} : "FB910_CNT_UHS";   // CNT de la Presencia
      CNTSeg_pHsMx { S7_SetPoint := 'True'} : "FB910_CNT_UHS";   // CNT de Seguridad de la Presencia
      CNT_ApHsMx { S7_SetPoint := 'True'} : "FB910_CNT_UHS";   // CNT de la Ausencia
      CNTSeg_ApHsMx { S7_SetPoint := 'True'} : "FB910_CNT_UHS";   // CNT de Seguridad de la Ausencia
      CNT_SubirTPCentral { S7_SetPoint := 'True'} : "FB910_CNT_UHS";   // CNT para Subir TP Central
      TMP_EnTension { S7_SetPoint := 'True'} : "FB910_CNT_UHS";
      TOut_Av_Mx { S7_SetPoint := 'True'} : "FB910_CNT_UHS";   // Time Out de Entrada de E1
      TOut_Subir_TPCentral { S7_SetPoint := 'True'} : "FB910_CNT_UHS";   // Time Out de Subida del TP
      TOut_Bajar_TPCentral { S7_SetPoint := 'True'} : "FB910_CNT_UHS";   // Time Out de Bajada del TP
      CNT_PerdidapHs { S7_SetPoint := 'True'} : "FB910_CNT_UHS";   // CNT de Perdida de pHs
      Interlock_manual { S7_SetPoint := 'True'} : "UDT_Interlock_manual_TE_CS/FS";
   END_VAR
   VAR_TEMP
      EstadoZona : "EstadoZona";   // Estado de Zona de la Mesa
      EstadoVI : "EstadosMesa";   // Estado del Vehiculo Inteliguente de la Mesa
      ConfigFB : "UDT_ConfigFB";   // Configuracion de la FB de la Mesa
      Interlock : "UDT_Interlock_TE_CS/FS";
      V_Protrusion : Int;
      retval : Int;
      cero : USInt;
      Aux_ET00 : Bool;
   END_VAR
BEGIN

REGION Network 1: CONTROL >>> TE Operativo
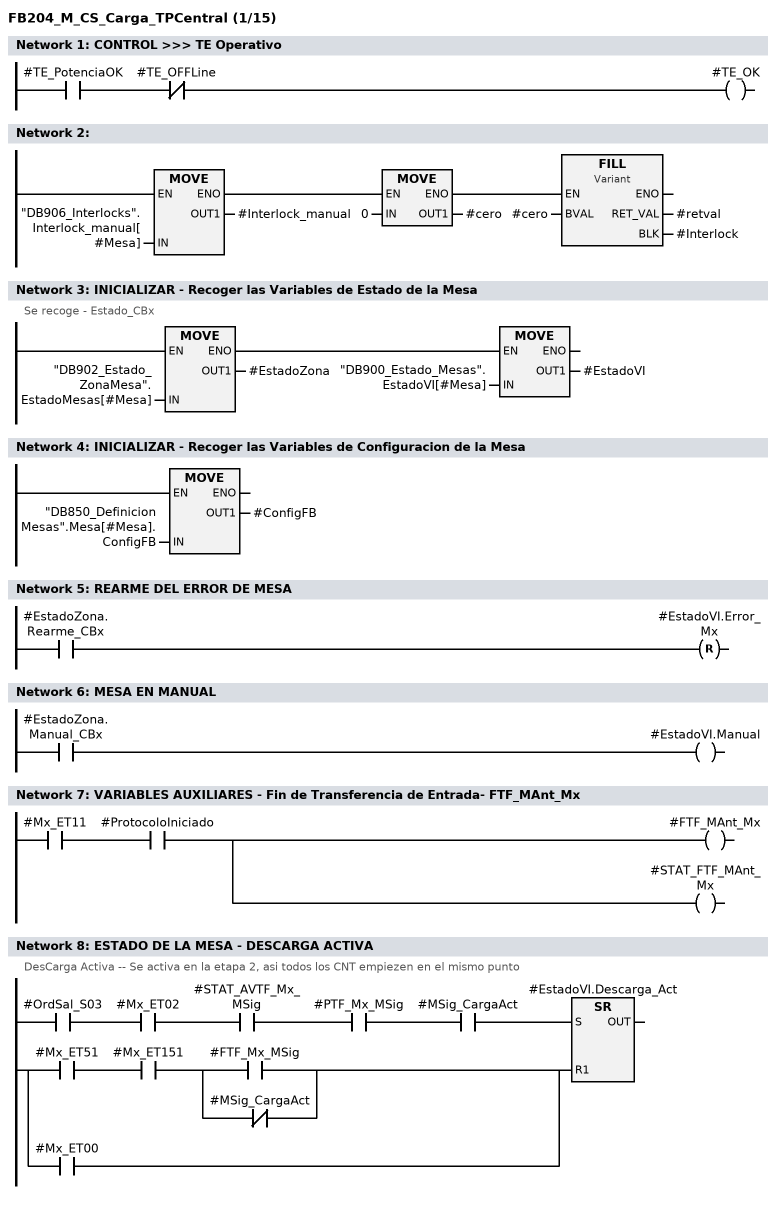
   RUNG wire#powerrail
      Contact( #TE_PotenciaOK )
      I_Contact( #TE_OFFLine )
      Coil( #TE_OK )
   END_RUNG
   // the same network as SCL:
   #TE_OK := #TE_PotenciaOK AND NOT #TE_OFFLine;
END_REGION

REGION Network 2
   RUNG wire#powerrail
      Move(in := "DB906_Interlocks".Interlock_manual[#Mesa], out1 => #Interlock_manual)
      Move(in := 0, out1 => #cero)
      { S7_Templates := "ptr_type := Variant" } FILL(BVAL := #cero, RET_VAL => #retval, BLK => #Interlock)
   END_RUNG
   // the same network as SCL:
   #Interlock_manual := "DB906_Interlocks".Interlock_manual[#Mesa];
   #cero := 0;
   #retval := FILL(BVAL := #cero, BLK => #Interlock);
END_REGION

REGION Network 3: INICIALIZAR - Recoger las Variables de Estado de la Mesa
   // Se recoge - Estado_CBx
   RUNG wire#powerrail
      Move(in := "DB902_Estado_ZonaMesa".EstadoMesas[#Mesa], out1 => #EstadoZona)
      Move(in := "DB900_Estado_Mesas".EstadoVI[#Mesa], out1 => #EstadoVI)
   END_RUNG
   // the same network as SCL:
   #EstadoZona := "DB902_Estado_ZonaMesa".EstadoMesas[#Mesa];
   #EstadoVI := "DB900_Estado_Mesas".EstadoVI[#Mesa];
END_REGION

REGION Network 4: INICIALIZAR - Recoger las Variables de Configuracion de la Mesa
   RUNG wire#powerrail
      Move(in := "DB850_DefinicionMesas".Mesa[#Mesa].ConfigFB, out1 => #ConfigFB)
   END_RUNG
   // the same network as SCL:
   #ConfigFB := "DB850_DefinicionMesas".Mesa[#Mesa].ConfigFB;
END_REGION

REGION Network 5: REARME DEL ERROR DE MESA
   RUNG wire#powerrail
      Contact( #EstadoZona.Rearme_CBx )
      R_Coil( #EstadoVI.Error_Mx )
   END_RUNG
   // the same network as SCL:
   IF #EstadoZona.Rearme_CBx THEN #EstadoVI.Error_Mx := FALSE; END_IF;
END_REGION

REGION Network 6: MESA EN MANUAL
   RUNG wire#powerrail
      Contact( #EstadoZona.Manual_CBx )
      Coil( #EstadoVI.Manual )
   END_RUNG
   // the same network as SCL:
   #EstadoVI.Manual := #EstadoZona.Manual_CBx;
END_REGION

REGION Network 7: VARIABLES AUXILIARES - Fin de Transferencia de Entrada- FTF_MAnt_Mx
   RUNG wire#powerrail
      Contact( #Mx_ET11 )
      Contact( #ProtocoloIniciado )
      wire#w1
      Coil( #FTF_MAnt_Mx )
   END_RUNG
   RUNG wire#w1
      Coil( #STAT_FTF_MAnt_Mx )
   END_RUNG
   // the same network as SCL:
   #FTF_MAnt_Mx := #Mx_ET11 AND #ProtocoloIniciado;
   #STAT_FTF_MAnt_Mx := #FTF_MAnt_Mx;
END_REGION

REGION Network 8: ESTADO DE LA MESA - DESCARGA ACTIVA
   // DesCarga Activa -- Se activa en la etapa 2, asi todos los CNT empiezen en el mismo punto
   RUNG wire#powerrail
      Contact( #OrdSal_S03 )
      Contact( #Mx_ET02 )
      Contact( #STAT_AVTF_Mx_MSig )
      Contact( #PTF_Mx_MSig )
      Contact( #MSig_CargaAct )
      S_SR(operand := #EstadoVI.Descarga_Act, r1 := wire#w2)
   END_RUNG
   RUNG wire#powerrail
      Contact( #Mx_ET51 )
      Contact( #Mx_ET151 )
      wire#w1
      Contact( #FTF_Mx_MSig )
   END_RUNG wire#w2
   RUNG wire#w1
      I_Contact( #MSig_CargaAct )
   END_RUNG wire#w2
   RUNG wire#powerrail
      Contact( #Mx_ET00 )
   END_RUNG wire#w2
   // the same network as SCL:
   IF #OrdSal_S03 AND #Mx_ET02 AND #STAT_AVTF_Mx_MSig AND #PTF_Mx_MSig AND #MSig_CargaAct THEN
       #EstadoVI.Descarga_Act := TRUE;   // SR flip-flop
   END_IF;
   IF (#Mx_ET51 AND #Mx_ET151 AND (#FTF_Mx_MSig OR NOT #MSig_CargaAct)) OR #Mx_ET00 THEN
       #EstadoVI.Descarga_Act := FALSE;
   END_IF;
END_REGION

REGION Network 9: ET171 - CONTROL DESCARGA MESA TE - PROTOCOLO
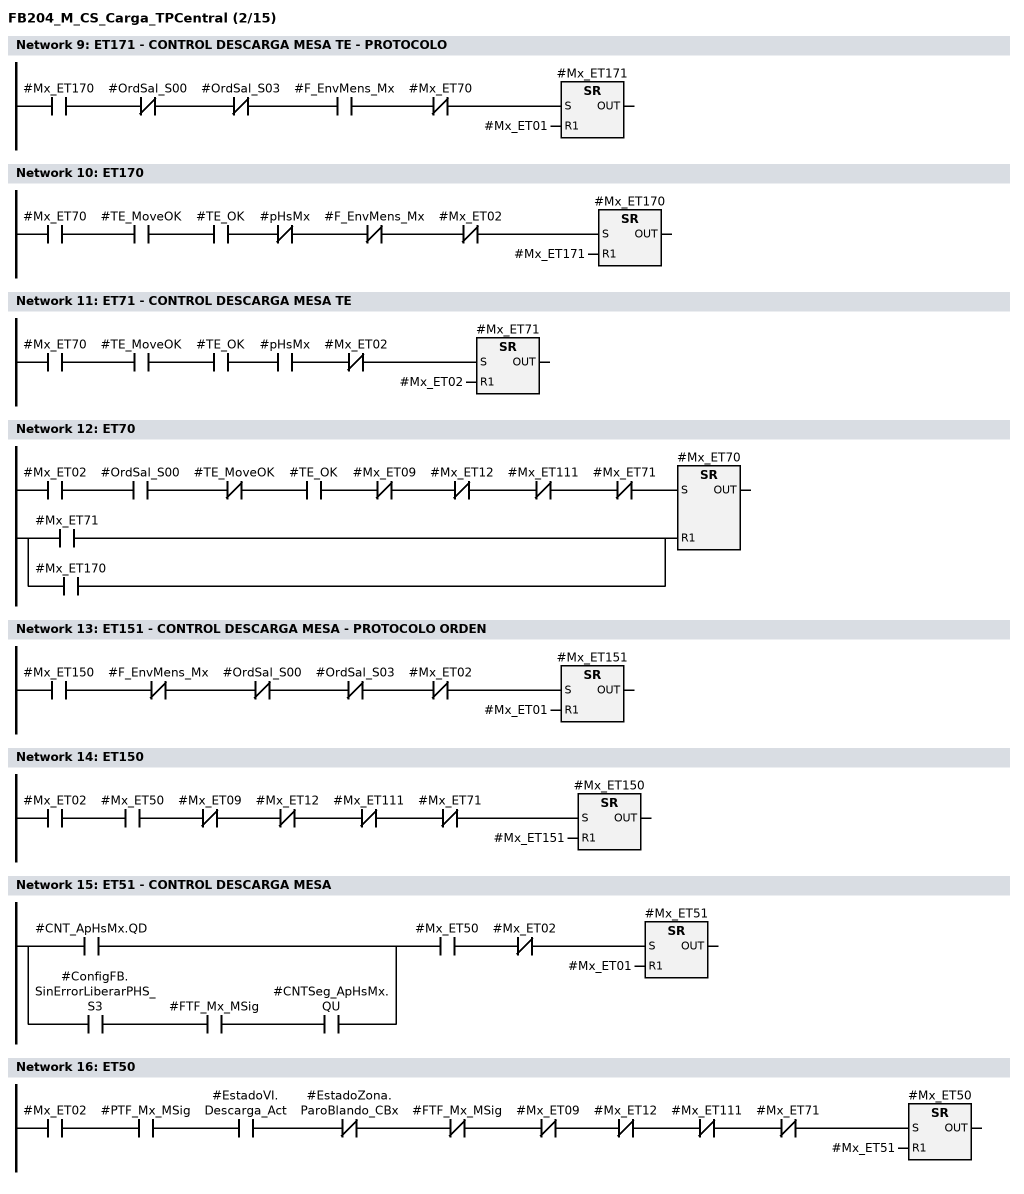
   RUNG wire#powerrail
      Contact( #Mx_ET170 )
      I_Contact( #OrdSal_S00 )
      I_Contact( #OrdSal_S03 )
      Contact( #F_EnvMens_Mx )
      I_Contact( #Mx_ET70 )
      S_SR(operand := #Mx_ET171, r1 := #Mx_ET01)
   END_RUNG
   // the same network as SCL:
   IF #Mx_ET170 AND NOT #OrdSal_S00 AND NOT #OrdSal_S03 AND #F_EnvMens_Mx AND NOT #Mx_ET70 THEN
       #Mx_ET171 := TRUE;   // SR flip-flop
   END_IF;
   IF #Mx_ET01 THEN #Mx_ET171 := FALSE; END_IF;
END_REGION

REGION Network 10: ET170
   RUNG wire#powerrail
      Contact( #Mx_ET70 )
      Contact( #TE_MoveOK )
      Contact( #TE_OK )
      I_Contact( #pHsMx )
      I_Contact( #F_EnvMens_Mx )
      I_Contact( #Mx_ET02 )
      S_SR(operand := #Mx_ET170, r1 := #Mx_ET171)
   END_RUNG
   // the same network as SCL:
   IF #Mx_ET70 AND #TE_MoveOK AND #TE_OK AND NOT #pHsMx AND NOT #F_EnvMens_Mx AND NOT #Mx_ET02 THEN
       #Mx_ET170 := TRUE;   // SR flip-flop
   END_IF;
   IF #Mx_ET171 THEN #Mx_ET170 := FALSE; END_IF;
END_REGION

REGION Network 11: ET71 - CONTROL DESCARGA MESA TE
   RUNG wire#powerrail
      Contact( #Mx_ET70 )
      Contact( #TE_MoveOK )
      Contact( #TE_OK )
      Contact( #pHsMx )
      I_Contact( #Mx_ET02 )
      S_SR(operand := #Mx_ET71, r1 := #Mx_ET02)
   END_RUNG
   // the same network as SCL:
   IF #Mx_ET70 AND #TE_MoveOK AND #TE_OK AND #pHsMx AND NOT #Mx_ET02 THEN
       #Mx_ET71 := TRUE;   // SR flip-flop
   END_IF;
   IF #Mx_ET02 THEN #Mx_ET71 := FALSE; END_IF;
END_REGION

REGION Network 12: ET70
   RUNG wire#powerrail
      Contact( #Mx_ET02 )
      Contact( #OrdSal_S00 )
      I_Contact( #TE_MoveOK )
      Contact( #TE_OK )
      I_Contact( #Mx_ET09 )
      I_Contact( #Mx_ET12 )
      I_Contact( #Mx_ET111 )
      I_Contact( #Mx_ET71 )
      S_SR(operand := #Mx_ET70, r1 := wire#w1)
   END_RUNG
   RUNG wire#powerrail
      Contact( #Mx_ET71 )
   END_RUNG wire#w1
   RUNG wire#powerrail
      Contact( #Mx_ET170 )
   END_RUNG wire#w1
   // the same network as SCL:
   IF #Mx_ET02 AND #OrdSal_S00 AND NOT #TE_MoveOK AND #TE_OK AND NOT #Mx_ET09 AND NOT #Mx_ET12 AND NOT #Mx_ET111 AND NOT #Mx_ET71 THEN
       #Mx_ET70 := TRUE;   // SR flip-flop
   END_IF;
   IF #Mx_ET71 OR #Mx_ET170 THEN #Mx_ET70 := FALSE; END_IF;
END_REGION

REGION Network 13: ET151 - CONTROL DESCARGA MESA - PROTOCOLO ORDEN
   RUNG wire#powerrail
      Contact( #Mx_ET150 )
      I_Contact( #F_EnvMens_Mx )
      I_Contact( #OrdSal_S00 )
      I_Contact( #OrdSal_S03 )
      I_Contact( #Mx_ET02 )
      S_SR(operand := #Mx_ET151, r1 := #Mx_ET01)
   END_RUNG
   // the same network as SCL:
   IF #Mx_ET150 AND NOT #F_EnvMens_Mx AND NOT #OrdSal_S00 AND NOT #OrdSal_S03 AND NOT #Mx_ET02 THEN
       #Mx_ET151 := TRUE;   // SR flip-flop
   END_IF;
   IF #Mx_ET01 THEN #Mx_ET151 := FALSE; END_IF;
END_REGION

REGION Network 14: ET150
   RUNG wire#powerrail
      Contact( #Mx_ET02 )
      Contact( #Mx_ET50 )
      I_Contact( #Mx_ET09 )
      I_Contact( #Mx_ET12 )
      I_Contact( #Mx_ET111 )
      I_Contact( #Mx_ET71 )
      S_SR(operand := #Mx_ET150, r1 := #Mx_ET151)
   END_RUNG
   // the same network as SCL:
   IF #Mx_ET02 AND #Mx_ET50 AND NOT #Mx_ET09 AND NOT #Mx_ET12 AND NOT #Mx_ET111 AND NOT #Mx_ET71 THEN
       #Mx_ET150 := TRUE;   // SR flip-flop
   END_IF;
   IF #Mx_ET151 THEN #Mx_ET150 := FALSE; END_IF;
END_REGION

REGION Network 15: ET51 - CONTROL DESCARGA MESA
   RUNG wire#powerrail
      Contact( #CNT_ApHsMx.QD )
      wire#w1
      Contact( #Mx_ET50 )
      I_Contact( #Mx_ET02 )
      S_SR(operand := #Mx_ET51, r1 := #Mx_ET01)
   END_RUNG
   RUNG wire#powerrail
      Contact( #ConfigFB.SinErrorLiberarPHS_S3 )
      Contact( #FTF_Mx_MSig )
      Contact( #CNTSeg_ApHsMx.QU )
   END_RUNG wire#w1
   // the same network as SCL:
   IF (#CNT_ApHsMx.QD OR (#ConfigFB.SinErrorLiberarPHS_S3 AND #FTF_Mx_MSig AND #CNTSeg_ApHsMx.QU)) AND #Mx_ET50 AND NOT #Mx_ET02 THEN
       #Mx_ET51 := TRUE;   // SR flip-flop
   END_IF;
   IF #Mx_ET01 THEN #Mx_ET51 := FALSE; END_IF;
END_REGION

REGION Network 16: ET50
   RUNG wire#powerrail
      Contact( #Mx_ET02 )
      Contact( #PTF_Mx_MSig )
      Contact( #EstadoVI.Descarga_Act )
      I_Contact( #EstadoZona.ParoBlando_CBx )
      I_Contact( #FTF_Mx_MSig )
      I_Contact( #Mx_ET09 )
      I_Contact( #Mx_ET12 )
      I_Contact( #Mx_ET111 )
      I_Contact( #Mx_ET71 )
      S_SR(operand := #Mx_ET50, r1 := #Mx_ET51)
   END_RUNG
   // the same network as SCL:
   IF #Mx_ET02 AND #PTF_Mx_MSig AND #EstadoVI.Descarga_Act AND NOT #EstadoZona.ParoBlando_CBx AND NOT #FTF_Mx_MSig AND NOT #Mx_ET09 AND NOT #Mx_ET12 AND NOT #Mx_ET111 AND NOT #Mx_ET71 THEN
       #Mx_ET50 := TRUE;   // SR flip-flop
   END_IF;
   IF #Mx_ET51 THEN #Mx_ET50 := FALSE; END_IF;
END_REGION

REGION Network 17: ET02 - ESTADO REPOSO CARGADA
